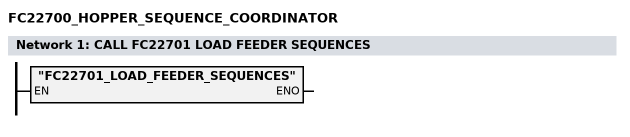
   RUNG wire#powerrail
      "FC22701_LOAD_FEEDER_SEQUENCES"()
   END_RUNG
   // the same network as SCL:
   "FC22701_LOAD_FEEDER_SEQUENCES"();
END_REGION
END_FUNCTION

FUNCTION "FC22701_LOAD_FEEDER_SEQUENCES" : Void   // FC22701, LAD
TITLE = FC22701 LOAD FEEDER SEQUENCES
{ S7_Optimized_Access := 'TRUE' }
VERSION : 0.1
// stored: AutoNumber false, IsIECCheckEnabled false, SetENOAutomatically false, UDAEnableTagReadback false
BEGIN

REGION Network 1: //////////_UNIT_01_//////////
END_REGION

REGION Network 2: /////_HOPPER_1_SEQUENCES_/////
END_REGION

REGION Network 3: CALL FB22701 LOAD FEEDER SEQUENCE TIME UNIT 01 HOPPER 1
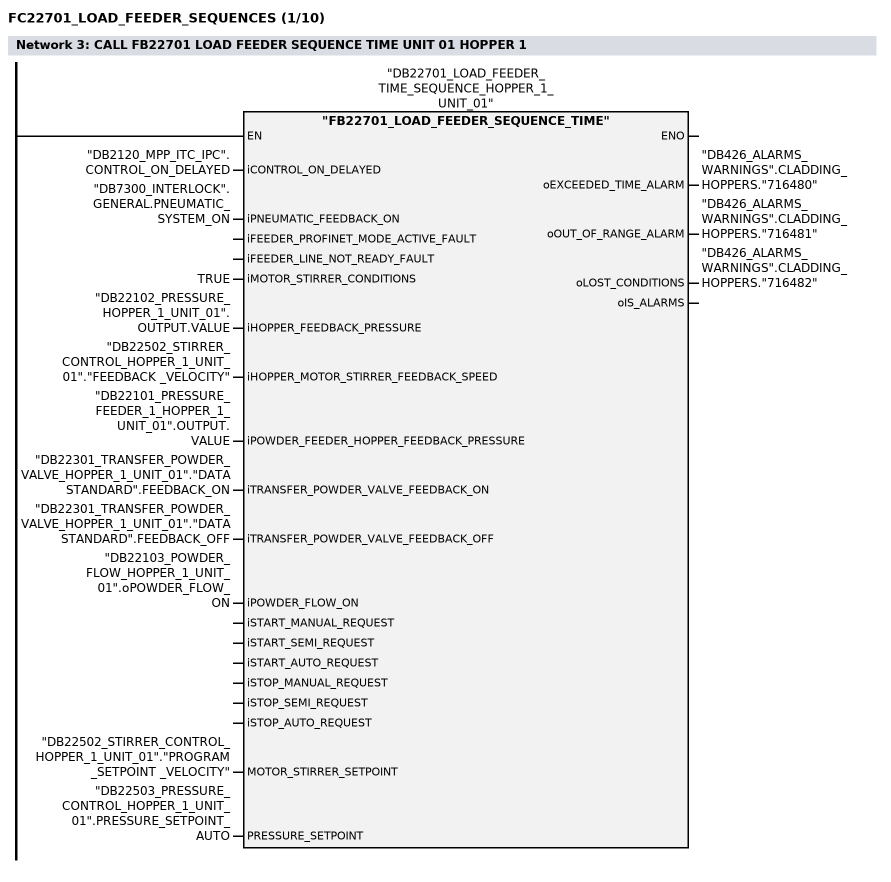
   RUNG wire#powerrail
      "DB22701_LOAD_FEEDER_TIME_SEQUENCE_HOPPER_1_UNIT_01"(iCONTROL_ON_DELAYED := "DB2120_MPP_ITC_IPC".CONTROL_ON_DELAYED, iPNEUMATIC_FEEDBACK_ON := "DB7300_INTERLOCK".GENERAL.PNEUMATIC_SYSTEM_ON, iFEEDER_PROFINET_MODE_ACTIVE_FAULT :=, iFEEDER_LINE_NOT_READY_FAULT :=, iMOTOR_STIRRER_CONDITIONS := TRUE, iHOPPER_FEEDBACK_PRESSURE := "DB22102_PRESSURE_HOPPER_1_UNIT_01".OUTPUT.VALUE, iHOPPER_MOTOR_STIRRER_FEEDBACK_SPEED := "DB22502_STIRRER_CONTROL_HOPPER_1_UNIT_01"."FEEDBACK _VELOCITY", iPOWDER_FEEDER_HOPPER_FEEDBACK_PRESSURE := "DB22101_PRESSURE_FEEDER_1_HOPPER_1_UNIT_01".OUTPUT.VALUE, iTRANSFER_POWDER_VALVE_FEEDBACK_ON := "DB22301_TRANSFER_POWDER_VALVE_HOPPER_1_UNIT_01"."DATA STANDARD".FEEDBACK_ON, iTRANSFER_POWDER_VALVE_FEEDBACK_OFF := "DB22301_TRANSFER_POWDER_VALVE_HOPPER_1_UNIT_01"."DATA STANDARD".FEEDBACK_OFF, iPOWDER_FLOW_ON := "DB22103_POWDER_FLOW_HOPPER_1_UNIT_01".oPOWDER_FLOW_ON, iSTART_MANUAL_REQUEST :=, iSTART_SEMI_REQUEST :=, iSTART_AUTO_REQUEST :=, iSTOP_MANUAL_REQUEST :=, iSTOP_SEMI_REQUEST :=, iSTOP_AUTO_REQUEST :=, MOTOR_STIRRER_SETPOINT := "DB22502_STIRRER_CONTROL_HOPPER_1_UNIT_01"."PROGRAM _SETPOINT _VELOCITY", PRESSURE_SETPOINT := "DB22503_PRESSURE_CONTROL_HOPPER_1_UNIT_01".PRESSURE_SETPOINT_AUTO, oEXCEEDED_TIME_ALARM => "DB426_ALARMS_WARNINGS".CLADDING_HOPPERS."716480", oOUT_OF_RANGE_ALARM => "DB426_ALARMS_WARNINGS".CLADDING_HOPPERS."716481", oLOST_CONDITIONS => "DB426_ALARMS_WARNINGS".CLADDING_HOPPERS."716482", oIS_ALARMS =>)
   END_RUNG
   // the same network as SCL:
   "DB22701_LOAD_FEEDER_TIME_SEQUENCE_HOPPER_1_UNIT_01"(iCONTROL_ON_DELAYED := "DB2120_MPP_ITC_IPC".CONTROL_ON_DELAYED,   // "FB22701_LOAD_FEEDER_SEQUENCE_TIME"
                           iPNEUMATIC_FEEDBACK_ON := "DB7300_INTERLOCK".GENERAL.PNEUMATIC_SYSTEM_ON,
                           iMOTOR_STIRRER_CONDITIONS := TRUE,
                           iHOPPER_FEEDBACK_PRESSURE := "DB22102_PRESSURE_HOPPER_1_UNIT_01".OUTPUT.VALUE,
                           iHOPPER_MOTOR_STIRRER_FEEDBACK_SPEED := "DB22502_STIRRER_CONTROL_HOPPER_1_UNIT_01"."FEEDBACK _VELOCITY",
                           iPOWDER_FEEDER_HOPPER_FEEDBACK_PRESSURE := "DB22101_PRESSURE_FEEDER_1_HOPPER_1_UNIT_01".OUTPUT.VALUE,
                           iTRANSFER_POWDER_VALVE_FEEDBACK_ON := "DB22301_TRANSFER_POWDER_VALVE_HOPPER_1_UNIT_01"."DATA STANDARD".FEEDBACK_ON,
                           iTRANSFER_POWDER_VALVE_FEEDBACK_OFF := "DB22301_TRANSFER_POWDER_VALVE_HOPPER_1_UNIT_01"."DATA STANDARD".FEEDBACK_OFF,
                           iPOWDER_FLOW_ON := "DB22103_POWDER_FLOW_HOPPER_1_UNIT_01".oPOWDER_FLOW_ON,
                           MOTOR_STIRRER_SETPOINT := "DB22502_STIRRER_CONTROL_HOPPER_1_UNIT_01"."PROGRAM _SETPOINT _VELOCITY",
                           PRESSURE_SETPOINT := "DB22503_PRESSURE_CONTROL_HOPPER_1_UNIT_01".PRESSURE_SETPOINT_AUTO,
                           oEXCEEDED_TIME_ALARM => "DB426_ALARMS_WARNINGS".CLADDING_HOPPERS."716480",
                           oOUT_OF_RANGE_ALARM => "DB426_ALARMS_WARNINGS".CLADDING_HOPPERS."716481",
                           oLOST_CONDITIONS => "DB426_ALARMS_WARNINGS".CLADDING_HOPPERS."716482");
END_REGION

REGION Network 4: CALL FB22702 LOAD FEEDER SEQUENCE WEIGHT UNIT 01 HOPPER 1
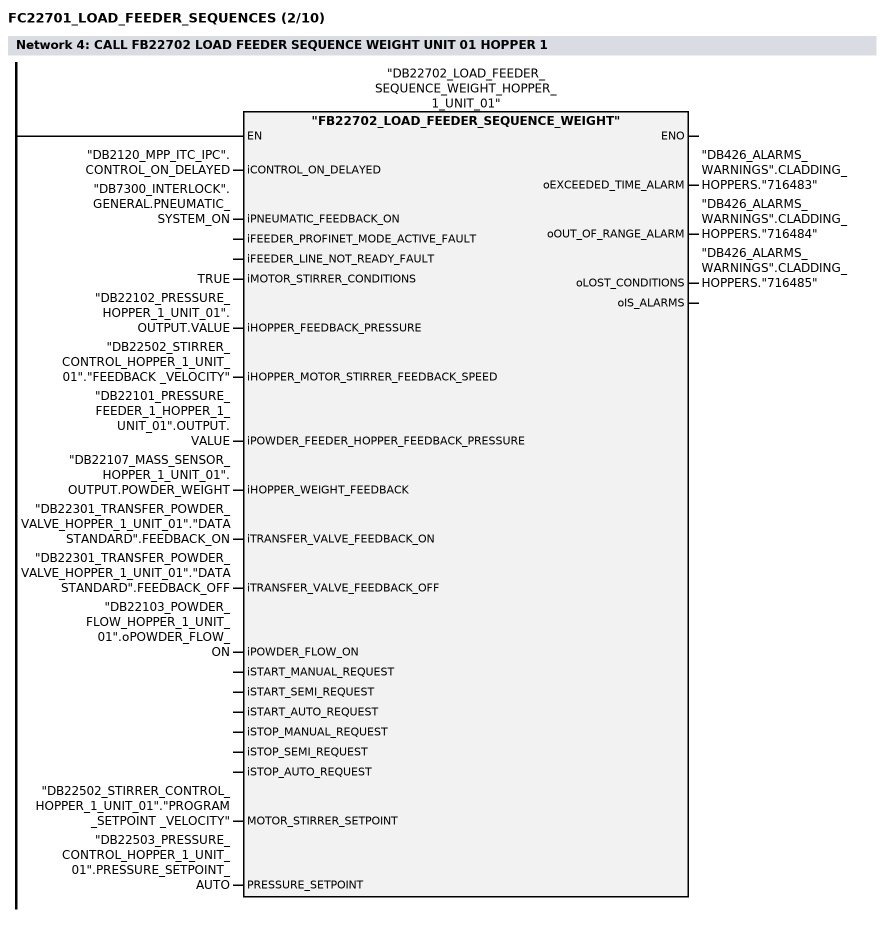
   RUNG wire#powerrail
      "DB22702_LOAD_FEEDER_SEQUENCE_WEIGHT_HOPPER_1_UNIT_01"(iCONTROL_ON_DELAYED := "DB2120_MPP_ITC_IPC".CONTROL_ON_DELAYED, iPNEUMATIC_FEEDBACK_ON := "DB7300_INTERLOCK".GENERAL.PNEUMATIC_SYSTEM_ON, iFEEDER_PROFINET_MODE_ACTIVE_FAULT :=, iFEEDER_LINE_NOT_READY_FAULT :=, iMOTOR_STIRRER_CONDITIONS := TRUE, iHOPPER_FEEDBACK_PRESSURE := "DB22102_PRESSURE_HOPPER_1_UNIT_01".OUTPUT.VALUE, iHOPPER_MOTOR_STIRRER_FEEDBACK_SPEED := "DB22502_STIRRER_CONTROL_HOPPER_1_UNIT_01"."FEEDBACK _VELOCITY", iPOWDER_FEEDER_HOPPER_FEEDBACK_PRESSURE := "DB22101_PRESSURE_FEEDER_1_HOPPER_1_UNIT_01".OUTPUT.VALUE, iHOPPER_WEIGHT_FEEDBACK := "DB22107_MASS_SENSOR_HOPPER_1_UNIT_01".OUTPUT.POWDER_WEIGHT, iTRANSFER_VALVE_FEEDBACK_ON := "DB22301_TRANSFER_POWDER_VALVE_HOPPER_1_UNIT_01"."DATA STANDARD".FEEDBACK_ON, iTRANSFER_VALVE_FEEDBACK_OFF := "DB22301_TRANSFER_POWDER_VALVE_HOPPER_1_UNIT_01"."DATA STANDARD".FEEDBACK_OFF, iPOWDER_FLOW_ON := "DB22103_POWDER_FLOW_HOPPER_1_UNIT_01".oPOWDER_FLOW_ON, iSTART_MANUAL_REQUEST :=, iSTART_SEMI_REQUEST :=, iSTART_AUTO_REQUEST :=, iSTOP_MANUAL_REQUEST :=, iSTOP_SEMI_REQUEST :=, iSTOP_AUTO_REQUEST :=, MOTOR_STIRRER_SETPOINT := "DB22502_STIRRER_CONTROL_HOPPER_1_UNIT_01"."PROGRAM _SETPOINT _VELOCITY", PRESSURE_SETPOINT := "DB22503_PRESSURE_CONTROL_HOPPER_1_UNIT_01".PRESSURE_SETPOINT_AUTO, oEXCEEDED_TIME_ALARM => "DB426_ALARMS_WARNINGS".CLADDING_HOPPERS."716483", oOUT_OF_RANGE_ALARM => "DB426_ALARMS_WARNINGS".CLADDING_HOPPERS."716484", oLOST_CONDITIONS => "DB426_ALARMS_WARNINGS".CLADDING_HOPPERS."716485", oIS_ALARMS =>)
   END_RUNG
   // the same network as SCL:
   "DB22702_LOAD_FEEDER_SEQUENCE_WEIGHT_HOPPER_1_UNIT_01"(iCONTROL_ON_DELAYED := "DB2120_MPP_ITC_IPC".CONTROL_ON_DELAYED,   // "FB22702_LOAD_FEEDER_SEQUENCE_WEIGHT"
                           iPNEUMATIC_FEEDBACK_ON := "DB7300_INTERLOCK".GENERAL.PNEUMATIC_SYSTEM_ON,
                           iMOTOR_STIRRER_CONDITIONS := TRUE,
                           iHOPPER_FEEDBACK_PRESSURE := "DB22102_PRESSURE_HOPPER_1_UNIT_01".OUTPUT.VALUE,
                           iHOPPER_MOTOR_STIRRER_FEEDBACK_SPEED := "DB22502_STIRRER_CONTROL_HOPPER_1_UNIT_01"."FEEDBACK _VELOCITY",
                           iPOWDER_FEEDER_HOPPER_FEEDBACK_PRESSURE := "DB22101_PRESSURE_FEEDER_1_HOPPER_1_UNIT_01".OUTPUT.VALUE,
                           iHOPPER_WEIGHT_FEEDBACK := "DB22107_MASS_SENSOR_HOPPER_1_UNIT_01".OUTPUT.POWDER_WEIGHT,
                           iTRANSFER_VALVE_FEEDBACK_ON := "DB22301_TRANSFER_POWDER_VALVE_HOPPER_1_UNIT_01"."DATA STANDARD".FEEDBACK_ON,
                           iTRANSFER_VALVE_FEEDBACK_OFF := "DB22301_TRANSFER_POWDER_VALVE_HOPPER_1_UNIT_01"."DATA STANDARD".FEEDBACK_OFF,
                           iPOWDER_FLOW_ON := "DB22103_POWDER_FLOW_HOPPER_1_UNIT_01".oPOWDER_FLOW_ON,
                           MOTOR_STIRRER_SETPOINT := "DB22502_STIRRER_CONTROL_HOPPER_1_UNIT_01"."PROGRAM _SETPOINT _VELOCITY",
                           PRESSURE_SETPOINT := "DB22503_PRESSURE_CONTROL_HOPPER_1_UNIT_01".PRESSURE_SETPOINT_AUTO,
                           oEXCEEDED_TIME_ALARM => "DB426_ALARMS_WARNINGS".CLADDING_HOPPERS."716483",
                           oOUT_OF_RANGE_ALARM => "DB426_ALARMS_WARNINGS".CLADDING_HOPPERS."716484",
                           oLOST_CONDITIONS => "DB426_ALARMS_WARNINGS".CLADDING_HOPPERS."716485");
END_REGION

REGION Network 5: /////_HOPPER_2_SEQUENCES_/////
END_REGION

REGION Network 6: CALL FB22701 LOAD FEEDER SEQUENCE TIME UNIT 01 HOPPER 2
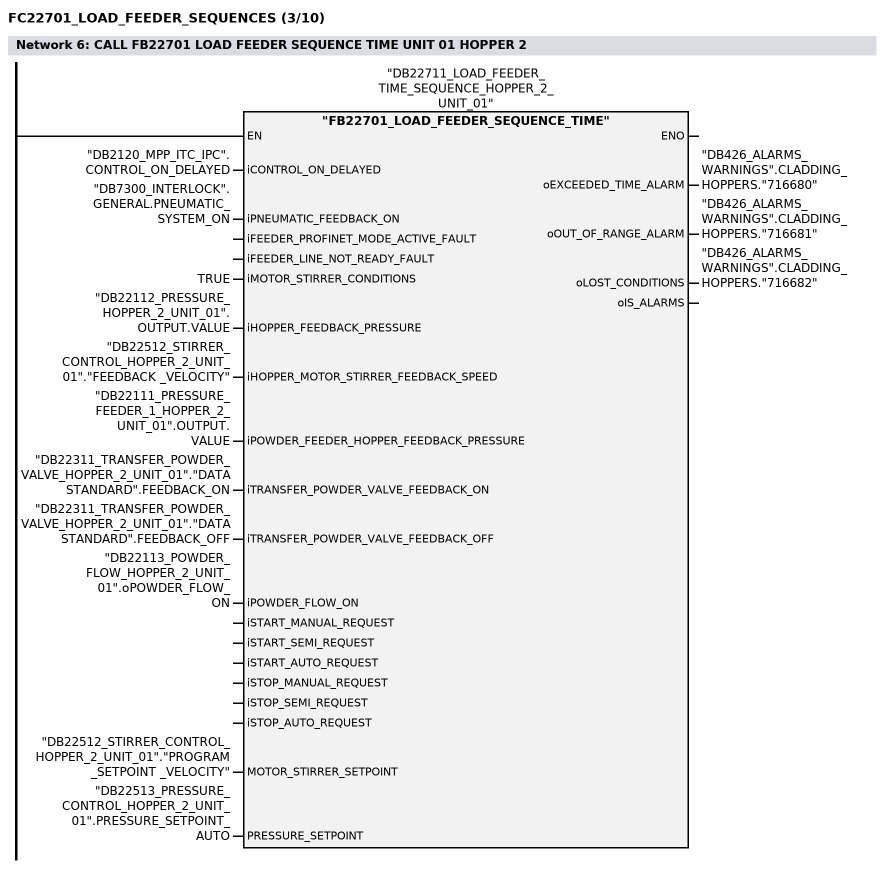
   RUNG wire#powerrail
      "DB22711_LOAD_FEEDER_TIME_SEQUENCE_HOPPER_2_UNIT_01"(iCONTROL_ON_DELAYED := "DB2120_MPP_ITC_IPC".CONTROL_ON_DELAYED, iPNEUMATIC_FEEDBACK_ON := "DB7300_INTERLOCK".GENERAL.PNEUMATIC_SYSTEM_ON, iFEEDER_PROFINET_MODE_ACTIVE_FAULT :=, iFEEDER_LINE_NOT_READY_FAULT :=, iMOTOR_STIRRER_CONDITIONS := TRUE, iHOPPER_FEEDBACK_PRESSURE := "DB22112_PRESSURE_HOPPER_2_UNIT_01".OUTPUT.VALUE, iHOPPER_MOTOR_STIRRER_FEEDBACK_SPEED := "DB22512_STIRRER_CONTROL_HOPPER_2_UNIT_01"."FEEDBACK _VELOCITY", iPOWDER_FEEDER_HOPPER_FEEDBACK_PRESSURE := "DB22111_PRESSURE_FEEDER_1_HOPPER_2_UNIT_01".OUTPUT.VALUE, iTRANSFER_POWDER_VALVE_FEEDBACK_ON := "DB22311_TRANSFER_POWDER_VALVE_HOPPER_2_UNIT_01"."DATA STANDARD".FEEDBACK_ON, iTRANSFER_POWDER_VALVE_FEEDBACK_OFF := "DB22311_TRANSFER_POWDER_VALVE_HOPPER_2_UNIT_01"."DATA STANDARD".FEEDBACK_OFF, iPOWDER_FLOW_ON := "DB22113_POWDER_FLOW_HOPPER_2_UNIT_01".oPOWDER_FLOW_ON, iSTART_MANUAL_REQUEST :=, iSTART_SEMI_REQUEST :=, iSTART_AUTO_REQUEST :=, iSTOP_MANUAL_REQUEST :=, iSTOP_SEMI_REQUEST :=, iSTOP_AUTO_REQUEST :=, MOTOR_STIRRER_SETPOINT := "DB22512_STIRRER_CONTROL_HOPPER_2_UNIT_01"."PROGRAM _SETPOINT _VELOCITY", PRESSURE_SETPOINT := "DB22513_PRESSURE_CONTROL_HOPPER_2_UNIT_01".PRESSURE_SETPOINT_AUTO, oEXCEEDED_TIME_ALARM => "DB426_ALARMS_WARNINGS".CLADDING_HOPPERS."716680", oOUT_OF_RANGE_ALARM => "DB426_ALARMS_WARNINGS".CLADDING_HOPPERS."716681", oLOST_CONDITIONS => "DB426_ALARMS_WARNINGS".CLADDING_HOPPERS."716682", oIS_ALARMS =>)
   END_RUNG
   // the same network as SCL:
   "DB22711_LOAD_FEEDER_TIME_SEQUENCE_HOPPER_2_UNIT_01"(iCONTROL_ON_DELAYED := "DB2120_MPP_ITC_IPC".CONTROL_ON_DELAYED,   // "FB22701_LOAD_FEEDER_SEQUENCE_TIME"
                           iPNEUMATIC_FEEDBACK_ON := "DB7300_INTERLOCK".GENERAL.PNEUMATIC_SYSTEM_ON,
                           iMOTOR_STIRRER_CONDITIONS := TRUE,
                           iHOPPER_FEEDBACK_PRESSURE := "DB22112_PRESSURE_HOPPER_2_UNIT_01".OUTPUT.VALUE,
                           iHOPPER_MOTOR_STIRRER_FEEDBACK_SPEED := "DB22512_STIRRER_CONTROL_HOPPER_2_UNIT_01"."FEEDBACK _VELOCITY",
                           iPOWDER_FEEDER_HOPPER_FEEDBACK_PRESSURE := "DB22111_PRESSURE_FEEDER_1_HOPPER_2_UNIT_01".OUTPUT.VALUE,
                           iTRANSFER_POWDER_VALVE_FEEDBACK_ON := "DB22311_TRANSFER_POWDER_VALVE_HOPPER_2_UNIT_01"."DATA STANDARD".FEEDBACK_ON,
                           iTRANSFER_POWDER_VALVE_FEEDBACK_OFF := "DB22311_TRANSFER_POWDER_VALVE_HOPPER_2_UNIT_01"."DATA STANDARD".FEEDBACK_OFF,
                           iPOWDER_FLOW_ON := "DB22113_POWDER_FLOW_HOPPER_2_UNIT_01".oPOWDER_FLOW_ON,
                           MOTOR_STIRRER_SETPOINT := "DB22512_STIRRER_CONTROL_HOPPER_2_UNIT_01"."PROGRAM _SETPOINT _VELOCITY",
                           PRESSURE_SETPOINT := "DB22513_PRESSURE_CONTROL_HOPPER_2_UNIT_01".PRESSURE_SETPOINT_AUTO,
                           oEXCEEDED_TIME_ALARM => "DB426_ALARMS_WARNINGS".CLADDING_HOPPERS."716680",
                           oOUT_OF_RANGE_ALARM => "DB426_ALARMS_WARNINGS".CLADDING_HOPPERS."716681",
                           oLOST_CONDITIONS => "DB426_ALARMS_WARNINGS".CLADDING_HOPPERS."716682");
END_REGION

REGION Network 7: CALL FB22702 LOAD FEEDER SEQUENCE WEIGHT UNIT 01 HOPPER 2
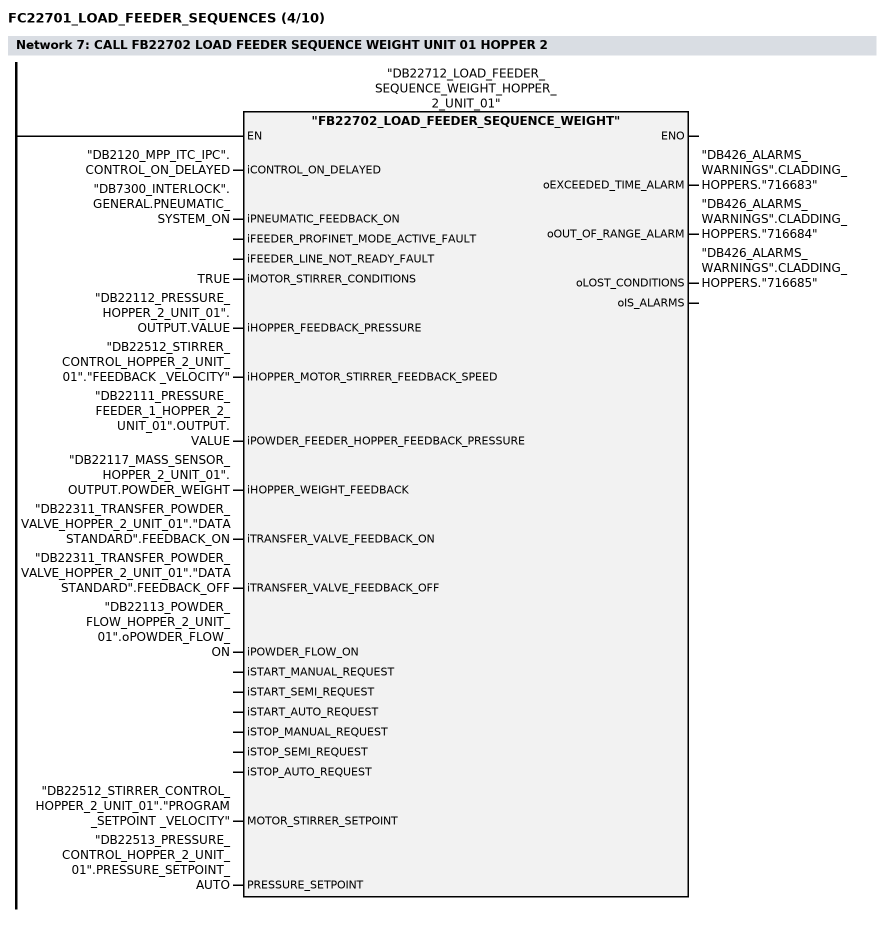
   RUNG wire#powerrail
      "DB22712_LOAD_FEEDER_SEQUENCE_WEIGHT_HOPPER_2_UNIT_01"(iCONTROL_ON_DELAYED := "DB2120_MPP_ITC_IPC".CONTROL_ON_DELAYED, iPNEUMATIC_FEEDBACK_ON := "DB7300_INTERLOCK".GENERAL.PNEUMATIC_SYSTEM_ON, iFEEDER_PROFINET_MODE_ACTIVE_FAULT :=, iFEEDER_LINE_NOT_READY_FAULT :=, iMOTOR_STIRRER_CONDITIONS := TRUE, iHOPPER_FEEDBACK_PRESSURE := "DB22112_PRESSURE_HOPPER_2_UNIT_01".OUTPUT.VALUE, iHOPPER_MOTOR_STIRRER_FEEDBACK_SPEED := "DB22512_STIRRER_CONTROL_HOPPER_2_UNIT_01"."FEEDBACK _VELOCITY", iPOWDER_FEEDER_HOPPER_FEEDBACK_PRESSURE := "DB22111_PRESSURE_FEEDER_1_HOPPER_2_UNIT_01".OUTPUT.VALUE, iHOPPER_WEIGHT_FEEDBACK := "DB22117_MASS_SENSOR_HOPPER_2_UNIT_01".OUTPUT.POWDER_WEIGHT, iTRANSFER_VALVE_FEEDBACK_ON := "DB22311_TRANSFER_POWDER_VALVE_HOPPER_2_UNIT_01"."DATA STANDARD".FEEDBACK_ON, iTRANSFER_VALVE_FEEDBACK_OFF := "DB22311_TRANSFER_POWDER_VALVE_HOPPER_2_UNIT_01"."DATA STANDARD".FEEDBACK_OFF, iPOWDER_FLOW_ON := "DB22113_POWDER_FLOW_HOPPER_2_UNIT_01".oPOWDER_FLOW_ON, iSTART_MANUAL_REQUEST :=, iSTART_SEMI_REQUEST :=, iSTART_AUTO_REQUEST :=, iSTOP_MANUAL_REQUEST :=, iSTOP_SEMI_REQUEST :=, iSTOP_AUTO_REQUEST :=, MOTOR_STIRRER_SETPOINT := "DB22512_STIRRER_CONTROL_HOPPER_2_UNIT_01"."PROGRAM _SETPOINT _VELOCITY", PRESSURE_SETPOINT := "DB22513_PRESSURE_CONTROL_HOPPER_2_UNIT_01".PRESSURE_SETPOINT_AUTO, oEXCEEDED_TIME_ALARM => "DB426_ALARMS_WARNINGS".CLADDING_HOPPERS."716683", oOUT_OF_RANGE_ALARM => "DB426_ALARMS_WARNINGS".CLADDING_HOPPERS."716684", oLOST_CONDITIONS => "DB426_ALARMS_WARNINGS".CLADDING_HOPPERS."716685", oIS_ALARMS =>)
   END_RUNG
   // the same network as SCL:
   "DB22712_LOAD_FEEDER_SEQUENCE_WEIGHT_HOPPER_2_UNIT_01"(iCONTROL_ON_DELAYED := "DB2120_MPP_ITC_IPC".CONTROL_ON_DELAYED,   // "FB22702_LOAD_FEEDER_SEQUENCE_WEIGHT"
                           iPNEUMATIC_FEEDBACK_ON := "DB7300_INTERLOCK".GENERAL.PNEUMATIC_SYSTEM_ON,
                           iMOTOR_STIRRER_CONDITIONS := TRUE,
                           iHOPPER_FEEDBACK_PRESSURE := "DB22112_PRESSURE_HOPPER_2_UNIT_01".OUTPUT.VALUE,
                           iHOPPER_MOTOR_STIRRER_FEEDBACK_SPEED := "DB22512_STIRRER_CONTROL_HOPPER_2_UNIT_01"."FEEDBACK _VELOCITY",
                           iPOWDER_FEEDER_HOPPER_FEEDBACK_PRESSURE := "DB22111_PRESSURE_FEEDER_1_HOPPER_2_UNIT_01".OUTPUT.VALUE,
                           iHOPPER_WEIGHT_FEEDBACK := "DB22117_MASS_SENSOR_HOPPER_2_UNIT_01".OUTPUT.POWDER_WEIGHT,
                           iTRANSFER_VALVE_FEEDBACK_ON := "DB22311_TRANSFER_POWDER_VALVE_HOPPER_2_UNIT_01"."DATA STANDARD".FEEDBACK_ON,
                           iTRANSFER_VALVE_FEEDBACK_OFF := "DB22311_TRANSFER_POWDER_VALVE_HOPPER_2_UNIT_01"."DATA STANDARD".FEEDBACK_OFF,
                           iPOWDER_FLOW_ON := "DB22113_POWDER_FLOW_HOPPER_2_UNIT_01".oPOWDER_FLOW_ON,
                           MOTOR_STIRRER_SETPOINT := "DB22512_STIRRER_CONTROL_HOPPER_2_UNIT_01"."PROGRAM _SETPOINT _VELOCITY",
                           PRESSURE_SETPOINT := "DB22513_PRESSURE_CONTROL_HOPPER_2_UNIT_01".PRESSURE_SETPOINT_AUTO,
                           oEXCEEDED_TIME_ALARM => "DB426_ALARMS_WARNINGS".CLADDING_HOPPERS."716683",
                           oOUT_OF_RANGE_ALARM => "DB426_ALARMS_WARNINGS".CLADDING_HOPPERS."716684",
                           oLOST_CONDITIONS => "DB426_ALARMS_WARNINGS".CLADDING_HOPPERS."716685");
END_REGION

REGION Network 8: //////////_UNIT_02_//////////
END_REGION

REGION Network 9: /////_HOPPER_1_SEQUENCES_/////
END_REGION

REGION Network 10: CALL FB22701 LOAD FEEDER SEQUENCE TIME UNIT 02 HOPPER 1
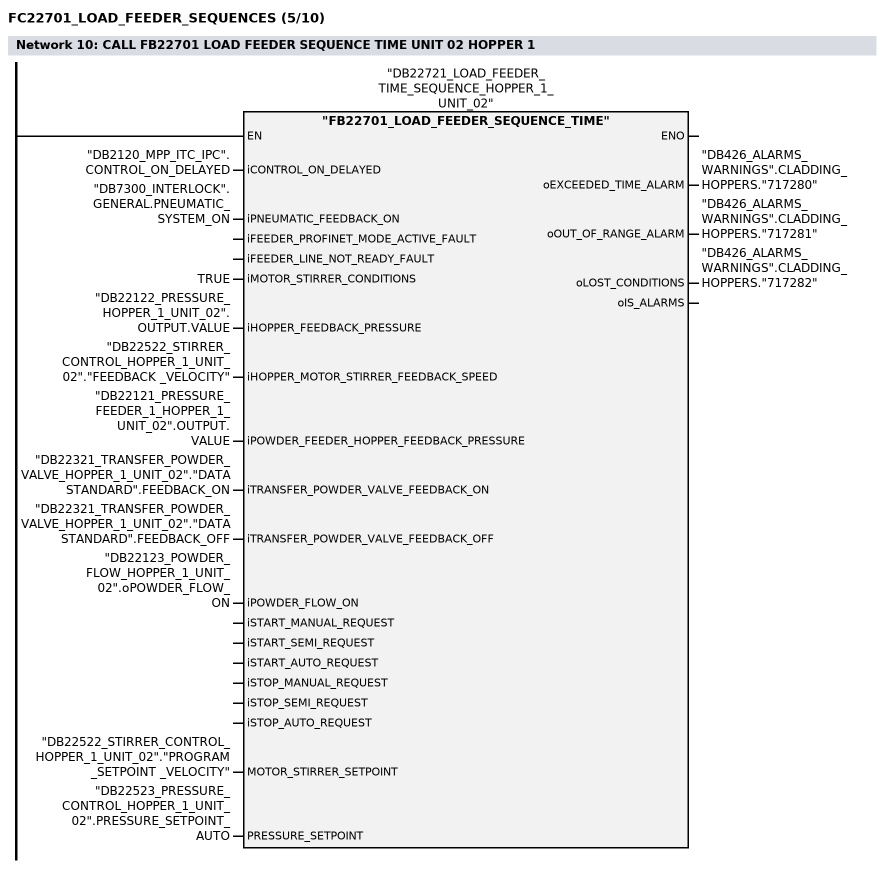
   RUNG wire#powerrail
      "DB22721_LOAD_FEEDER_TIME_SEQUENCE_HOPPER_1_UNIT_02"(iCONTROL_ON_DELAYED := "DB2120_MPP_ITC_IPC".CONTROL_ON_DELAYED, iPNEUMATIC_FEEDBACK_ON := "DB7300_INTERLOCK".GENERAL.PNEUMATIC_SYSTEM_ON, iFEEDER_PROFINET_MODE_ACTIVE_FAULT :=, iFEEDER_LINE_NOT_READY_FAULT :=, iMOTOR_STIRRER_CONDITIONS := TRUE, iHOPPER_FEEDBACK_PRESSURE := "DB22122_PRESSURE_HOPPER_1_UNIT_02".OUTPUT.VALUE, iHOPPER_MOTOR_STIRRER_FEEDBACK_SPEED := "DB22522_STIRRER_CONTROL_HOPPER_1_UNIT_02"."FEEDBACK _VELOCITY", iPOWDER_FEEDER_HOPPER_FEEDBACK_PRESSURE := "DB22121_PRESSURE_FEEDER_1_HOPPER_1_UNIT_02".OUTPUT.VALUE, iTRANSFER_POWDER_VALVE_FEEDBACK_ON := "DB22321_TRANSFER_POWDER_VALVE_HOPPER_1_UNIT_02"."DATA STANDARD".FEEDBACK_ON, iTRANSFER_POWDER_VALVE_FEEDBACK_OFF := "DB22321_TRANSFER_POWDER_VALVE_HOPPER_1_UNIT_02"."DATA STANDARD".FEEDBACK_OFF, iPOWDER_FLOW_ON := "DB22123_POWDER_FLOW_HOPPER_1_UNIT_02".oPOWDER_FLOW_ON, iSTART_MANUAL_REQUEST :=, iSTART_SEMI_REQUEST :=, iSTART_AUTO_REQUEST :=, iSTOP_MANUAL_REQUEST :=, iSTOP_SEMI_REQUEST :=, iSTOP_AUTO_REQUEST :=, MOTOR_STIRRER_SETPOINT := "DB22522_STIRRER_CONTROL_HOPPER_1_UNIT_02"."PROGRAM _SETPOINT _VELOCITY", PRESSURE_SETPOINT := "DB22523_PRESSURE_CONTROL_HOPPER_1_UNIT_02".PRESSURE_SETPOINT_AUTO, oEXCEEDED_TIME_ALARM => "DB426_ALARMS_WARNINGS".CLADDING_HOPPERS."717280", oOUT_OF_RANGE_ALARM => "DB426_ALARMS_WARNINGS".CLADDING_HOPPERS."717281", oLOST_CONDITIONS => "DB426_ALARMS_WARNINGS".CLADDING_HOPPERS."717282", oIS_ALARMS =>)
   END_RUNG
   // the same network as SCL:
   "DB22721_LOAD_FEEDER_TIME_SEQUENCE_HOPPER_1_UNIT_02"(iCONTROL_ON_DELAYED := "DB2120_MPP_ITC_IPC".CONTROL_ON_DELAYED,   // "FB22701_LOAD_FEEDER_SEQUENCE_TIME"
                           iPNEUMATIC_FEEDBACK_ON := "DB7300_INTERLOCK".GENERAL.PNEUMATIC_SYSTEM_ON,
                           iMOTOR_STIRRER_CONDITIONS := TRUE,
                           iHOPPER_FEEDBACK_PRESSURE := "DB22122_PRESSURE_HOPPER_1_UNIT_02".OUTPUT.VALUE,
                           iHOPPER_MOTOR_STIRRER_FEEDBACK_SPEED := "DB22522_STIRRER_CONTROL_HOPPER_1_UNIT_02"."FEEDBACK _VELOCITY",
                           iPOWDER_FEEDER_HOPPER_FEEDBACK_PRESSURE := "DB22121_PRESSURE_FEEDER_1_HOPPER_1_UNIT_02".OUTPUT.VALUE,
                           iTRANSFER_POWDER_VALVE_FEEDBACK_ON := "DB22321_TRANSFER_POWDER_VALVE_HOPPER_1_UNIT_02"."DATA STANDARD".FEEDBACK_ON,
                           iTRANSFER_POWDER_VALVE_FEEDBACK_OFF := "DB22321_TRANSFER_POWDER_VALVE_HOPPER_1_UNIT_02"."DATA STANDARD".FEEDBACK_OFF,
                           iPOWDER_FLOW_ON := "DB22123_POWDER_FLOW_HOPPER_1_UNIT_02".oPOWDER_FLOW_ON,
                           MOTOR_STIRRER_SETPOINT := "DB22522_STIRRER_CONTROL_HOPPER_1_UNIT_02"."PROGRAM _SETPOINT _VELOCITY",
                           PRESSURE_SETPOINT := "DB22523_PRESSURE_CONTROL_HOPPER_1_UNIT_02".PRESSURE_SETPOINT_AUTO,
                           oEXCEEDED_TIME_ALARM => "DB426_ALARMS_WARNINGS".CLADDING_HOPPERS."717280",
                           oOUT_OF_RANGE_ALARM => "DB426_ALARMS_WARNINGS".CLADDING_HOPPERS."717281",
                           oLOST_CONDITIONS => "DB426_ALARMS_WARNINGS".CLADDING_HOPPERS."717282");
END_REGION

REGION Network 11: CALL FB22702 LOAD FEEDER SEQUENCE WEIGHT UNIT 02 HOPPER 1
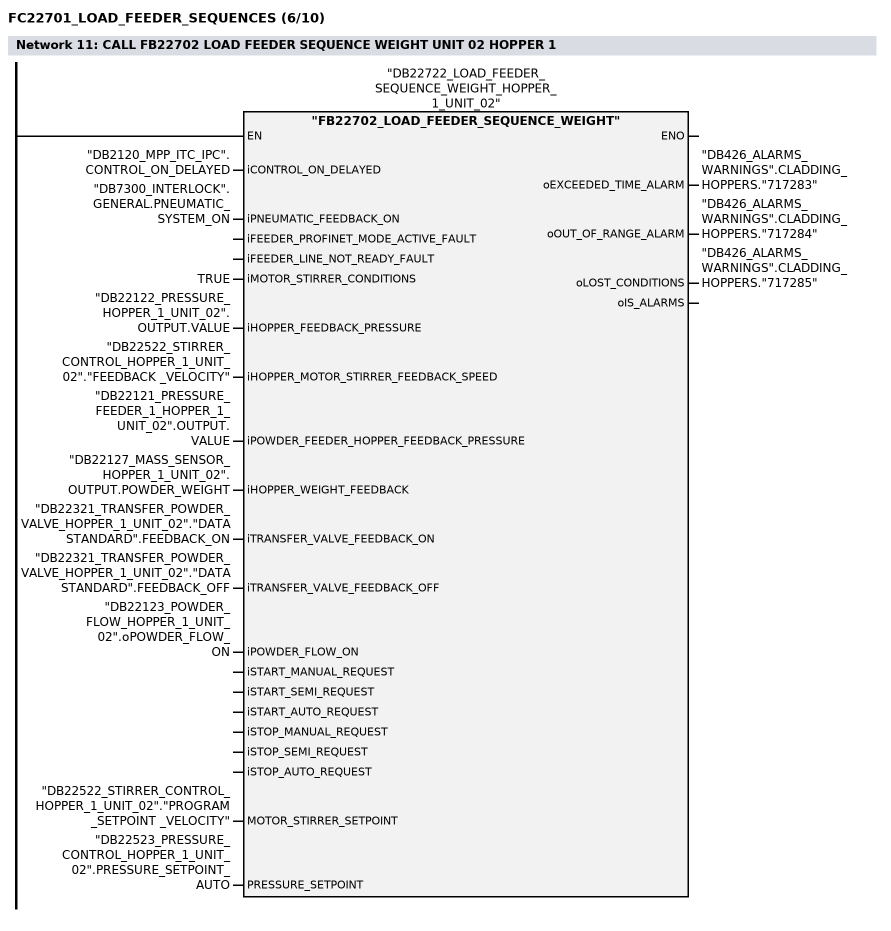
   RUNG wire#powerrail
      "DB22722_LOAD_FEEDER_SEQUENCE_WEIGHT_HOPPER_1_UNIT_02"(iCONTROL_ON_DELAYED := "DB2120_MPP_ITC_IPC".CONTROL_ON_DELAYED, iPNEUMATIC_FEEDBACK_ON := "DB7300_INTERLOCK".GENERAL.PNEUMATIC_SYSTEM_ON, iFEEDER_PROFINET_MODE_ACTIVE_FAULT :=, iFEEDER_LINE_NOT_READY_FAULT :=, iMOTOR_STIRRER_CONDITIONS := TRUE, iHOPPER_FEEDBACK_PRESSURE := "DB22122_PRESSURE_HOPPER_1_UNIT_02".OUTPUT.VALUE, iHOPPER_MOTOR_STIRRER_FEEDBACK_SPEED := "DB22522_STIRRER_CONTROL_HOPPER_1_UNIT_02"."FEEDBACK _VELOCITY", iPOWDER_FEEDER_HOPPER_FEEDBACK_PRESSURE := "DB22121_PRESSURE_FEEDER_1_HOPPER_1_UNIT_02".OUTPUT.VALUE, iHOPPER_WEIGHT_FEEDBACK := "DB22127_MASS_SENSOR_HOPPER_1_UNIT_02".OUTPUT.POWDER_WEIGHT, iTRANSFER_VALVE_FEEDBACK_ON := "DB22321_TRANSFER_POWDER_VALVE_HOPPER_1_UNIT_02"."DATA STANDARD".FEEDBACK_ON, iTRANSFER_VALVE_FEEDBACK_OFF := "DB22321_TRANSFER_POWDER_VALVE_HOPPER_1_UNIT_02"."DATA STANDARD".FEEDBACK_OFF, iPOWDER_FLOW_ON := "DB22123_POWDER_FLOW_HOPPER_1_UNIT_02".oPOWDER_FLOW_ON, iSTART_MANUAL_REQUEST :=, iSTART_SEMI_REQUEST :=, iSTART_AUTO_REQUEST :=, iSTOP_MANUAL_REQUEST :=, iSTOP_SEMI_REQUEST :=, iSTOP_AUTO_REQUEST :=, MOTOR_STIRRER_SETPOINT := "DB22522_STIRRER_CONTROL_HOPPER_1_UNIT_02"."PROGRAM _SETPOINT _VELOCITY", PRESSURE_SETPOINT := "DB22523_PRESSURE_CONTROL_HOPPER_1_UNIT_02".PRESSURE_SETPOINT_AUTO, oEXCEEDED_TIME_ALARM => "DB426_ALARMS_WARNINGS".CLADDING_HOPPERS."717283", oOUT_OF_RANGE_ALARM => "DB426_ALARMS_WARNINGS".CLADDING_HOPPERS."717284", oLOST_CONDITIONS => "DB426_ALARMS_WARNINGS".CLADDING_HOPPERS."717285", oIS_ALARMS =>)
   END_RUNG
   // the same network as SCL:
   "DB22722_LOAD_FEEDER_SEQUENCE_WEIGHT_HOPPER_1_UNIT_02"(iCONTROL_ON_DELAYED := "DB2120_MPP_ITC_IPC".CONTROL_ON_DELAYED,   // "FB22702_LOAD_FEEDER_SEQUENCE_WEIGHT"
                           iPNEUMATIC_FEEDBACK_ON := "DB7300_INTERLOCK".GENERAL.PNEUMATIC_SYSTEM_ON,
                           iMOTOR_STIRRER_CONDITIONS := TRUE,
                           iHOPPER_FEEDBACK_PRESSURE := "DB22122_PRESSURE_HOPPER_1_UNIT_02".OUTPUT.VALUE,
                           iHOPPER_MOTOR_STIRRER_FEEDBACK_SPEED := "DB22522_STIRRER_CONTROL_HOPPER_1_UNIT_02"."FEEDBACK _VELOCITY",
                           iPOWDER_FEEDER_HOPPER_FEEDBACK_PRESSURE := "DB22121_PRESSURE_FEEDER_1_HOPPER_1_UNIT_02".OUTPUT.VALUE,
                           iHOPPER_WEIGHT_FEEDBACK := "DB22127_MASS_SENSOR_HOPPER_1_UNIT_02".OUTPUT.POWDER_WEIGHT,
                           iTRANSFER_VALVE_FEEDBACK_ON := "DB22321_TRANSFER_POWDER_VALVE_HOPPER_1_UNIT_02"."DATA STANDARD".FEEDBACK_ON,
                           iTRANSFER_VALVE_FEEDBACK_OFF := "DB22321_TRANSFER_POWDER_VALVE_HOPPER_1_UNIT_02"."DATA STANDARD".FEEDBACK_OFF,
                           iPOWDER_FLOW_ON := "DB22123_POWDER_FLOW_HOPPER_1_UNIT_02".oPOWDER_FLOW_ON,
                           MOTOR_STIRRER_SETPOINT := "DB22522_STIRRER_CONTROL_HOPPER_1_UNIT_02"."PROGRAM _SETPOINT _VELOCITY",
                           PRESSURE_SETPOINT := "DB22523_PRESSURE_CONTROL_HOPPER_1_UNIT_02".PRESSURE_SETPOINT_AUTO,
                           oEXCEEDED_TIME_ALARM => "DB426_ALARMS_WARNINGS".CLADDING_HOPPERS."717283",
                           oOUT_OF_RANGE_ALARM => "DB426_ALARMS_WARNINGS".CLADDING_HOPPERS."717284",
                           oLOST_CONDITIONS => "DB426_ALARMS_WARNINGS".CLADDING_HOPPERS."717285");
END_REGION

REGION Network 12: /////_HOPPER_2_SEQUENCES_/////
END_REGION

REGION Network 13: CALL FB22701 LOAD FEEDER SEQUENCE TIME UNIT 02 HOPPER 2
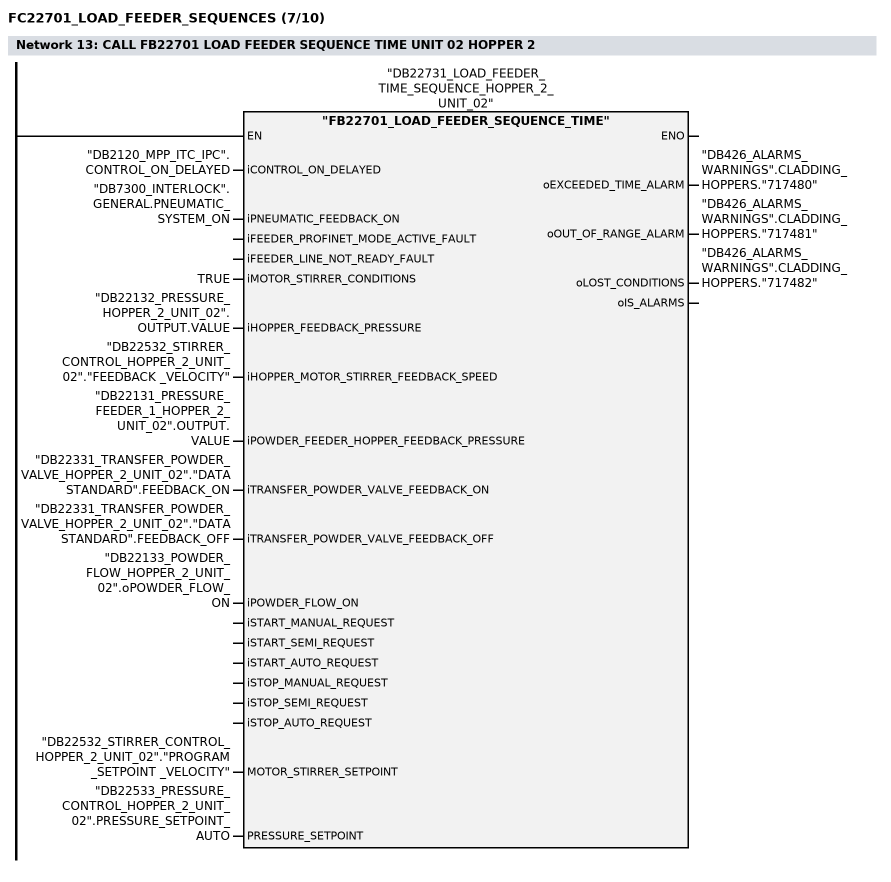
   RUNG wire#powerrail
      "DB22731_LOAD_FEEDER_TIME_SEQUENCE_HOPPER_2_UNIT_02"(iCONTROL_ON_DELAYED := "DB2120_MPP_ITC_IPC".CONTROL_ON_DELAYED, iPNEUMATIC_FEEDBACK_ON := "DB7300_INTERLOCK".GENERAL.PNEUMATIC_SYSTEM_ON, iFEEDER_PROFINET_MODE_ACTIVE_FAULT :=, iFEEDER_LINE_NOT_READY_FAULT :=, iMOTOR_STIRRER_CONDITIONS := TRUE, iHOPPER_FEEDBACK_PRESSURE := "DB22132_PRESSURE_HOPPER_2_UNIT_02".OUTPUT.VALUE, iHOPPER_MOTOR_STIRRER_FEEDBACK_SPEED := "DB22532_STIRRER_CONTROL_HOPPER_2_UNIT_02"."FEEDBACK _VELOCITY", iPOWDER_FEEDER_HOPPER_FEEDBACK_PRESSURE := "DB22131_PRESSURE_FEEDER_1_HOPPER_2_UNIT_02".OUTPUT.VALUE, iTRANSFER_POWDER_VALVE_FEEDBACK_ON := "DB22331_TRANSFER_POWDER_VALVE_HOPPER_2_UNIT_02"."DATA STANDARD".FEEDBACK_ON, iTRANSFER_POWDER_VALVE_FEEDBACK_OFF := "DB22331_TRANSFER_POWDER_VALVE_HOPPER_2_UNIT_02"."DATA STANDARD".FEEDBACK_OFF, iPOWDER_FLOW_ON := "DB22133_POWDER_FLOW_HOPPER_2_UNIT_02".oPOWDER_FLOW_ON, iSTART_MANUAL_REQUEST :=, iSTART_SEMI_REQUEST :=, iSTART_AUTO_REQUEST :=, iSTOP_MANUAL_REQUEST :=, iSTOP_SEMI_REQUEST :=, iSTOP_AUTO_REQUEST :=, MOTOR_STIRRER_SETPOINT := "DB22532_STIRRER_CONTROL_HOPPER_2_UNIT_02"."PROGRAM _SETPOINT _VELOCITY", PRESSURE_SETPOINT := "DB22533_PRESSURE_CONTROL_HOPPER_2_UNIT_02".PRESSURE_SETPOINT_AUTO, oEXCEEDED_TIME_ALARM => "DB426_ALARMS_WARNINGS".CLADDING_HOPPERS."717480", oOUT_OF_RANGE_ALARM => "DB426_ALARMS_WARNINGS".CLADDING_HOPPERS."717481", oLOST_CONDITIONS => "DB426_ALARMS_WARNINGS".CLADDING_HOPPERS."717482", oIS_ALARMS =>)
   END_RUNG
   // the same network as SCL:
   "DB22731_LOAD_FEEDER_TIME_SEQUENCE_HOPPER_2_UNIT_02"(iCONTROL_ON_DELAYED := "DB2120_MPP_ITC_IPC".CONTROL_ON_DELAYED,   // "FB22701_LOAD_FEEDER_SEQUENCE_TIME"
                           iPNEUMATIC_FEEDBACK_ON := "DB7300_INTERLOCK".GENERAL.PNEUMATIC_SYSTEM_ON,
                           iMOTOR_STIRRER_CONDITIONS := TRUE,
                           iHOPPER_FEEDBACK_PRESSURE := "DB22132_PRESSURE_HOPPER_2_UNIT_02".OUTPUT.VALUE,
                           iHOPPER_MOTOR_STIRRER_FEEDBACK_SPEED := "DB22532_STIRRER_CONTROL_HOPPER_2_UNIT_02"."FEEDBACK _VELOCITY",
                           iPOWDER_FEEDER_HOPPER_FEEDBACK_PRESSURE := "DB22131_PRESSURE_FEEDER_1_HOPPER_2_UNIT_02".OUTPUT.VALUE,
                           iTRANSFER_POWDER_VALVE_FEEDBACK_ON := "DB22331_TRANSFER_POWDER_VALVE_HOPPER_2_UNIT_02"."DATA STANDARD".FEEDBACK_ON,
                           iTRANSFER_POWDER_VALVE_FEEDBACK_OFF := "DB22331_TRANSFER_POWDER_VALVE_HOPPER_2_UNIT_02"."DATA STANDARD".FEEDBACK_OFF,
                           iPOWDER_FLOW_ON := "DB22133_POWDER_FLOW_HOPPER_2_UNIT_02".oPOWDER_FLOW_ON,
                           MOTOR_STIRRER_SETPOINT := "DB22532_STIRRER_CONTROL_HOPPER_2_UNIT_02"."PROGRAM _SETPOINT _VELOCITY",
                           PRESSURE_SETPOINT := "DB22533_PRESSURE_CONTROL_HOPPER_2_UNIT_02".PRESSURE_SETPOINT_AUTO,
                           oEXCEEDED_TIME_ALARM => "DB426_ALARMS_WARNINGS".CLADDING_HOPPERS."717480",
                           oOUT_OF_RANGE_ALARM => "DB426_ALARMS_WARNINGS".CLADDING_HOPPERS."717481",
                           oLOST_CONDITIONS => "DB426_ALARMS_WARNINGS".CLADDING_HOPPERS."717482");
END_REGION

REGION Network 14: CALL FB22702 LOAD FEEDER SEQUENCE WEIGHT UNIT 02 HOPPER 2
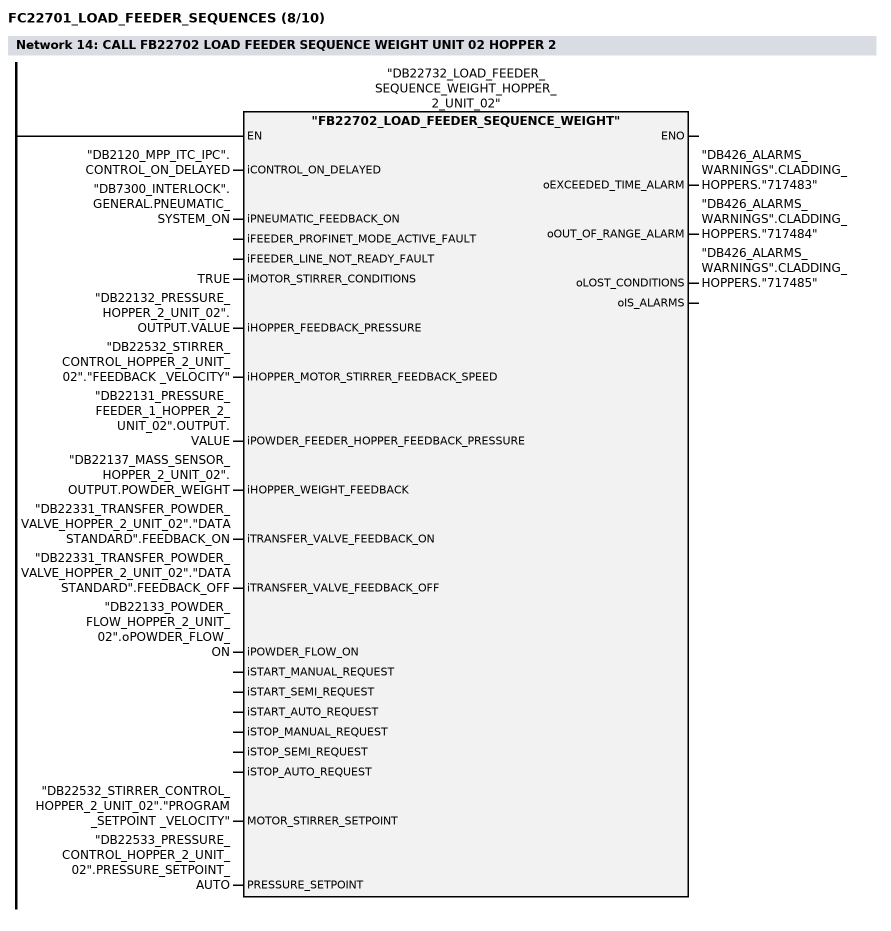
   RUNG wire#powerrail
      "DB22732_LOAD_FEEDER_SEQUENCE_WEIGHT_HOPPER_2_UNIT_02"(iCONTROL_ON_DELAYED := "DB2120_MPP_ITC_IPC".CONTROL_ON_DELAYED, iPNEUMATIC_FEEDBACK_ON := "DB7300_INTERLOCK".GENERAL.PNEUMATIC_SYSTEM_ON, iFEEDER_PROFINET_MODE_ACTIVE_FAULT :=, iFEEDER_LINE_NOT_READY_FAULT :=, iMOTOR_STIRRER_CONDITIONS := TRUE, iHOPPER_FEEDBACK_PRESSURE := "DB22132_PRESSURE_HOPPER_2_UNIT_02".OUTPUT.VALUE, iHOPPER_MOTOR_STIRRER_FEEDBACK_SPEED := "DB22532_STIRRER_CONTROL_HOPPER_2_UNIT_02"."FEEDBACK _VELOCITY", iPOWDER_FEEDER_HOPPER_FEEDBACK_PRESSURE := "DB22131_PRESSURE_FEEDER_1_HOPPER_2_UNIT_02".OUTPUT.VALUE, iHOPPER_WEIGHT_FEEDBACK := "DB22137_MASS_SENSOR_HOPPER_2_UNIT_02".OUTPUT.POWDER_WEIGHT, iTRANSFER_VALVE_FEEDBACK_ON := "DB22331_TRANSFER_POWDER_VALVE_HOPPER_2_UNIT_02"."DATA STANDARD".FEEDBACK_ON, iTRANSFER_VALVE_FEEDBACK_OFF := "DB22331_TRANSFER_POWDER_VALVE_HOPPER_2_UNIT_02"."DATA STANDARD".FEEDBACK_OFF, iPOWDER_FLOW_ON := "DB22133_POWDER_FLOW_HOPPER_2_UNIT_02".oPOWDER_FLOW_ON, iSTART_MANUAL_REQUEST :=, iSTART_SEMI_REQUEST :=, iSTART_AUTO_REQUEST :=, iSTOP_MANUAL_REQUEST :=, iSTOP_SEMI_REQUEST :=, iSTOP_AUTO_REQUEST :=, MOTOR_STIRRER_SETPOINT := "DB22532_STIRRER_CONTROL_HOPPER_2_UNIT_02"."PROGRAM _SETPOINT _VELOCITY", PRESSURE_SETPOINT := "DB22533_PRESSURE_CONTROL_HOPPER_2_UNIT_02".PRESSURE_SETPOINT_AUTO, oEXCEEDED_TIME_ALARM => "DB426_ALARMS_WARNINGS".CLADDING_HOPPERS."717483", oOUT_OF_RANGE_ALARM => "DB426_ALARMS_WARNINGS".CLADDING_HOPPERS."717484", oLOST_CONDITIONS => "DB426_ALARMS_WARNINGS".CLADDING_HOPPERS."717485", oIS_ALARMS =>)
   END_RUNG
   // the same network as SCL:
   "DB22732_LOAD_FEEDER_SEQUENCE_WEIGHT_HOPPER_2_UNIT_02"(iCONTROL_ON_DELAYED := "DB2120_MPP_ITC_IPC".CONTROL_ON_DELAYED,   // "FB22702_LOAD_FEEDER_SEQUENCE_WEIGHT"
                           iPNEUMATIC_FEEDBACK_ON := "DB7300_INTERLOCK".GENERAL.PNEUMATIC_SYSTEM_ON,
                           iMOTOR_STIRRER_CONDITIONS := TRUE,
                           iHOPPER_FEEDBACK_PRESSURE := "DB22132_PRESSURE_HOPPER_2_UNIT_02".OUTPUT.VALUE,
                           iHOPPER_MOTOR_STIRRER_FEEDBACK_SPEED := "DB22532_STIRRER_CONTROL_HOPPER_2_UNIT_02"."FEEDBACK _VELOCITY",
                           iPOWDER_FEEDER_HOPPER_FEEDBACK_PRESSURE := "DB22131_PRESSURE_FEEDER_1_HOPPER_2_UNIT_02".OUTPUT.VALUE,
                           iHOPPER_WEIGHT_FEEDBACK := "DB22137_MASS_SENSOR_HOPPER_2_UNIT_02".OUTPUT.POWDER_WEIGHT,
                           iTRANSFER_VALVE_FEEDBACK_ON := "DB22331_TRANSFER_POWDER_VALVE_HOPPER_2_UNIT_02"."DATA STANDARD".FEEDBACK_ON,
                           iTRANSFER_VALVE_FEEDBACK_OFF := "DB22331_TRANSFER_POWDER_VALVE_HOPPER_2_UNIT_02"."DATA STANDARD".FEEDBACK_OFF,
                           iPOWDER_FLOW_ON := "DB22133_POWDER_FLOW_HOPPER_2_UNIT_02".oPOWDER_FLOW_ON,
                           MOTOR_STIRRER_SETPOINT := "DB22532_STIRRER_CONTROL_HOPPER_2_UNIT_02"."PROGRAM _SETPOINT _VELOCITY",
                           PRESSURE_SETPOINT := "DB22533_PRESSURE_CONTROL_HOPPER_2_UNIT_02".PRESSURE_SETPOINT_AUTO,
                           oEXCEEDED_TIME_ALARM => "DB426_ALARMS_WARNINGS".CLADDING_HOPPERS."717483",
                           oOUT_OF_RANGE_ALARM => "DB426_ALARMS_WARNINGS".CLADDING_HOPPERS."717484",
                           oLOST_CONDITIONS => "DB426_ALARMS_WARNINGS".CLADDING_HOPPERS."717485");
END_REGION

REGION Network 15: /////_HOPPER_3_SEQUENCES_/////
END_REGION

REGION Network 16: CALL FB22701 LOAD FEEDER SEQUENCE TIME UNIT 02 HOPPER 3
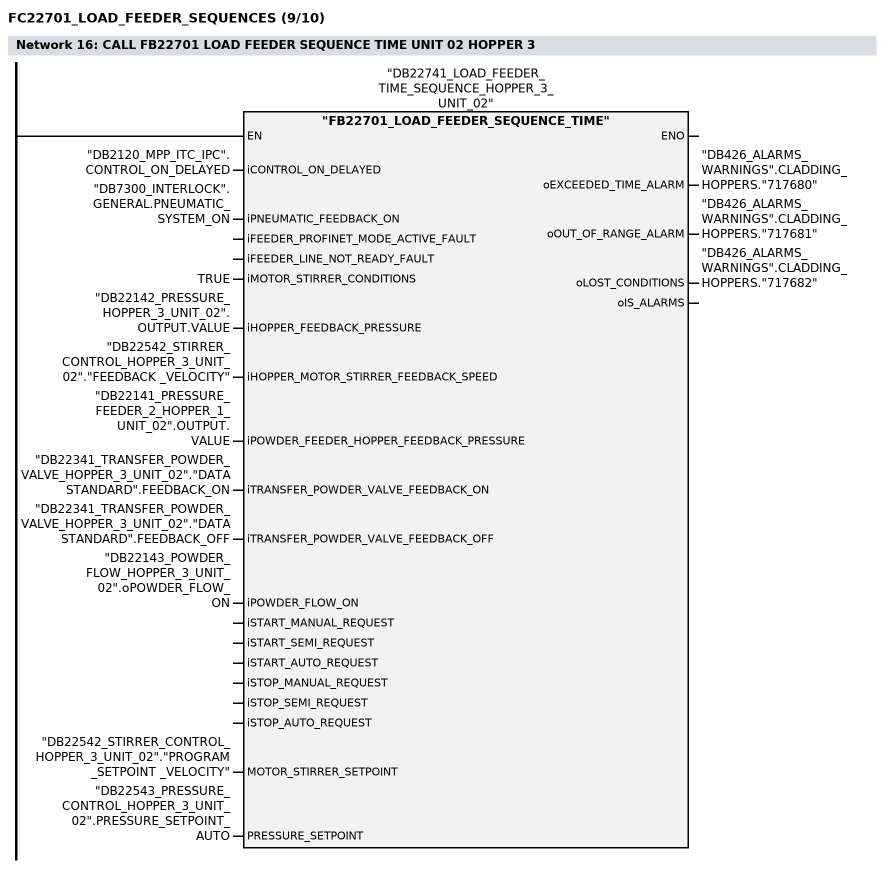
   RUNG wire#powerrail
      "DB22741_LOAD_FEEDER_TIME_SEQUENCE_HOPPER_3_UNIT_02"(iCONTROL_ON_DELAYED := "DB2120_MPP_ITC_IPC".CONTROL_ON_DELAYED, iPNEUMATIC_FEEDBACK_ON := "DB7300_INTERLOCK".GENERAL.PNEUMATIC_SYSTEM_ON, iFEEDER_PROFINET_MODE_ACTIVE_FAULT :=, iFEEDER_LINE_NOT_READY_FAULT :=, iMOTOR_STIRRER_CONDITIONS := TRUE, iHOPPER_FEEDBACK_PRESSURE := "DB22142_PRESSURE_HOPPER_3_UNIT_02".OUTPUT.VALUE, iHOPPER_MOTOR_STIRRER_FEEDBACK_SPEED := "DB22542_STIRRER_CONTROL_HOPPER_3_UNIT_02"."FEEDBACK _VELOCITY", iPOWDER_FEEDER_HOPPER_FEEDBACK_PRESSURE := "DB22141_PRESSURE_FEEDER_2_HOPPER_1_UNIT_02".OUTPUT.VALUE, iTRANSFER_POWDER_VALVE_FEEDBACK_ON := "DB22341_TRANSFER_POWDER_VALVE_HOPPER_3_UNIT_02"."DATA STANDARD".FEEDBACK_ON, iTRANSFER_POWDER_VALVE_FEEDBACK_OFF := "DB22341_TRANSFER_POWDER_VALVE_HOPPER_3_UNIT_02"."DATA STANDARD".FEEDBACK_OFF, iPOWDER_FLOW_ON := "DB22143_POWDER_FLOW_HOPPER_3_UNIT_02".oPOWDER_FLOW_ON, iSTART_MANUAL_REQUEST :=, iSTART_SEMI_REQUEST :=, iSTART_AUTO_REQUEST :=, iSTOP_MANUAL_REQUEST :=, iSTOP_SEMI_REQUEST :=, iSTOP_AUTO_REQUEST :=, MOTOR_STIRRER_SETPOINT := "DB22542_STIRRER_CONTROL_HOPPER_3_UNIT_02"."PROGRAM _SETPOINT _VELOCITY", PRESSURE_SETPOINT := "DB22543_PRESSURE_CONTROL_HOPPER_3_UNIT_02".PRESSURE_SETPOINT_AUTO, oEXCEEDED_TIME_ALARM => "DB426_ALARMS_WARNINGS".CLADDING_HOPPERS."717680", oOUT_OF_RANGE_ALARM => "DB426_ALARMS_WARNINGS".CLADDING_HOPPERS."717681", oLOST_CONDITIONS => "DB426_ALARMS_WARNINGS".CLADDING_HOPPERS."717682", oIS_ALARMS =>)
   END_RUNG
   // the same network as SCL:
   "DB22741_LOAD_FEEDER_TIME_SEQUENCE_HOPPER_3_UNIT_02"(iCONTROL_ON_DELAYED := "DB2120_MPP_ITC_IPC".CONTROL_ON_DELAYED,   // "FB22701_LOAD_FEEDER_SEQUENCE_TIME"
                           iPNEUMATIC_FEEDBACK_ON := "DB7300_INTERLOCK".GENERAL.PNEUMATIC_SYSTEM_ON,
                           iMOTOR_STIRRER_CONDITIONS := TRUE,
                           iHOPPER_FEEDBACK_PRESSURE := "DB22142_PRESSURE_HOPPER_3_UNIT_02".OUTPUT.VALUE,
                           iHOPPER_MOTOR_STIRRER_FEEDBACK_SPEED := "DB22542_STIRRER_CONTROL_HOPPER_3_UNIT_02"."FEEDBACK _VELOCITY",
                           iPOWDER_FEEDER_HOPPER_FEEDBACK_PRESSURE := "DB22141_PRESSURE_FEEDER_2_HOPPER_1_UNIT_02".OUTPUT.VALUE,
                           iTRANSFER_POWDER_VALVE_FEEDBACK_ON := "DB22341_TRANSFER_POWDER_VALVE_HOPPER_3_UNIT_02"."DATA STANDARD".FEEDBACK_ON,
                           iTRANSFER_POWDER_VALVE_FEEDBACK_OFF := "DB22341_TRANSFER_POWDER_VALVE_HOPPER_3_UNIT_02"."DATA STANDARD".FEEDBACK_OFF,
                           iPOWDER_FLOW_ON := "DB22143_POWDER_FLOW_HOPPER_3_UNIT_02".oPOWDER_FLOW_ON,
                           MOTOR_STIRRER_SETPOINT := "DB22542_STIRRER_CONTROL_HOPPER_3_UNIT_02"."PROGRAM _SETPOINT _VELOCITY",
                           PRESSURE_SETPOINT := "DB22543_PRESSURE_CONTROL_HOPPER_3_UNIT_02".PRESSURE_SETPOINT_AUTO,
                           oEXCEEDED_TIME_ALARM => "DB426_ALARMS_WARNINGS".CLADDING_HOPPERS."717680",
                           oOUT_OF_RANGE_ALARM => "DB426_ALARMS_WARNINGS".CLADDING_HOPPERS."717681",
                           oLOST_CONDITIONS => "DB426_ALARMS_WARNINGS".CLADDING_HOPPERS."717682");
END_REGION

REGION Network 17: CALL FB22702 LOAD FEEDER SEQUENCE WEIGHT UNIT 02 HOPPER 3
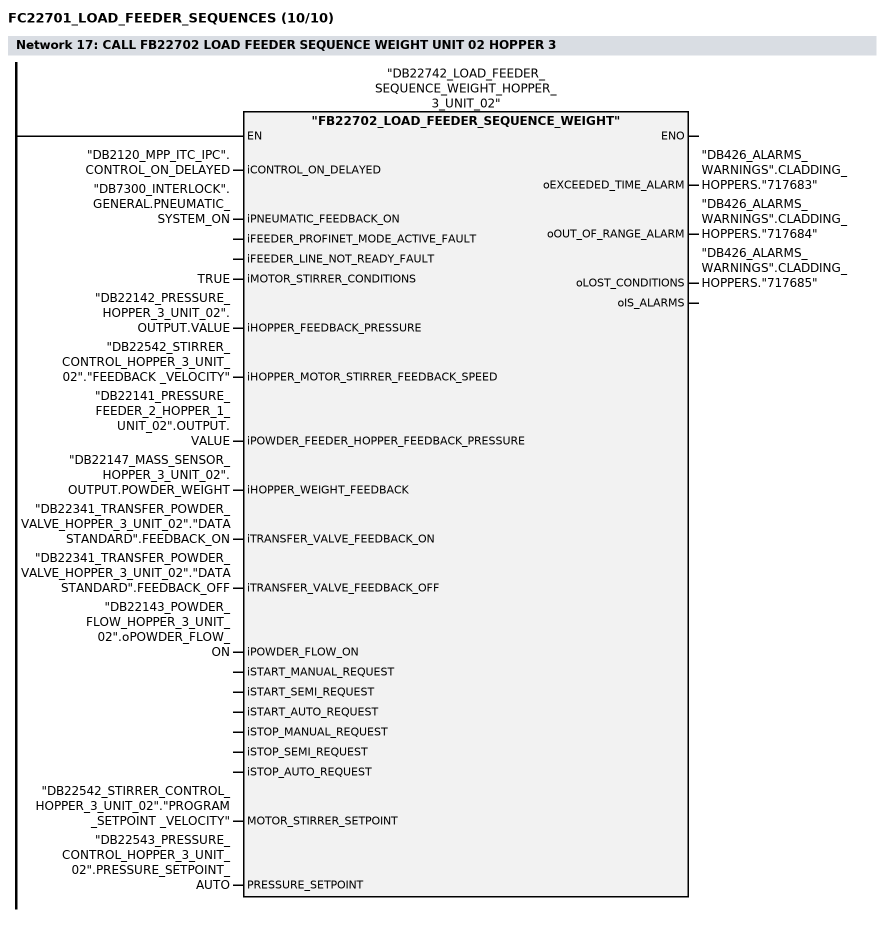
   RUNG wire#powerrail
      "DB22742_LOAD_FEEDER_SEQUENCE_WEIGHT_HOPPER_3_UNIT_02"(iCONTROL_ON_DELAYED := "DB2120_MPP_ITC_IPC".CONTROL_ON_DELAYED, iPNEUMATIC_FEEDBACK_ON := "DB7300_INTERLOCK".GENERAL.PNEUMATIC_SYSTEM_ON, iFEEDER_PROFINET_MODE_ACTIVE_FAULT :=, iFEEDER_LINE_NOT_READY_FAULT :=, iMOTOR_STIRRER_CONDITIONS := TRUE, iHOPPER_FEEDBACK_PRESSURE := "DB22142_PRESSURE_HOPPER_3_UNIT_02".OUTPUT.VALUE, iHOPPER_MOTOR_STIRRER_FEEDBACK_SPEED := "DB22542_STIRRER_CONTROL_HOPPER_3_UNIT_02"."FEEDBACK _VELOCITY", iPOWDER_FEEDER_HOPPER_FEEDBACK_PRESSURE := "DB22141_PRESSURE_FEEDER_2_HOPPER_1_UNIT_02".OUTPUT.VALUE, iHOPPER_WEIGHT_FEEDBACK := "DB22147_MASS_SENSOR_HOPPER_3_UNIT_02".OUTPUT.POWDER_WEIGHT, iTRANSFER_VALVE_FEEDBACK_ON := "DB22341_TRANSFER_POWDER_VALVE_HOPPER_3_UNIT_02"."DATA STANDARD".FEEDBACK_ON, iTRANSFER_VALVE_FEEDBACK_OFF := "DB22341_TRANSFER_POWDER_VALVE_HOPPER_3_UNIT_02"."DATA STANDARD".FEEDBACK_OFF, iPOWDER_FLOW_ON := "DB22143_POWDER_FLOW_HOPPER_3_UNIT_02".oPOWDER_FLOW_ON, iSTART_MANUAL_REQUEST :=, iSTART_SEMI_REQUEST :=, iSTART_AUTO_REQUEST :=, iSTOP_MANUAL_REQUEST :=, iSTOP_SEMI_REQUEST :=, iSTOP_AUTO_REQUEST :=, MOTOR_STIRRER_SETPOINT := "DB22542_STIRRER_CONTROL_HOPPER_3_UNIT_02"."PROGRAM _SETPOINT _VELOCITY", PRESSURE_SETPOINT := "DB22543_PRESSURE_CONTROL_HOPPER_3_UNIT_02".PRESSURE_SETPOINT_AUTO, oEXCEEDED_TIME_ALARM => "DB426_ALARMS_WARNINGS".CLADDING_HOPPERS."717683", oOUT_OF_RANGE_ALARM => "DB426_ALARMS_WARNINGS".CLADDING_HOPPERS."717684", oLOST_CONDITIONS => "DB426_ALARMS_WARNINGS".CLADDING_HOPPERS."717685", oIS_ALARMS =>)
   END_RUNG
   // the same network as SCL:
   "DB22742_LOAD_FEEDER_SEQUENCE_WEIGHT_HOPPER_3_UNIT_02"(iCONTROL_ON_DELAYED := "DB2120_MPP_ITC_IPC".CONTROL_ON_DELAYED,   // "FB22702_LOAD_FEEDER_SEQUENCE_WEIGHT"
                           iPNEUMATIC_FEEDBACK_ON := "DB7300_INTERLOCK".GENERAL.PNEUMATIC_SYSTEM_ON,
                           iMOTOR_STIRRER_CONDITIONS := TRUE,
                           iHOPPER_FEEDBACK_PRESSURE := "DB22142_PRESSURE_HOPPER_3_UNIT_02".OUTPUT.VALUE,
                           iHOPPER_MOTOR_STIRRER_FEEDBACK_SPEED := "DB22542_STIRRER_CONTROL_HOPPER_3_UNIT_02"."FEEDBACK _VELOCITY",
                           iPOWDER_FEEDER_HOPPER_FEEDBACK_PRESSURE := "DB22141_PRESSURE_FEEDER_2_HOPPER_1_UNIT_02".OUTPUT.VALUE,
                           iHOPPER_WEIGHT_FEEDBACK := "DB22147_MASS_SENSOR_HOPPER_3_UNIT_02".OUTPUT.POWDER_WEIGHT,
                           iTRANSFER_VALVE_FEEDBACK_ON := "DB22341_TRANSFER_POWDER_VALVE_HOPPER_3_UNIT_02"."DATA STANDARD".FEEDBACK_ON,
                           iTRANSFER_VALVE_FEEDBACK_OFF := "DB22341_TRANSFER_POWDER_VALVE_HOPPER_3_UNIT_02"."DATA STANDARD".FEEDBACK_OFF,
                           iPOWDER_FLOW_ON := "DB22143_POWDER_FLOW_HOPPER_3_UNIT_02".oPOWDER_FLOW_ON,
                           MOTOR_STIRRER_SETPOINT := "DB22542_STIRRER_CONTROL_HOPPER_3_UNIT_02"."PROGRAM _SETPOINT _VELOCITY",
                           PRESSURE_SETPOINT := "DB22543_PRESSURE_CONTROL_HOPPER_3_UNIT_02".PRESSURE_SETPOINT_AUTO,
                           oEXCEEDED_TIME_ALARM => "DB426_ALARMS_WARNINGS".CLADDING_HOPPERS."717683",
                           oOUT_OF_RANGE_ALARM => "DB426_ALARMS_WARNINGS".CLADDING_HOPPERS."717684",
                           oLOST_CONDITIONS => "DB426_ALARMS_WARNINGS".CLADDING_HOPPERS."717685");
END_REGION
END_FUNCTION

FUNCTION "FC2100_GENERAL" : Void   // FC2100, LAD
{ S7_Optimized_Access := 'FALSE' }
AUTHOR : ETXETAR
VERSION : 1.0
// stored: AutoNumber false, IsIECCheckEnabled false, SetENOAutomatically false, UDAEnableTagReadback false
   VAR CONSTANT
      FC_NUMBER : DInt := 2100;   // FC NUMBER
   END_VAR
BEGIN

REGION Network 1: ALWAYS OFF
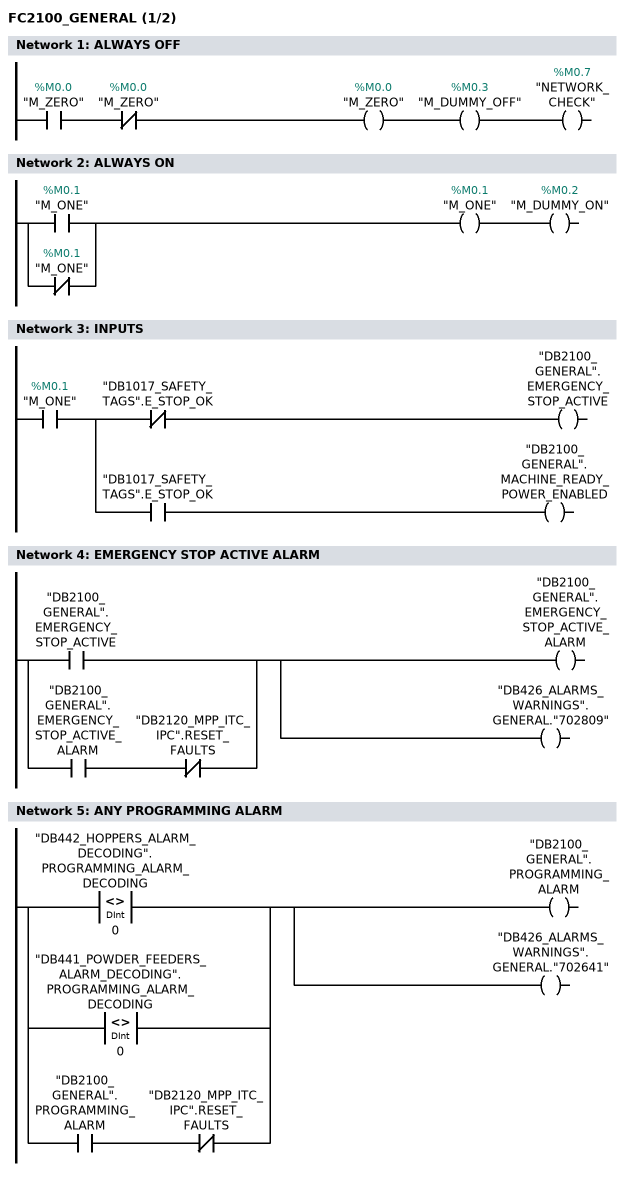
   RUNG wire#powerrail
      Contact( "M_ZERO" )
      I_Contact( "M_ZERO" )
      Coil( "M_ZERO" )
      Coil( "M_DUMMY_OFF" )
      Coil( "NETWORK_CHECK" )
   END_RUNG
   // the same network as SCL:
   "M_ZERO" := "M_ZERO" AND NOT "M_ZERO";
   "M_DUMMY_OFF" := "M_ZERO";
   "NETWORK_CHECK" := "M_ZERO";
END_REGION

REGION Network 2: ALWAYS ON
   RUNG wire#powerrail
      Contact( "M_ONE" )
      wire#w1
      Coil( "M_ONE" )
      Coil( "M_DUMMY_ON" )
   END_RUNG
   RUNG wire#powerrail
      I_Contact( "M_ONE" )
   END_RUNG wire#w1
   // the same network as SCL:
   "M_ONE" := "M_ONE" OR NOT "M_ONE";
   "M_DUMMY_ON" := "M_ONE";
END_REGION

REGION Network 3: INPUTS
   RUNG wire#powerrail
      Contact( "M_ONE" )
      wire#w1
      I_Contact( "DB1017_SAFETY_TAGS".E_STOP_OK )
      Coil( "DB2100_GENERAL".EMERGENCY_STOP_ACTIVE )
   END_RUNG
   RUNG wire#w1
      Contact( "DB1017_SAFETY_TAGS".E_STOP_OK )
      Coil( "DB2100_GENERAL".MACHINE_READY_POWER_ENABLED )
   END_RUNG
   // the same network as SCL:
   "DB2100_GENERAL".EMERGENCY_STOP_ACTIVE := "M_ONE" AND NOT "DB1017_SAFETY_TAGS".E_STOP_OK;
   "DB2100_GENERAL".MACHINE_READY_POWER_ENABLED := "M_ONE" AND "DB1017_SAFETY_TAGS".E_STOP_OK;
END_REGION

REGION Network 4: EMERGENCY STOP ACTIVE ALARM
   RUNG wire#powerrail
      Contact( "DB2100_GENERAL".EMERGENCY_STOP_ACTIVE )
      wire#w1
      Coil( "DB2100_GENERAL".EMERGENCY_STOP_ACTIVE_ALARM )
   END_RUNG
   RUNG wire#powerrail
      Contact( "DB2100_GENERAL".EMERGENCY_STOP_ACTIVE_ALARM )
      I_Contact( "DB2120_MPP_ITC_IPC".RESET_FAULTS )
   END_RUNG wire#w1
   RUNG wire#w1
      Coil( "DB426_ALARMS_WARNINGS".GENERAL."702809" )
   END_RUNG
   // the same network as SCL:
   "DB2100_GENERAL".EMERGENCY_STOP_ACTIVE_ALARM := "DB2100_GENERAL".EMERGENCY_STOP_ACTIVE OR ("DB2100_GENERAL".EMERGENCY_STOP_ACTIVE_ALARM AND NOT "DB2120_MPP_ITC_IPC".RESET_FAULTS);
   "DB426_ALARMS_WARNINGS".GENERAL."702809" := "DB2100_GENERAL".EMERGENCY_STOP_ACTIVE_ALARM;
END_REGION

REGION Network 5: ANY PROGRAMMING ALARM
   RUNG wire#powerrail
      { S7_Templates := "SrcType := DInt" } NE_Contact(in1 := "DB442_HOPPERS_ALARM_DECODING".PROGRAMMING_ALARM_DECODING, in2 := 0)
      wire#w1
      Coil( "DB2100_GENERAL".PROGRAMMING_ALARM )
   END_RUNG
   RUNG wire#powerrail
      { S7_Templates := "SrcType := DInt" } NE_Contact(in1 := "DB441_POWDER_FEEDERS_ALARM_DECODING".PROGRAMMING_ALARM_DECODING, in2 := 0)
   END_RUNG wire#w1
   RUNG wire#powerrail
      Contact( "DB2100_GENERAL".PROGRAMMING_ALARM )
      I_Contact( "DB2120_MPP_ITC_IPC".RESET_FAULTS )
   END_RUNG wire#w1
   RUNG wire#w1
      Coil( "DB426_ALARMS_WARNINGS".GENERAL."702641" )
   END_RUNG
   // the same network as SCL:
   "DB2100_GENERAL".PROGRAMMING_ALARM := ("DB442_HOPPERS_ALARM_DECODING".PROGRAMMING_ALARM_DECODING <> 0) OR ("DB441_POWDER_FEEDERS_ALARM_DECODING".PROGRAMMING_ALARM_DECODING <> 0) OR ("DB2100_GENERAL".PROGRAMMING_ALARM AND NOT "DB2120_MPP_ITC_IPC".RESET_FAULTS);
   "DB426_ALARMS_WARNINGS".GENERAL."702641" := "DB2100_GENERAL".PROGRAMMING_ALARM;
END_REGION

REGION Network 6: CHECK NETWORK LOGIC ALARM
   // CHECK EVERY NETWORK LOGIC WHERE THE M0.7 IS PROGRAMMED, THOSE NETWORK MUST BE ADAPTED ACCORDING TO THE MACHINE STRUCTURE
   // 
   // DELETE THIS NETWORK
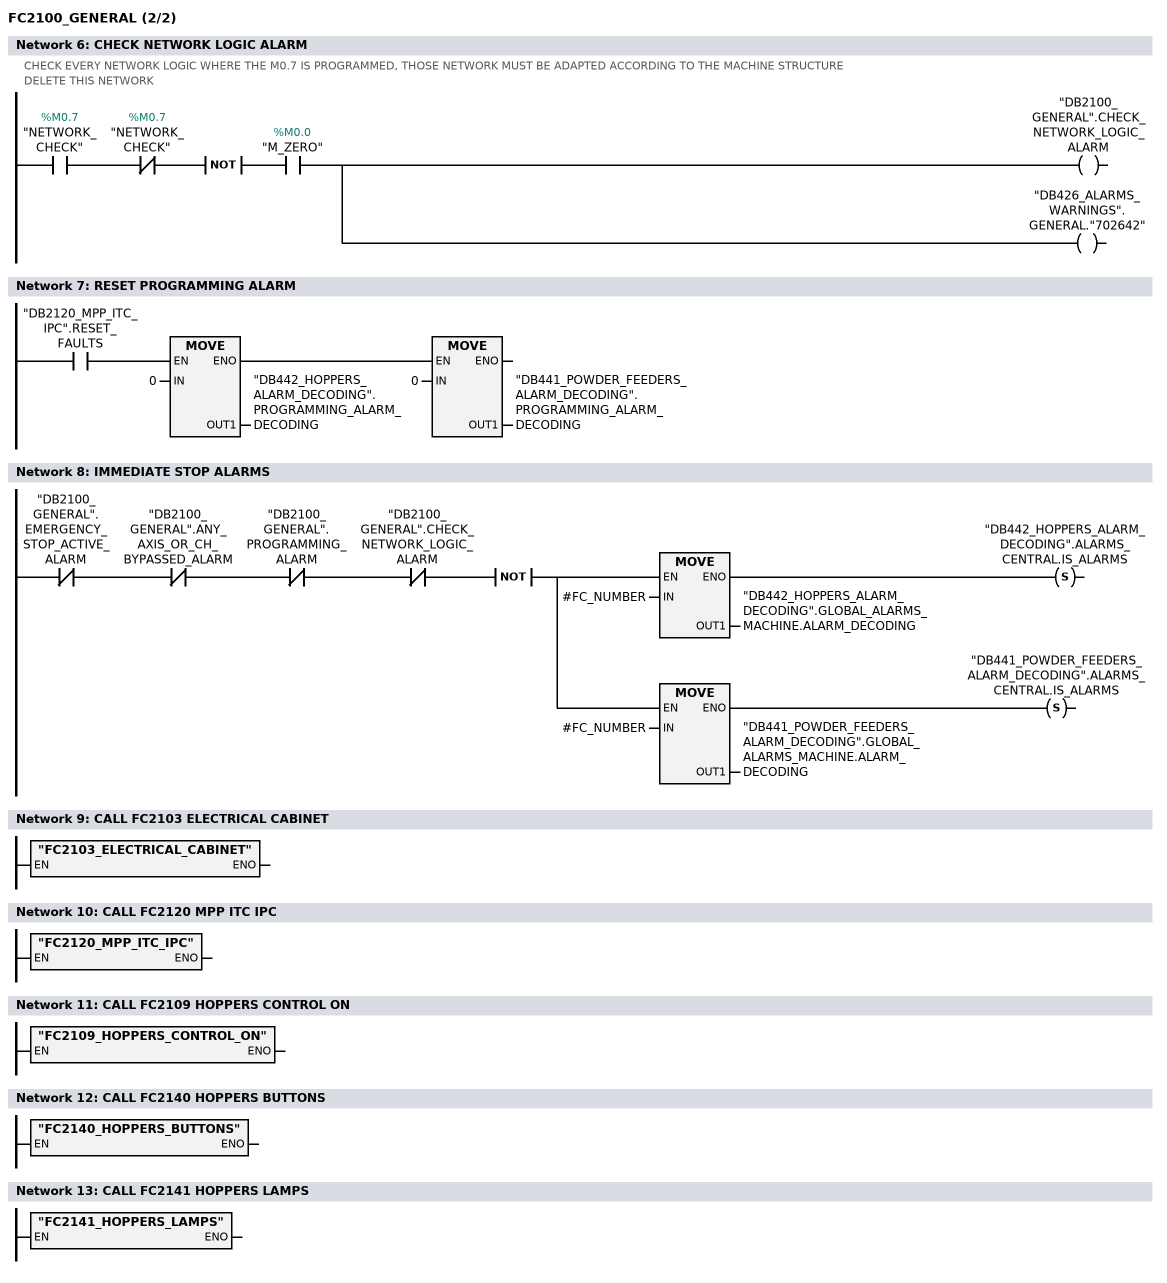
   RUNG wire#powerrail
      Contact( "NETWORK_CHECK" )
      I_Contact( "NETWORK_CHECK" )
      Not()
      Contact( "M_ZERO" )
      wire#w1
      Coil( "DB2100_GENERAL".CHECK_NETWORK_LOGIC_ALARM )
   END_RUNG
   RUNG wire#w1
      Coil( "DB426_ALARMS_WARNINGS".GENERAL."702642" )
   END_RUNG
   // the same network as SCL:
   "DB2100_GENERAL".CHECK_NETWORK_LOGIC_ALARM := NOT ("NETWORK_CHECK" AND NOT "NETWORK_CHECK") AND "M_ZERO";
   "DB426_ALARMS_WARNINGS".GENERAL."702642" := "DB2100_GENERAL".CHECK_NETWORK_LOGIC_ALARM;
END_REGION

REGION Network 7: RESET PROGRAMMING ALARM
   RUNG wire#powerrail
      Contact( "DB2120_MPP_ITC_IPC".RESET_FAULTS )
      { S7_GenerateENO := "TRUE" } Move(in := 0, out1 => "DB442_HOPPERS_ALARM_DECODING".PROGRAMMING_ALARM_DECODING)
      { S7_GenerateENO := "TRUE" } Move(in := 0, out1 => "DB441_POWDER_FEEDERS_ALARM_DECODING".PROGRAMMING_ALARM_DECODING)
   END_RUNG
   // the same network as SCL:
   // ENO of a box is taken as its EN; it also drops when the box reports an error
   IF "DB2120_MPP_ITC_IPC".RESET_FAULTS THEN
       "DB442_HOPPERS_ALARM_DECODING".PROGRAMMING_ALARM_DECODING := 0;
       "DB441_POWDER_FEEDERS_ALARM_DECODING".PROGRAMMING_ALARM_DECODING := 0;
   END_IF;
END_REGION

REGION Network 8: IMMEDIATE STOP ALARMS
   RUNG wire#powerrail
      I_Contact( "DB2100_GENERAL".EMERGENCY_STOP_ACTIVE_ALARM )
      I_Contact( "DB2100_GENERAL".ANY_AXIS_OR_CH_BYPASSED_ALARM )
      I_Contact( "DB2100_GENERAL".PROGRAMMING_ALARM )
      I_Contact( "DB2100_GENERAL".CHECK_NETWORK_LOGIC_ALARM )
      Not()
      wire#w1
      { S7_GenerateENO := "TRUE" } Move(in := #FC_NUMBER, out1 => "DB442_HOPPERS_ALARM_DECODING".GLOBAL_ALARMS_MACHINE.ALARM_DECODING)
      S_Coil( "DB442_HOPPERS_ALARM_DECODING".ALARMS_CENTRAL.IS_ALARMS )
   END_RUNG
   RUNG wire#w1
      { S7_GenerateENO := "TRUE" } Move(in := #FC_NUMBER, out1 => "DB441_POWDER_FEEDERS_ALARM_DECODING".GLOBAL_ALARMS_MACHINE.ALARM_DECODING)
      S_Coil( "DB441_POWDER_FEEDERS_ALARM_DECODING".ALARMS_CENTRAL.IS_ALARMS )
   END_RUNG
   // the same network as SCL:
   // ENO of a box is taken as its EN; it also drops when the box reports an error
   IF NOT (NOT "DB2100_GENERAL".EMERGENCY_STOP_ACTIVE_ALARM AND NOT "DB2100_GENERAL".ANY_AXIS_OR_CH_BYPASSED_ALARM AND NOT "DB2100_GENERAL".PROGRAMMING_ALARM AND NOT "DB2100_GENERAL".CHECK_NETWORK_LOGIC_ALARM) THEN
       "DB442_HOPPERS_ALARM_DECODING".GLOBAL_ALARMS_MACHINE.ALARM_DECODING := #FC_NUMBER;
       "DB442_HOPPERS_ALARM_DECODING".ALARMS_CENTRAL.IS_ALARMS := TRUE;
       "DB441_POWDER_FEEDERS_ALARM_DECODING".GLOBAL_ALARMS_MACHINE.ALARM_DECODING := #FC_NUMBER;
       "DB441_POWDER_FEEDERS_ALARM_DECODING".ALARMS_CENTRAL.IS_ALARMS := TRUE;
   END_IF;
END_REGION

REGION Network 9: CALL FC2103 ELECTRICAL CABINET
   RUNG wire#powerrail
      "FC2103_ELECTRICAL_CABINET"()
   END_RUNG
   // the same network as SCL:
   "FC2103_ELECTRICAL_CABINET"();
END_REGION

REGION Network 10: CALL FC2120 MPP ITC IPC
   RUNG wire#powerrail
      "FC2120_MPP_ITC_IPC"()
   END_RUNG
   // the same network as SCL:
   "FC2120_MPP_ITC_IPC"();
END_REGION

REGION Network 11: CALL FC2109 HOPPERS CONTROL ON
   RUNG wire#powerrail
      "FC2109_HOPPERS_CONTROL_ON"()
   END_RUNG
   // the same network as SCL:
   "FC2109_HOPPERS_CONTROL_ON"();
END_REGION

REGION Network 12: CALL FC2140 HOPPERS BUTTONS
   RUNG wire#powerrail
      "FC2140_HOPPERS_BUTTONS"()
   END_RUNG
   // the same network as SCL:
   "FC2140_HOPPERS_BUTTONS"();
END_REGION

REGION Network 13: CALL FC2141 HOPPERS LAMPS
   RUNG wire#powerrail
      "FC2141_HOPPERS_LAMPS"()
   END_RUNG
   // the same network as SCL:
   "FC2141_HOPPERS_LAMPS"();
END_REGION
END_FUNCTION

FUNCTION "FC2103_ELECTRICAL_CABINET" : Void   // FC2103, LAD
{ S7_Optimized_Access := 'FALSE' }
AUTHOR : ETXETAR
VERSION : 1.0
// stored: AutoNumber false, IsIECCheckEnabled false, SetENOAutomatically false, UDAEnableTagReadback false
   VAR CONSTANT
      FC_NUMBER : DInt := 2103;
   END_VAR
   VAR_TEMP   // added for the SCL form of the ladder/FBD networks
      _w1 : Bool;
   END_VAR
BEGIN

REGION Network 1: INPUTS
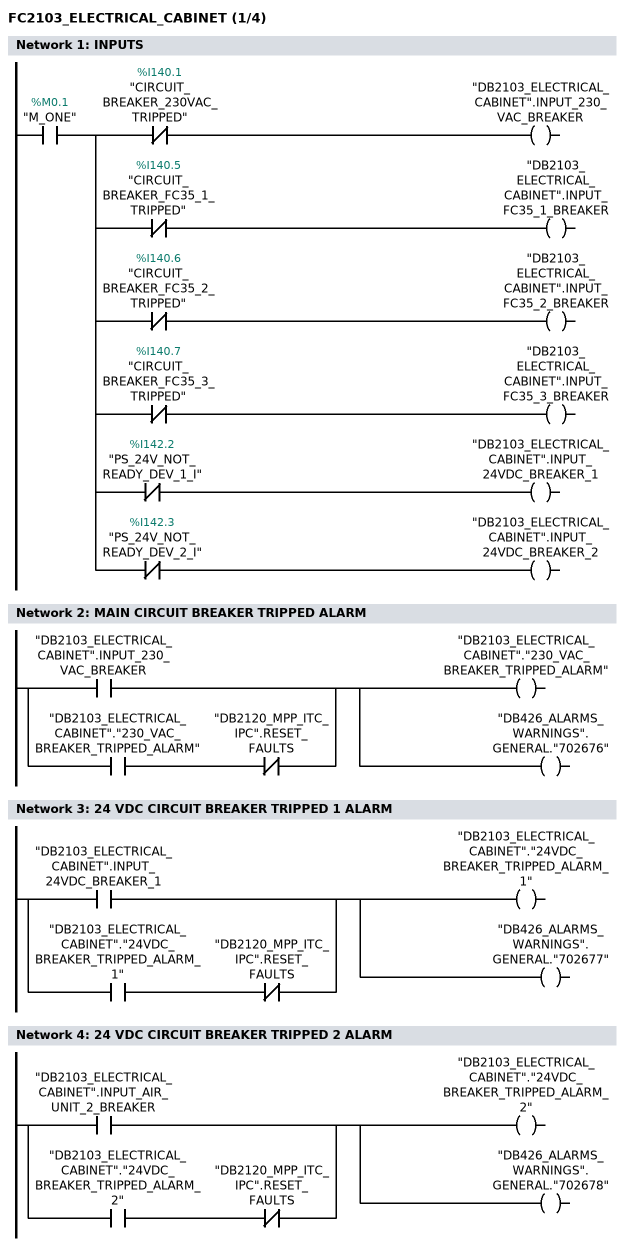
   RUNG wire#powerrail
      Contact( "M_ONE" )
      wire#w1
      I_Contact( "CIRCUIT_BREAKER_230VAC_TRIPPED" )
      Coil( "DB2103_ELECTRICAL_CABINET".INPUT_230_VAC_BREAKER )
   END_RUNG
   RUNG wire#w1
      I_Contact( "CIRCUIT_BREAKER_FC35_1_TRIPPED" )
      Coil( "DB2103_ELECTRICAL_CABINET".INPUT_FC35_1_BREAKER )
   END_RUNG
   RUNG wire#w1
      I_Contact( "CIRCUIT_BREAKER_FC35_2_TRIPPED" )
      Coil( "DB2103_ELECTRICAL_CABINET".INPUT_FC35_2_BREAKER )
   END_RUNG
   RUNG wire#w1
      I_Contact( "CIRCUIT_BREAKER_FC35_3_TRIPPED" )
      Coil( "DB2103_ELECTRICAL_CABINET".INPUT_FC35_3_BREAKER )
   END_RUNG
   RUNG wire#w1
      I_Contact( "PS_24V_NOT_READY_DEV_1_I" )
      Coil( "DB2103_ELECTRICAL_CABINET".INPUT_24VDC_BREAKER_1 )
   END_RUNG
   RUNG wire#w1
      I_Contact( "PS_24V_NOT_READY_DEV_2_I" )
      Coil( "DB2103_ELECTRICAL_CABINET".INPUT_24VDC_BREAKER_2 )
   END_RUNG
   // the same network as SCL:
   "DB2103_ELECTRICAL_CABINET".INPUT_230_VAC_BREAKER := "M_ONE" AND NOT "CIRCUIT_BREAKER_230VAC_TRIPPED";
   "DB2103_ELECTRICAL_CABINET".INPUT_FC35_1_BREAKER := "M_ONE" AND NOT "CIRCUIT_BREAKER_FC35_1_TRIPPED";
   "DB2103_ELECTRICAL_CABINET".INPUT_FC35_2_BREAKER := "M_ONE" AND NOT "CIRCUIT_BREAKER_FC35_2_TRIPPED";
   "DB2103_ELECTRICAL_CABINET".INPUT_FC35_3_BREAKER := "M_ONE" AND NOT "CIRCUIT_BREAKER_FC35_3_TRIPPED";
   "DB2103_ELECTRICAL_CABINET".INPUT_24VDC_BREAKER_1 := "M_ONE" AND NOT "PS_24V_NOT_READY_DEV_1_I";
   "DB2103_ELECTRICAL_CABINET".INPUT_24VDC_BREAKER_2 := "M_ONE" AND NOT "PS_24V_NOT_READY_DEV_2_I";
END_REGION

REGION Network 2: MAIN CIRCUIT BREAKER TRIPPED ALARM
   RUNG wire#powerrail
      Contact( "DB2103_ELECTRICAL_CABINET".INPUT_230_VAC_BREAKER )
      wire#w1
      Coil( "DB2103_ELECTRICAL_CABINET"."230_VAC_BREAKER_TRIPPED_ALARM" )
   END_RUNG
   RUNG wire#powerrail
      Contact( "DB2103_ELECTRICAL_CABINET"."230_VAC_BREAKER_TRIPPED_ALARM" )
      I_Contact( "DB2120_MPP_ITC_IPC".RESET_FAULTS )
   END_RUNG wire#w1
   RUNG wire#w1
      Coil( "DB426_ALARMS_WARNINGS".GENERAL."702676" )
   END_RUNG
   // the same network as SCL:
   "DB2103_ELECTRICAL_CABINET"."230_VAC_BREAKER_TRIPPED_ALARM" := "DB2103_ELECTRICAL_CABINET".INPUT_230_VAC_BREAKER OR ("DB2103_ELECTRICAL_CABINET"."230_VAC_BREAKER_TRIPPED_ALARM" AND NOT "DB2120_MPP_ITC_IPC".RESET_FAULTS);
   "DB426_ALARMS_WARNINGS".GENERAL."702676" := "DB2103_ELECTRICAL_CABINET"."230_VAC_BREAKER_TRIPPED_ALARM";
END_REGION

REGION Network 3: 24 VDC CIRCUIT BREAKER TRIPPED 1 ALARM
   RUNG wire#powerrail
      Contact( "DB2103_ELECTRICAL_CABINET".INPUT_24VDC_BREAKER_1 )
      wire#w1
      Coil( "DB2103_ELECTRICAL_CABINET"."24VDC_BREAKER_TRIPPED_ALARM_1" )
   END_RUNG
   RUNG wire#powerrail
      Contact( "DB2103_ELECTRICAL_CABINET"."24VDC_BREAKER_TRIPPED_ALARM_1" )
      I_Contact( "DB2120_MPP_ITC_IPC".RESET_FAULTS )
   END_RUNG wire#w1
   RUNG wire#w1
      Coil( "DB426_ALARMS_WARNINGS".GENERAL."702677" )
   END_RUNG
   // the same network as SCL:
   "DB2103_ELECTRICAL_CABINET"."24VDC_BREAKER_TRIPPED_ALARM_1" := "DB2103_ELECTRICAL_CABINET".INPUT_24VDC_BREAKER_1 OR ("DB2103_ELECTRICAL_CABINET"."24VDC_BREAKER_TRIPPED_ALARM_1" AND NOT "DB2120_MPP_ITC_IPC".RESET_FAULTS);
   "DB426_ALARMS_WARNINGS".GENERAL."702677" := "DB2103_ELECTRICAL_CABINET"."24VDC_BREAKER_TRIPPED_ALARM_1";
END_REGION

REGION Network 4: 24 VDC CIRCUIT BREAKER TRIPPED 2 ALARM
   RUNG wire#powerrail
      Contact( "DB2103_ELECTRICAL_CABINET".INPUT_AIR_UNIT_2_BREAKER )
      wire#w1
      Coil( "DB2103_ELECTRICAL_CABINET"."24VDC_BREAKER_TRIPPED_ALARM_2" )
   END_RUNG
   RUNG wire#powerrail
      Contact( "DB2103_ELECTRICAL_CABINET"."24VDC_BREAKER_TRIPPED_ALARM_2" )
      I_Contact( "DB2120_MPP_ITC_IPC".RESET_FAULTS )
   END_RUNG wire#w1
   RUNG wire#w1
      Coil( "DB426_ALARMS_WARNINGS".GENERAL."702678" )
   END_RUNG
   // the same network as SCL:
   "DB2103_ELECTRICAL_CABINET"."24VDC_BREAKER_TRIPPED_ALARM_2" := "DB2103_ELECTRICAL_CABINET".INPUT_AIR_UNIT_2_BREAKER OR ("DB2103_ELECTRICAL_CABINET"."24VDC_BREAKER_TRIPPED_ALARM_2" AND NOT "DB2120_MPP_ITC_IPC".RESET_FAULTS);
   "DB426_ALARMS_WARNINGS".GENERAL."702678" := "DB2103_ELECTRICAL_CABINET"."24VDC_BREAKER_TRIPPED_ALARM_2";
END_REGION

REGION Network 5: FC35_1 CIRCUIT BREAKER TRIPPED ALARM
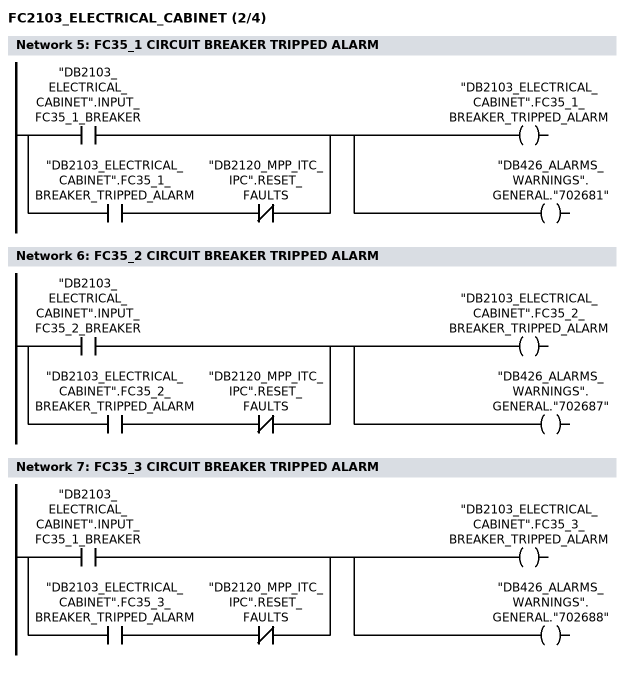
   RUNG wire#powerrail
      Contact( "DB2103_ELECTRICAL_CABINET".INPUT_FC35_1_BREAKER )
      wire#w1
      Coil( "DB2103_ELECTRICAL_CABINET".FC35_1_BREAKER_TRIPPED_ALARM )
   END_RUNG
   RUNG wire#powerrail
      Contact( "DB2103_ELECTRICAL_CABINET".FC35_1_BREAKER_TRIPPED_ALARM )
      I_Contact( "DB2120_MPP_ITC_IPC".RESET_FAULTS )
   END_RUNG wire#w1
   RUNG wire#w1
      Coil( "DB426_ALARMS_WARNINGS".GENERAL."702681" )
   END_RUNG
   // the same network as SCL:
   "DB2103_ELECTRICAL_CABINET".FC35_1_BREAKER_TRIPPED_ALARM := "DB2103_ELECTRICAL_CABINET".INPUT_FC35_1_BREAKER OR ("DB2103_ELECTRICAL_CABINET".FC35_1_BREAKER_TRIPPED_ALARM AND NOT "DB2120_MPP_ITC_IPC".RESET_FAULTS);
   "DB426_ALARMS_WARNINGS".GENERAL."702681" := "DB2103_ELECTRICAL_CABINET".FC35_1_BREAKER_TRIPPED_ALARM;
END_REGION

REGION Network 6: FC35_2 CIRCUIT BREAKER TRIPPED ALARM
   RUNG wire#powerrail
      Contact( "DB2103_ELECTRICAL_CABINET".INPUT_FC35_2_BREAKER )
      wire#w1
      Coil( "DB2103_ELECTRICAL_CABINET".FC35_2_BREAKER_TRIPPED_ALARM )
   END_RUNG
   RUNG wire#powerrail
      Contact( "DB2103_ELECTRICAL_CABINET".FC35_2_BREAKER_TRIPPED_ALARM )
      I_Contact( "DB2120_MPP_ITC_IPC".RESET_FAULTS )
   END_RUNG wire#w1
   RUNG wire#w1
      Coil( "DB426_ALARMS_WARNINGS".GENERAL."702687" )
   END_RUNG
   // the same network as SCL:
   "DB2103_ELECTRICAL_CABINET".FC35_2_BREAKER_TRIPPED_ALARM := "DB2103_ELECTRICAL_CABINET".INPUT_FC35_2_BREAKER OR ("DB2103_ELECTRICAL_CABINET".FC35_2_BREAKER_TRIPPED_ALARM AND NOT "DB2120_MPP_ITC_IPC".RESET_FAULTS);
   "DB426_ALARMS_WARNINGS".GENERAL."702687" := "DB2103_ELECTRICAL_CABINET".FC35_2_BREAKER_TRIPPED_ALARM;
END_REGION

REGION Network 7: FC35_3 CIRCUIT BREAKER TRIPPED ALARM
   RUNG wire#powerrail
      Contact( "DB2103_ELECTRICAL_CABINET".INPUT_FC35_1_BREAKER )
      wire#w1
      Coil( "DB2103_ELECTRICAL_CABINET".FC35_3_BREAKER_TRIPPED_ALARM )
   END_RUNG
   RUNG wire#powerrail
      Contact( "DB2103_ELECTRICAL_CABINET".FC35_3_BREAKER_TRIPPED_ALARM )
      I_Contact( "DB2120_MPP_ITC_IPC".RESET_FAULTS )
   END_RUNG wire#w1
   RUNG wire#w1
      Coil( "DB426_ALARMS_WARNINGS".GENERAL."702688" )
   END_RUNG
   // the same network as SCL:
   "DB2103_ELECTRICAL_CABINET".FC35_3_BREAKER_TRIPPED_ALARM := "DB2103_ELECTRICAL_CABINET".INPUT_FC35_1_BREAKER OR ("DB2103_ELECTRICAL_CABINET".FC35_3_BREAKER_TRIPPED_ALARM AND NOT "DB2120_MPP_ITC_IPC".RESET_FAULTS);
   "DB426_ALARMS_WARNINGS".GENERAL."702688" := "DB2103_ELECTRICAL_CABINET".FC35_3_BREAKER_TRIPPED_ALARM;
END_REGION

REGION Network 8: IMMEDIATE STOP ALARMS
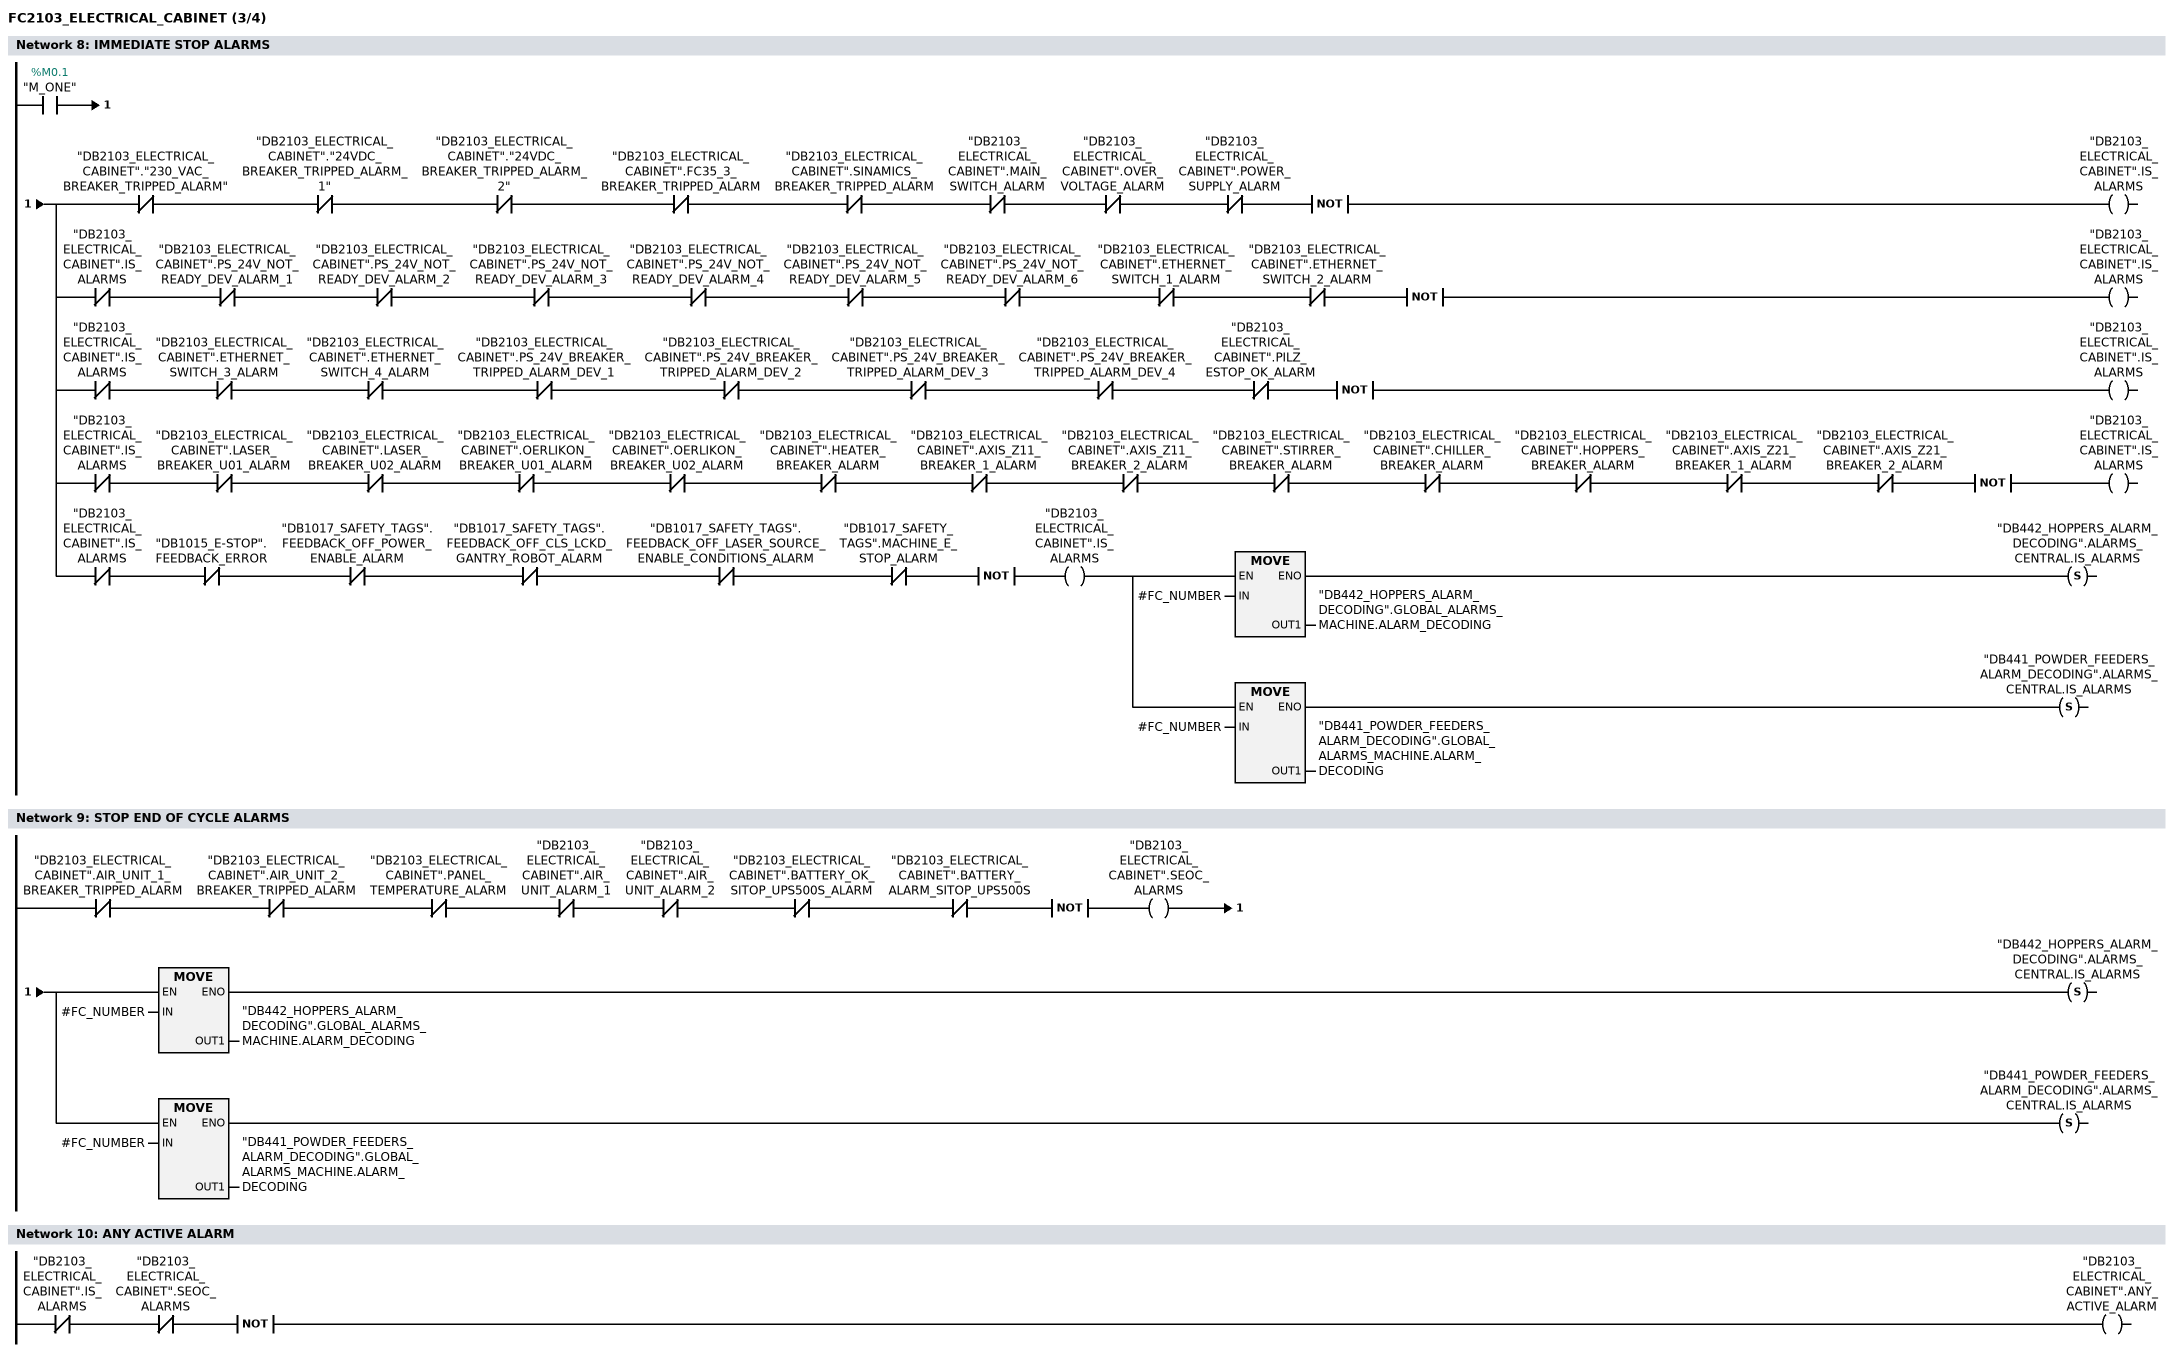
   RUNG wire#powerrail
      Contact( "M_ONE" )
      wire#w1
      I_Contact( "DB2103_ELECTRICAL_CABINET"."230_VAC_BREAKER_TRIPPED_ALARM" )
      I_Contact( "DB2103_ELECTRICAL_CABINET"."24VDC_BREAKER_TRIPPED_ALARM_1" )
      I_Contact( "DB2103_ELECTRICAL_CABINET"."24VDC_BREAKER_TRIPPED_ALARM_2" )
      I_Contact( "DB2103_ELECTRICAL_CABINET".FC35_3_BREAKER_TRIPPED_ALARM )
      I_Contact( "DB2103_ELECTRICAL_CABINET".SINAMICS_BREAKER_TRIPPED_ALARM )
      I_Contact( "DB2103_ELECTRICAL_CABINET".MAIN_SWITCH_ALARM )
      I_Contact( "DB2103_ELECTRICAL_CABINET".OVER_VOLTAGE_ALARM )
      I_Contact( "DB2103_ELECTRICAL_CABINET".POWER_SUPPLY_ALARM )
      Not()
      Coil( "DB2103_ELECTRICAL_CABINET".IS_ALARMS )
   END_RUNG
   RUNG wire#w1
      I_Contact( "DB2103_ELECTRICAL_CABINET".IS_ALARMS )
      I_Contact( "DB2103_ELECTRICAL_CABINET".PS_24V_NOT_READY_DEV_ALARM_1 )
      I_Contact( "DB2103_ELECTRICAL_CABINET".PS_24V_NOT_READY_DEV_ALARM_2 )
      I_Contact( "DB2103_ELECTRICAL_CABINET".PS_24V_NOT_READY_DEV_ALARM_3 )
      I_Contact( "DB2103_ELECTRICAL_CABINET".PS_24V_NOT_READY_DEV_ALARM_4 )
      I_Contact( "DB2103_ELECTRICAL_CABINET".PS_24V_NOT_READY_DEV_ALARM_5 )
      I_Contact( "DB2103_ELECTRICAL_CABINET".PS_24V_NOT_READY_DEV_ALARM_6 )
      I_Contact( "DB2103_ELECTRICAL_CABINET".ETHERNET_SWITCH_1_ALARM )
      I_Contact( "DB2103_ELECTRICAL_CABINET".ETHERNET_SWITCH_2_ALARM )
      Not()
      Coil( "DB2103_ELECTRICAL_CABINET".IS_ALARMS )
   END_RUNG
   RUNG wire#w1
      I_Contact( "DB2103_ELECTRICAL_CABINET".IS_ALARMS )
      I_Contact( "DB2103_ELECTRICAL_CABINET".ETHERNET_SWITCH_3_ALARM )
      I_Contact( "DB2103_ELECTRICAL_CABINET".ETHERNET_SWITCH_4_ALARM )
      I_Contact( "DB2103_ELECTRICAL_CABINET".PS_24V_BREAKER_TRIPPED_ALARM_DEV_1 )
      I_Contact( "DB2103_ELECTRICAL_CABINET".PS_24V_BREAKER_TRIPPED_ALARM_DEV_2 )
      I_Contact( "DB2103_ELECTRICAL_CABINET".PS_24V_BREAKER_TRIPPED_ALARM_DEV_3 )
      I_Contact( "DB2103_ELECTRICAL_CABINET".PS_24V_BREAKER_TRIPPED_ALARM_DEV_4 )
      I_Contact( "DB2103_ELECTRICAL_CABINET".PILZ_ESTOP_OK_ALARM )
      Not()
      Coil( "DB2103_ELECTRICAL_CABINET".IS_ALARMS )
   END_RUNG
   RUNG wire#w1
      I_Contact( "DB2103_ELECTRICAL_CABINET".IS_ALARMS )
      I_Contact( "DB2103_ELECTRICAL_CABINET".LASER_BREAKER_U01_ALARM )
      I_Contact( "DB2103_ELECTRICAL_CABINET".LASER_BREAKER_U02_ALARM )
      I_Contact( "DB2103_ELECTRICAL_CABINET".OERLIKON_BREAKER_U01_ALARM )
      I_Contact( "DB2103_ELECTRICAL_CABINET".OERLIKON_BREAKER_U02_ALARM )
      I_Contact( "DB2103_ELECTRICAL_CABINET".HEATER_BREAKER_ALARM )
      I_Contact( "DB2103_ELECTRICAL_CABINET".AXIS_Z11_BREAKER_1_ALARM )
      I_Contact( "DB2103_ELECTRICAL_CABINET".AXIS_Z11_BREAKER_2_ALARM )
      I_Contact( "DB2103_ELECTRICAL_CABINET".STIRRER_BREAKER_ALARM )
      I_Contact( "DB2103_ELECTRICAL_CABINET".CHILLER_BREAKER_ALARM )
      I_Contact( "DB2103_ELECTRICAL_CABINET".HOPPERS_BREAKER_ALARM )
      I_Contact( "DB2103_ELECTRICAL_CABINET".AXIS_Z21_BREAKER_1_ALARM )
      I_Contact( "DB2103_ELECTRICAL_CABINET".AXIS_Z21_BREAKER_2_ALARM )
      Not()
      Coil( "DB2103_ELECTRICAL_CABINET".IS_ALARMS )
   END_RUNG
   RUNG wire#w1
      I_Contact( "DB2103_ELECTRICAL_CABINET".IS_ALARMS )
      I_Contact( "DB1015_E-STOP".FEEDBACK_ERROR )
      I_Contact( "DB1017_SAFETY_TAGS".FEEDBACK_OFF_POWER_ENABLE_ALARM )
      I_Contact( "DB1017_SAFETY_TAGS".FEEDBACK_OFF_CLS_LCKD_GANTRY_ROBOT_ALARM )
      I_Contact( "DB1017_SAFETY_TAGS".FEEDBACK_OFF_LASER_SOURCE_ENABLE_CONDITIONS_ALARM )
      I_Contact( "DB1017_SAFETY_TAGS".MACHINE_E_STOP_ALARM )
      Not()
      Coil( "DB2103_ELECTRICAL_CABINET".IS_ALARMS )
      wire#w2
      { S7_GenerateENO := "TRUE" } Move(in := #FC_NUMBER, out1 => "DB442_HOPPERS_ALARM_DECODING".GLOBAL_ALARMS_MACHINE.ALARM_DECODING)
      S_Coil( "DB442_HOPPERS_ALARM_DECODING".ALARMS_CENTRAL.IS_ALARMS )
   END_RUNG
   RUNG wire#w2
      { S7_GenerateENO := "TRUE" } Move(in := #FC_NUMBER, out1 => "DB441_POWDER_FEEDERS_ALARM_DECODING".GLOBAL_ALARMS_MACHINE.ALARM_DECODING)
      S_Coil( "DB441_POWDER_FEEDERS_ALARM_DECODING".ALARMS_CENTRAL.IS_ALARMS )
   END_RUNG
   // the same network as SCL:
   // ENO of a box is taken as its EN; it also drops when the box reports an error
   "DB2103_ELECTRICAL_CABINET".IS_ALARMS := NOT ("M_ONE" AND NOT "DB2103_ELECTRICAL_CABINET"."230_VAC_BREAKER_TRIPPED_ALARM" AND NOT "DB2103_ELECTRICAL_CABINET"."24VDC_BREAKER_TRIPPED_ALARM_1" AND NOT "DB2103_ELECTRICAL_CABINET"."24VDC_BREAKER_TRIPPED_ALARM_2" AND NOT "DB2103_ELECTRICAL_CABINET".FC35_3_BREAKER_TRIPPED_ALARM AND NOT "DB2103_ELECTRICAL_CABINET".SINAMICS_BREAKER_TRIPPED_ALARM AND NOT "DB2103_ELECTRICAL_CABINET".MAIN_SWITCH_ALARM AND NOT "DB2103_ELECTRICAL_CABINET".OVER_VOLTAGE_ALARM AND NOT "DB2103_ELECTRICAL_CABINET".POWER_SUPPLY_ALARM);
   "DB2103_ELECTRICAL_CABINET".IS_ALARMS := NOT ("M_ONE" AND NOT "DB2103_ELECTRICAL_CABINET".IS_ALARMS AND NOT "DB2103_ELECTRICAL_CABINET".PS_24V_NOT_READY_DEV_ALARM_1 AND NOT "DB2103_ELECTRICAL_CABINET".PS_24V_NOT_READY_DEV_ALARM_2 AND NOT "DB2103_ELECTRICAL_CABINET".PS_24V_NOT_READY_DEV_ALARM_3 AND NOT "DB2103_ELECTRICAL_CABINET".PS_24V_NOT_READY_DEV_ALARM_4 AND NOT "DB2103_ELECTRICAL_CABINET".PS_24V_NOT_READY_DEV_ALARM_5 AND NOT "DB2103_ELECTRICAL_CABINET".PS_24V_NOT_READY_DEV_ALARM_6 AND NOT "DB2103_ELECTRICAL_CABINET".ETHERNET_SWITCH_1_ALARM AND NOT "DB2103_ELECTRICAL_CABINET".ETHERNET_SWITCH_2_ALARM);
   "DB2103_ELECTRICAL_CABINET".IS_ALARMS := NOT ("M_ONE" AND NOT "DB2103_ELECTRICAL_CABINET".IS_ALARMS AND NOT "DB2103_ELECTRICAL_CABINET".ETHERNET_SWITCH_3_ALARM AND NOT "DB2103_ELECTRICAL_CABINET".ETHERNET_SWITCH_4_ALARM AND NOT "DB2103_ELECTRICAL_CABINET".PS_24V_BREAKER_TRIPPED_ALARM_DEV_1 AND NOT "DB2103_ELECTRICAL_CABINET".PS_24V_BREAKER_TRIPPED_ALARM_DEV_2 AND NOT "DB2103_ELECTRICAL_CABINET".PS_24V_BREAKER_TRIPPED_ALARM_DEV_3 AND NOT "DB2103_ELECTRICAL_CABINET".PS_24V_BREAKER_TRIPPED_ALARM_DEV_4 AND NOT "DB2103_ELECTRICAL_CABINET".PILZ_ESTOP_OK_ALARM);
   "DB2103_ELECTRICAL_CABINET".IS_ALARMS := NOT ("M_ONE" AND NOT "DB2103_ELECTRICAL_CABINET".IS_ALARMS AND NOT "DB2103_ELECTRICAL_CABINET".LASER_BREAKER_U01_ALARM AND NOT "DB2103_ELECTRICAL_CABINET".LASER_BREAKER_U02_ALARM AND NOT "DB2103_ELECTRICAL_CABINET".OERLIKON_BREAKER_U01_ALARM AND NOT "DB2103_ELECTRICAL_CABINET".OERLIKON_BREAKER_U02_ALARM AND NOT "DB2103_ELECTRICAL_CABINET".HEATER_BREAKER_ALARM AND NOT "DB2103_ELECTRICAL_CABINET".AXIS_Z11_BREAKER_1_ALARM AND NOT "DB2103_ELECTRICAL_CABINET".AXIS_Z11_BREAKER_2_ALARM AND NOT "DB2103_ELECTRICAL_CABINET".STIRRER_BREAKER_ALARM AND NOT "DB2103_ELECTRICAL_CABINET".CHILLER_BREAKER_ALARM AND NOT "DB2103_ELECTRICAL_CABINET".HOPPERS_BREAKER_ALARM AND NOT "DB2103_ELECTRICAL_CABINET".AXIS_Z21_BREAKER_1_ALARM AND NOT "DB2103_ELECTRICAL_CABINET".AXIS_Z21_BREAKER_2_ALARM);
   "DB2103_ELECTRICAL_CABINET".IS_ALARMS := NOT ("M_ONE" AND NOT "DB2103_ELECTRICAL_CABINET".IS_ALARMS AND NOT "DB1015_E-STOP".FEEDBACK_ERROR AND NOT "DB1017_SAFETY_TAGS".FEEDBACK_OFF_POWER_ENABLE_ALARM AND NOT "DB1017_SAFETY_TAGS".FEEDBACK_OFF_CLS_LCKD_GANTRY_ROBOT_ALARM AND NOT "DB1017_SAFETY_TAGS".FEEDBACK_OFF_LASER_SOURCE_ENABLE_CONDITIONS_ALARM AND NOT "DB1017_SAFETY_TAGS".MACHINE_E_STOP_ALARM);
   IF "DB2103_ELECTRICAL_CABINET".IS_ALARMS THEN
       "DB442_HOPPERS_ALARM_DECODING".GLOBAL_ALARMS_MACHINE.ALARM_DECODING := #FC_NUMBER;
       "DB442_HOPPERS_ALARM_DECODING".ALARMS_CENTRAL.IS_ALARMS := TRUE;
       "DB441_POWDER_FEEDERS_ALARM_DECODING".GLOBAL_ALARMS_MACHINE.ALARM_DECODING := #FC_NUMBER;
       "DB441_POWDER_FEEDERS_ALARM_DECODING".ALARMS_CENTRAL.IS_ALARMS := TRUE;
   END_IF;
END_REGION

REGION Network 9: STOP END OF CYCLE ALARMS
   RUNG wire#powerrail
      I_Contact( "DB2103_ELECTRICAL_CABINET".AIR_UNIT_1_BREAKER_TRIPPED_ALARM )
      I_Contact( "DB2103_ELECTRICAL_CABINET".AIR_UNIT_2_BREAKER_TRIPPED_ALARM )
      I_Contact( "DB2103_ELECTRICAL_CABINET".PANEL_TEMPERATURE_ALARM )
      I_Contact( "DB2103_ELECTRICAL_CABINET".AIR_UNIT_ALARM_1 )
      I_Contact( "DB2103_ELECTRICAL_CABINET".AIR_UNIT_ALARM_2 )
      I_Contact( "DB2103_ELECTRICAL_CABINET".BATTERY_OK_SITOP_UPS500S_ALARM )
      I_Contact( "DB2103_ELECTRICAL_CABINET".BATTERY_ALARM_SITOP_UPS500S )
      Not()
      Coil( "DB2103_ELECTRICAL_CABINET".SEOC_ALARMS )
      wire#w1
      { S7_GenerateENO := "TRUE" } Move(in := #FC_NUMBER, out1 => "DB442_HOPPERS_ALARM_DECODING".GLOBAL_ALARMS_MACHINE.ALARM_DECODING)
      S_Coil( "DB442_HOPPERS_ALARM_DECODING".ALARMS_CENTRAL.IS_ALARMS )
   END_RUNG
   RUNG wire#w1
      { S7_GenerateENO := "TRUE" } Move(in := #FC_NUMBER, out1 => "DB441_POWDER_FEEDERS_ALARM_DECODING".GLOBAL_ALARMS_MACHINE.ALARM_DECODING)
      S_Coil( "DB441_POWDER_FEEDERS_ALARM_DECODING".ALARMS_CENTRAL.IS_ALARMS )
   END_RUNG
   // the same network as SCL:
   // ENO of a box is taken as its EN; it also drops when the box reports an error
   "DB2103_ELECTRICAL_CABINET".SEOC_ALARMS := NOT (NOT "DB2103_ELECTRICAL_CABINET".AIR_UNIT_1_BREAKER_TRIPPED_ALARM AND NOT "DB2103_ELECTRICAL_CABINET".AIR_UNIT_2_BREAKER_TRIPPED_ALARM AND NOT "DB2103_ELECTRICAL_CABINET".PANEL_TEMPERATURE_ALARM AND NOT "DB2103_ELECTRICAL_CABINET".AIR_UNIT_ALARM_1 AND NOT "DB2103_ELECTRICAL_CABINET".AIR_UNIT_ALARM_2 AND NOT "DB2103_ELECTRICAL_CABINET".BATTERY_OK_SITOP_UPS500S_ALARM AND NOT "DB2103_ELECTRICAL_CABINET".BATTERY_ALARM_SITOP_UPS500S);
   IF "DB2103_ELECTRICAL_CABINET".SEOC_ALARMS THEN
       "DB442_HOPPERS_ALARM_DECODING".GLOBAL_ALARMS_MACHINE.ALARM_DECODING := #FC_NUMBER;
       "DB442_HOPPERS_ALARM_DECODING".ALARMS_CENTRAL.IS_ALARMS := TRUE;
       "DB441_POWDER_FEEDERS_ALARM_DECODING".GLOBAL_ALARMS_MACHINE.ALARM_DECODING := #FC_NUMBER;
       "DB441_POWDER_FEEDERS_ALARM_DECODING".ALARMS_CENTRAL.IS_ALARMS := TRUE;
   END_IF;
END_REGION

REGION Network 10: ANY ACTIVE ALARM
   RUNG wire#powerrail
      I_Contact( "DB2103_ELECTRICAL_CABINET".IS_ALARMS )
      I_Contact( "DB2103_ELECTRICAL_CABINET".SEOC_ALARMS )
      Not()
      Coil( "DB2103_ELECTRICAL_CABINET".ANY_ACTIVE_ALARM )
   END_RUNG
   // the same network as SCL:
   "DB2103_ELECTRICAL_CABINET".ANY_ACTIVE_ALARM := NOT (NOT "DB2103_ELECTRICAL_CABINET".IS_ALARMS AND NOT "DB2103_ELECTRICAL_CABINET".SEOC_ALARMS);
END_REGION

REGION Network 11: WARNINGS
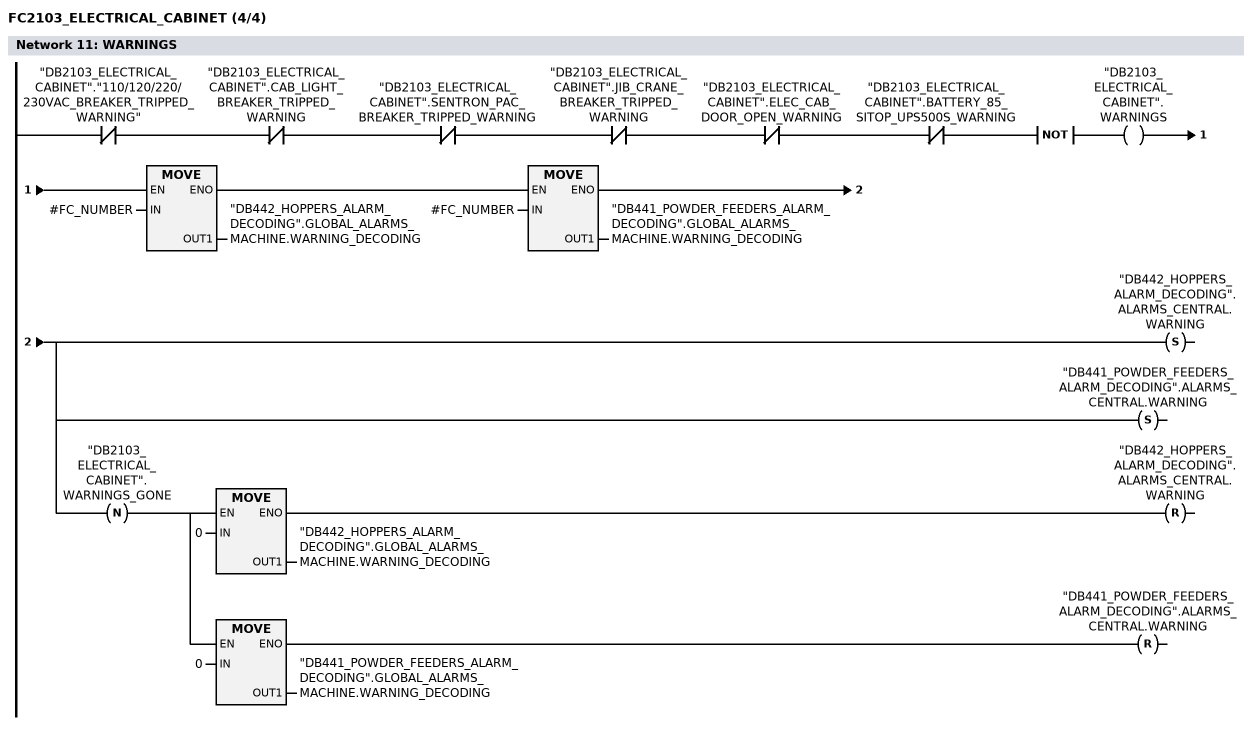
   RUNG wire#powerrail
      I_Contact( "DB2103_ELECTRICAL_CABINET"."110/120/220/230VAC_BREAKER_TRIPPED_WARNING" )
      I_Contact( "DB2103_ELECTRICAL_CABINET".CAB_LIGHT_BREAKER_TRIPPED_WARNING )
      I_Contact( "DB2103_ELECTRICAL_CABINET".SENTRON_PAC_BREAKER_TRIPPED_WARNING )
      I_Contact( "DB2103_ELECTRICAL_CABINET".JIB_CRANE_BREAKER_TRIPPED_WARNING )
      I_Contact( "DB2103_ELECTRICAL_CABINET".ELEC_CAB_DOOR_OPEN_WARNING )
      I_Contact( "DB2103_ELECTRICAL_CABINET".BATTERY_85_SITOP_UPS500S_WARNING )
      Not()
      Coil( "DB2103_ELECTRICAL_CABINET".WARNINGS )
      { S7_GenerateENO := "TRUE" } Move(in := #FC_NUMBER, out1 => "DB442_HOPPERS_ALARM_DECODING".GLOBAL_ALARMS_MACHINE.WARNING_DECODING)
      { S7_GenerateENO := "TRUE" } Move(in := #FC_NUMBER, out1 => "DB441_POWDER_FEEDERS_ALARM_DECODING".GLOBAL_ALARMS_MACHINE.WARNING_DECODING)
      wire#w1
      S_Coil( "DB442_HOPPERS_ALARM_DECODING".ALARMS_CENTRAL.WARNING )
   END_RUNG
   RUNG wire#w1
      S_Coil( "DB441_POWDER_FEEDERS_ALARM_DECODING".ALARMS_CENTRAL.WARNING )
   END_RUNG
   RUNG wire#w1
      N_Trig( "DB2103_ELECTRICAL_CABINET".WARNINGS_GONE )
      wire#w2
      { S7_GenerateENO := "TRUE" } Move(in := 0, out1 => "DB442_HOPPERS_ALARM_DECODING".GLOBAL_ALARMS_MACHINE.WARNING_DECODING)
      R_Coil( "DB442_HOPPERS_ALARM_DECODING".ALARMS_CENTRAL.WARNING )
   END_RUNG
   RUNG wire#w2
      { S7_GenerateENO := "TRUE" } Move(in := 0, out1 => "DB441_POWDER_FEEDERS_ALARM_DECODING".GLOBAL_ALARMS_MACHINE.WARNING_DECODING)
      R_Coil( "DB441_POWDER_FEEDERS_ALARM_DECODING".ALARMS_CENTRAL.WARNING )
   END_RUNG
   // the same network as SCL:
   // ENO of a box is taken as its EN; it also drops when the box reports an error
   "DB2103_ELECTRICAL_CABINET".WARNINGS := NOT (NOT "DB2103_ELECTRICAL_CABINET"."110/120/220/230VAC_BREAKER_TRIPPED_WARNING" AND NOT "DB2103_ELECTRICAL_CABINET".CAB_LIGHT_BREAKER_TRIPPED_WARNING AND NOT "DB2103_ELECTRICAL_CABINET".SENTRON_PAC_BREAKER_TRIPPED_WARNING AND NOT "DB2103_ELECTRICAL_CABINET".JIB_CRANE_BREAKER_TRIPPED_WARNING AND NOT "DB2103_ELECTRICAL_CABINET".ELEC_CAB_DOOR_OPEN_WARNING AND NOT "DB2103_ELECTRICAL_CABINET".BATTERY_85_SITOP_UPS500S_WARNING);
   IF "DB2103_ELECTRICAL_CABINET".WARNINGS THEN
       "DB442_HOPPERS_ALARM_DECODING".GLOBAL_ALARMS_MACHINE.WARNING_DECODING := #FC_NUMBER;
       "DB441_POWDER_FEEDERS_ALARM_DECODING".GLOBAL_ALARMS_MACHINE.WARNING_DECODING := #FC_NUMBER;
       "DB442_HOPPERS_ALARM_DECODING".ALARMS_CENTRAL.WARNING := TRUE;
       "DB441_POWDER_FEEDERS_ALARM_DECODING".ALARMS_CENTRAL.WARNING := TRUE;
   END_IF;
   #_w1 := NOT "DB2103_ELECTRICAL_CABINET".WARNINGS AND "DB2103_ELECTRICAL_CABINET".WARNINGS_GONE;   // falling edge
   "DB2103_ELECTRICAL_CABINET".WARNINGS_GONE := "DB2103_ELECTRICAL_CABINET".WARNINGS;
   IF #_w1 THEN
       "DB442_HOPPERS_ALARM_DECODING".GLOBAL_ALARMS_MACHINE.WARNING_DECODING := 0;
       "DB442_HOPPERS_ALARM_DECODING".ALARMS_CENTRAL.WARNING := FALSE;
       "DB441_POWDER_FEEDERS_ALARM_DECODING".GLOBAL_ALARMS_MACHINE.WARNING_DECODING := 0;
       "DB441_POWDER_FEEDERS_ALARM_DECODING".ALARMS_CENTRAL.WARNING := FALSE;
   END_IF;
END_REGION
END_FUNCTION

FUNCTION "FC2120_MPP_ITC_IPC" : Void   // FC2120, LAD
{ S7_Optimized_Access := 'FALSE' }
AUTHOR : ETXETAR
VERSION : 1.0
// stored: AutoNumber false, IsIECCheckEnabled false, SetENOAutomatically false, UDAEnableTagReadback false
   VAR_TEMP
      O_BYTE_0 : Struct   // OPTIONS BYTE 0
         IPC : Bool;   // IPC OPTION
      END_STRUCT;
      TCU_INDEX_SEL : Int;
   END_VAR
   VAR CONSTANT
      FC_NUMBER : DInt := 2120;   // FC NUMBER
   END_VAR
   VAR_TEMP   // added for the SCL form of the ladder/FBD networks
      _w1 : Bool;
      _w2 : Bool;
   END_VAR
BEGIN

REGION Network 1: OPTIONS
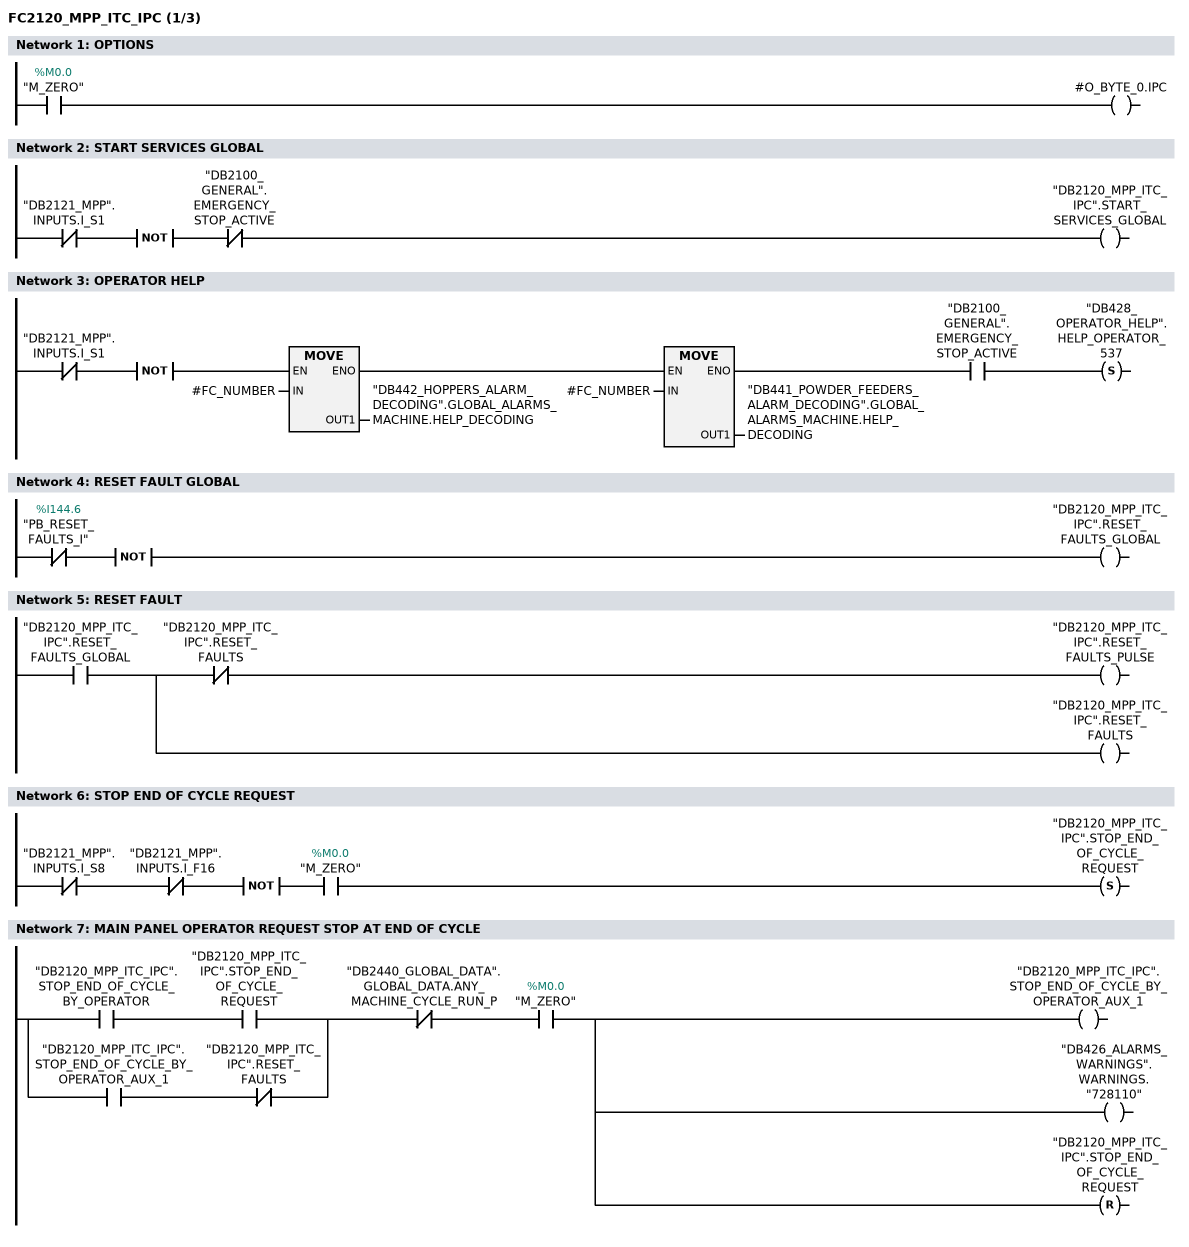
   RUNG wire#powerrail
      Contact( "M_ZERO" )
      Coil( #O_BYTE_0.IPC )
   END_RUNG
   // the same network as SCL:
   #O_BYTE_0.IPC := "M_ZERO";
END_REGION

REGION Network 2: START SERVICES GLOBAL
   RUNG wire#powerrail
      I_Contact( "DB2121_MPP".INPUTS.I_S1 )
      Not()
      I_Contact( "DB2100_GENERAL".EMERGENCY_STOP_ACTIVE )
      Coil( "DB2120_MPP_ITC_IPC".START_SERVICES_GLOBAL )
   END_RUNG
   // the same network as SCL:
   "DB2120_MPP_ITC_IPC".START_SERVICES_GLOBAL := NOT (NOT "DB2121_MPP".INPUTS.I_S1) AND NOT "DB2100_GENERAL".EMERGENCY_STOP_ACTIVE;
END_REGION

REGION Network 3: OPERATOR HELP
   RUNG wire#powerrail
      I_Contact( "DB2121_MPP".INPUTS.I_S1 )
      Not()
      { S7_GenerateENO := "TRUE" } Move(in := #FC_NUMBER, out1 => "DB442_HOPPERS_ALARM_DECODING".GLOBAL_ALARMS_MACHINE.HELP_DECODING)
      { S7_GenerateENO := "TRUE" } Move(in := #FC_NUMBER, out1 => "DB441_POWDER_FEEDERS_ALARM_DECODING".GLOBAL_ALARMS_MACHINE.HELP_DECODING)
      Contact( "DB2100_GENERAL".EMERGENCY_STOP_ACTIVE )
      S_Coil( "DB428_OPERATOR_HELP".HELP_OPERATOR_537 )
   END_RUNG
   // the same network as SCL:
   // ENO of a box is taken as its EN; it also drops when the box reports an error
   #_w1 := NOT (NOT "DB2121_MPP".INPUTS.I_S1);
   IF #_w1 THEN
       "DB442_HOPPERS_ALARM_DECODING".GLOBAL_ALARMS_MACHINE.HELP_DECODING := #FC_NUMBER;
       "DB441_POWDER_FEEDERS_ALARM_DECODING".GLOBAL_ALARMS_MACHINE.HELP_DECODING := #FC_NUMBER;
   END_IF;
   IF #_w1 AND "DB2100_GENERAL".EMERGENCY_STOP_ACTIVE THEN
       "DB428_OPERATOR_HELP".HELP_OPERATOR_537 := TRUE;
   END_IF;
END_REGION

REGION Network 4: RESET FAULT GLOBAL
   RUNG wire#powerrail
      I_Contact( "PB_RESET_FAULTS_I" )
      Not()
      Coil( "DB2120_MPP_ITC_IPC".RESET_FAULTS_GLOBAL )
   END_RUNG
   // the same network as SCL:
   "DB2120_MPP_ITC_IPC".RESET_FAULTS_GLOBAL := NOT (NOT "PB_RESET_FAULTS_I");
END_REGION

REGION Network 5: RESET FAULT
   RUNG wire#powerrail
      Contact( "DB2120_MPP_ITC_IPC".RESET_FAULTS_GLOBAL )
      wire#w1
      I_Contact( "DB2120_MPP_ITC_IPC".RESET_FAULTS )
      Coil( "DB2120_MPP_ITC_IPC".RESET_FAULTS_PULSE )
   END_RUNG
   RUNG wire#w1
      Coil( "DB2120_MPP_ITC_IPC".RESET_FAULTS )
   END_RUNG
   // the same network as SCL:
   "DB2120_MPP_ITC_IPC".RESET_FAULTS_PULSE := "DB2120_MPP_ITC_IPC".RESET_FAULTS_GLOBAL AND NOT "DB2120_MPP_ITC_IPC".RESET_FAULTS;
   "DB2120_MPP_ITC_IPC".RESET_FAULTS := "DB2120_MPP_ITC_IPC".RESET_FAULTS_GLOBAL;
END_REGION

REGION Network 6: STOP END OF CYCLE REQUEST
   RUNG wire#powerrail
      I_Contact( "DB2121_MPP".INPUTS.I_S8 )
      I_Contact( "DB2121_MPP".INPUTS.I_F16 )
      Not()
      Contact( "M_ZERO" )
      S_Coil( "DB2120_MPP_ITC_IPC".STOP_END_OF_CYCLE_REQUEST )
   END_RUNG
   // the same network as SCL:
   IF NOT (NOT "DB2121_MPP".INPUTS.I_S8 AND NOT "DB2121_MPP".INPUTS.I_F16) AND "M_ZERO" THEN
       "DB2120_MPP_ITC_IPC".STOP_END_OF_CYCLE_REQUEST := TRUE;
   END_IF;
END_REGION

REGION Network 7: MAIN PANEL OPERATOR REQUEST STOP AT END OF CYCLE
   RUNG wire#powerrail
      Contact( "DB2120_MPP_ITC_IPC".STOP_END_OF_CYCLE_BY_OPERATOR )
      Contact( "DB2120_MPP_ITC_IPC".STOP_END_OF_CYCLE_REQUEST )
      wire#w1
      I_Contact( "DB2440_GLOBAL_DATA".GLOBAL_DATA.ANY_MACHINE_CYCLE_RUN_P )
      Contact( "M_ZERO" )
      wire#w2
      Coil( "DB2120_MPP_ITC_IPC".STOP_END_OF_CYCLE_BY_OPERATOR_AUX_1 )
   END_RUNG
   RUNG wire#powerrail
      Contact( "DB2120_MPP_ITC_IPC".STOP_END_OF_CYCLE_BY_OPERATOR_AUX_1 )
      I_Contact( "DB2120_MPP_ITC_IPC".RESET_FAULTS )
   END_RUNG wire#w1
   RUNG wire#w2
      Coil( "DB426_ALARMS_WARNINGS".WARNINGS."728110" )
   END_RUNG
   RUNG wire#w2
      R_Coil( "DB2120_MPP_ITC_IPC".STOP_END_OF_CYCLE_REQUEST )
   END_RUNG
   // the same network as SCL:
   "DB2120_MPP_ITC_IPC".STOP_END_OF_CYCLE_BY_OPERATOR_AUX_1 := (("DB2120_MPP_ITC_IPC".STOP_END_OF_CYCLE_BY_OPERATOR AND "DB2120_MPP_ITC_IPC".STOP_END_OF_CYCLE_REQUEST) OR ("DB2120_MPP_ITC_IPC".STOP_END_OF_CYCLE_BY_OPERATOR_AUX_1 AND NOT "DB2120_MPP_ITC_IPC".RESET_FAULTS)) AND NOT "DB2440_GLOBAL_DATA".GLOBAL_DATA.ANY_MACHINE_CYCLE_RUN_P AND "M_ZERO";
   "DB426_ALARMS_WARNINGS".WARNINGS."728110" := "DB2120_MPP_ITC_IPC".STOP_END_OF_CYCLE_BY_OPERATOR_AUX_1;
   IF "DB2120_MPP_ITC_IPC".STOP_END_OF_CYCLE_BY_OPERATOR_AUX_1 THEN
       "DB2120_MPP_ITC_IPC".STOP_END_OF_CYCLE_REQUEST := FALSE;
   END_IF;
END_REGION

REGION Network 8: AUXILIARY PANEL OPERATOR REQUEST STOP AT END OF CYCLE
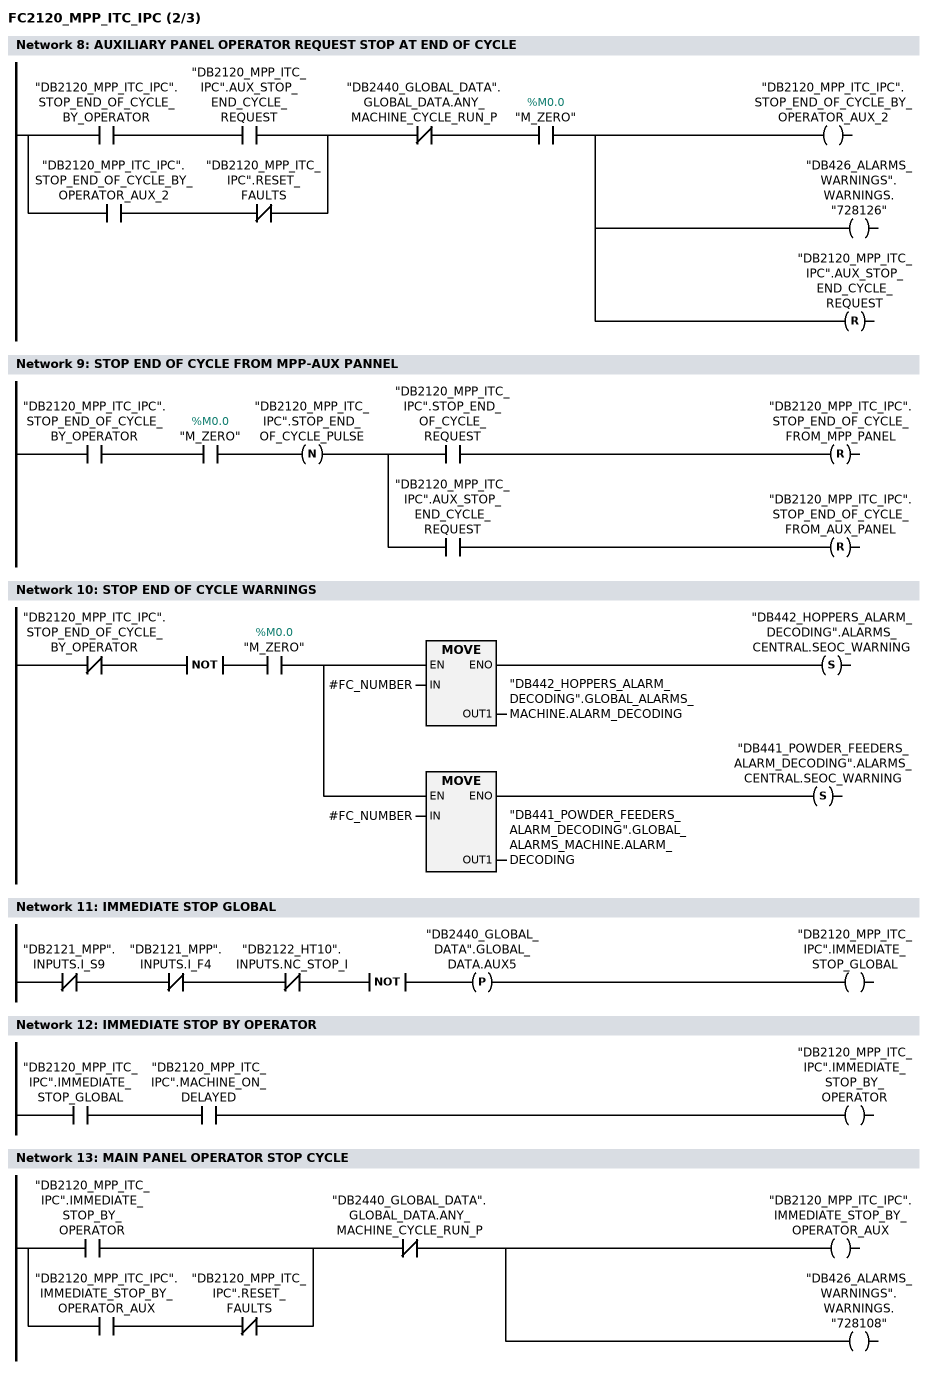
   RUNG wire#powerrail
      Contact( "DB2120_MPP_ITC_IPC".STOP_END_OF_CYCLE_BY_OPERATOR )
      Contact( "DB2120_MPP_ITC_IPC".AUX_STOP_END_CYCLE_REQUEST )
      wire#w1
      I_Contact( "DB2440_GLOBAL_DATA".GLOBAL_DATA.ANY_MACHINE_CYCLE_RUN_P )
      Contact( "M_ZERO" )
      wire#w2
      Coil( "DB2120_MPP_ITC_IPC".STOP_END_OF_CYCLE_BY_OPERATOR_AUX_2 )
   END_RUNG
   RUNG wire#powerrail
      Contact( "DB2120_MPP_ITC_IPC".STOP_END_OF_CYCLE_BY_OPERATOR_AUX_2 )
      I_Contact( "DB2120_MPP_ITC_IPC".RESET_FAULTS )
   END_RUNG wire#w1
   RUNG wire#w2
      Coil( "DB426_ALARMS_WARNINGS".WARNINGS."728126" )
   END_RUNG
   RUNG wire#w2
      R_Coil( "DB2120_MPP_ITC_IPC".AUX_STOP_END_CYCLE_REQUEST )
   END_RUNG
   // the same network as SCL:
   "DB2120_MPP_ITC_IPC".STOP_END_OF_CYCLE_BY_OPERATOR_AUX_2 := (("DB2120_MPP_ITC_IPC".STOP_END_OF_CYCLE_BY_OPERATOR AND "DB2120_MPP_ITC_IPC".AUX_STOP_END_CYCLE_REQUEST) OR ("DB2120_MPP_ITC_IPC".STOP_END_OF_CYCLE_BY_OPERATOR_AUX_2 AND NOT "DB2120_MPP_ITC_IPC".RESET_FAULTS)) AND NOT "DB2440_GLOBAL_DATA".GLOBAL_DATA.ANY_MACHINE_CYCLE_RUN_P AND "M_ZERO";
   "DB426_ALARMS_WARNINGS".WARNINGS."728126" := "DB2120_MPP_ITC_IPC".STOP_END_OF_CYCLE_BY_OPERATOR_AUX_2;
   IF "DB2120_MPP_ITC_IPC".STOP_END_OF_CYCLE_BY_OPERATOR_AUX_2 THEN
       "DB2120_MPP_ITC_IPC".AUX_STOP_END_CYCLE_REQUEST := FALSE;
   END_IF;
END_REGION

REGION Network 9: STOP END OF CYCLE FROM MPP-AUX PANNEL
   RUNG wire#powerrail
      Contact( "DB2120_MPP_ITC_IPC".STOP_END_OF_CYCLE_BY_OPERATOR )
      Contact( "M_ZERO" )
      N_Trig( "DB2120_MPP_ITC_IPC".STOP_END_OF_CYCLE_PULSE )
      wire#w1
      Contact( "DB2120_MPP_ITC_IPC".STOP_END_OF_CYCLE_REQUEST )
      R_Coil( "DB2120_MPP_ITC_IPC".STOP_END_OF_CYCLE_FROM_MPP_PANEL )
   END_RUNG
   RUNG wire#w1
      Contact( "DB2120_MPP_ITC_IPC".AUX_STOP_END_CYCLE_REQUEST )
      R_Coil( "DB2120_MPP_ITC_IPC".STOP_END_OF_CYCLE_FROM_AUX_PANEL )
   END_RUNG
   // the same network as SCL:
   #_w1 := "DB2120_MPP_ITC_IPC".STOP_END_OF_CYCLE_BY_OPERATOR AND "M_ZERO";
   #_w2 := NOT #_w1 AND "DB2120_MPP_ITC_IPC".STOP_END_OF_CYCLE_PULSE;   // falling edge
   "DB2120_MPP_ITC_IPC".STOP_END_OF_CYCLE_PULSE := #_w1;
   IF #_w2 AND "DB2120_MPP_ITC_IPC".STOP_END_OF_CYCLE_REQUEST THEN
       "DB2120_MPP_ITC_IPC".STOP_END_OF_CYCLE_FROM_MPP_PANEL := FALSE;
   END_IF;
   IF #_w2 AND "DB2120_MPP_ITC_IPC".AUX_STOP_END_CYCLE_REQUEST THEN
       "DB2120_MPP_ITC_IPC".STOP_END_OF_CYCLE_FROM_AUX_PANEL := FALSE;
   END_IF;
END_REGION

REGION Network 10: STOP END OF CYCLE WARNINGS
   RUNG wire#powerrail
      I_Contact( "DB2120_MPP_ITC_IPC".STOP_END_OF_CYCLE_BY_OPERATOR )
      Not()
      Contact( "M_ZERO" )
      wire#w1
      { S7_GenerateENO := "TRUE" } Move(in := #FC_NUMBER, out1 => "DB442_HOPPERS_ALARM_DECODING".GLOBAL_ALARMS_MACHINE.ALARM_DECODING)
      S_Coil( "DB442_HOPPERS_ALARM_DECODING".ALARMS_CENTRAL.SEOC_WARNING )
   END_RUNG
   RUNG wire#w1
      { S7_GenerateENO := "TRUE" } Move(in := #FC_NUMBER, out1 => "DB441_POWDER_FEEDERS_ALARM_DECODING".GLOBAL_ALARMS_MACHINE.ALARM_DECODING)
      S_Coil( "DB441_POWDER_FEEDERS_ALARM_DECODING".ALARMS_CENTRAL.SEOC_WARNING )
   END_RUNG
   // the same network as SCL:
   // ENO of a box is taken as its EN; it also drops when the box reports an error
   IF NOT (NOT "DB2120_MPP_ITC_IPC".STOP_END_OF_CYCLE_BY_OPERATOR) AND "M_ZERO" THEN
       "DB442_HOPPERS_ALARM_DECODING".GLOBAL_ALARMS_MACHINE.ALARM_DECODING := #FC_NUMBER;
       "DB442_HOPPERS_ALARM_DECODING".ALARMS_CENTRAL.SEOC_WARNING := TRUE;
       "DB441_POWDER_FEEDERS_ALARM_DECODING".GLOBAL_ALARMS_MACHINE.ALARM_DECODING := #FC_NUMBER;
       "DB441_POWDER_FEEDERS_ALARM_DECODING".ALARMS_CENTRAL.SEOC_WARNING := TRUE;
   END_IF;
END_REGION

REGION Network 11: IMMEDIATE STOP GLOBAL
   RUNG wire#powerrail
      I_Contact( "DB2121_MPP".INPUTS.I_S9 )
      I_Contact( "DB2121_MPP".INPUTS.I_F4 )
      I_Contact( "DB2122_HT10".INPUTS.NC_STOP_I )
      Not()
      P_Trig( "DB2440_GLOBAL_DATA".GLOBAL_DATA.AUX5 )
      Coil( "DB2120_MPP_ITC_IPC".IMMEDIATE_STOP_GLOBAL )
   END_RUNG
   // the same network as SCL:
   #_w1 := NOT (NOT "DB2121_MPP".INPUTS.I_S9 AND NOT "DB2121_MPP".INPUTS.I_F4 AND NOT "DB2122_HT10".INPUTS.NC_STOP_I);
   #_w2 := #_w1 AND NOT "DB2440_GLOBAL_DATA".GLOBAL_DATA.AUX5;   // rising edge
   "DB2440_GLOBAL_DATA".GLOBAL_DATA.AUX5 := #_w1;
   "DB2120_MPP_ITC_IPC".IMMEDIATE_STOP_GLOBAL := #_w2;
END_REGION

REGION Network 12: IMMEDIATE STOP BY OPERATOR
   RUNG wire#powerrail
      Contact( "DB2120_MPP_ITC_IPC".IMMEDIATE_STOP_GLOBAL )
      Contact( "DB2120_MPP_ITC_IPC".MACHINE_ON_DELAYED )
      Coil( "DB2120_MPP_ITC_IPC".IMMEDIATE_STOP_BY_OPERATOR )
   END_RUNG
   // the same network as SCL:
   "DB2120_MPP_ITC_IPC".IMMEDIATE_STOP_BY_OPERATOR := "DB2120_MPP_ITC_IPC".IMMEDIATE_STOP_GLOBAL AND "DB2120_MPP_ITC_IPC".MACHINE_ON_DELAYED;
END_REGION

REGION Network 13: MAIN PANEL OPERATOR STOP CYCLE
   RUNG wire#powerrail
      Contact( "DB2120_MPP_ITC_IPC".IMMEDIATE_STOP_BY_OPERATOR )
      wire#w1
      I_Contact( "DB2440_GLOBAL_DATA".GLOBAL_DATA.ANY_MACHINE_CYCLE_RUN_P )
      wire#w2
      Coil( "DB2120_MPP_ITC_IPC".IMMEDIATE_STOP_BY_OPERATOR_AUX )
   END_RUNG
   RUNG wire#powerrail
      Contact( "DB2120_MPP_ITC_IPC".IMMEDIATE_STOP_BY_OPERATOR_AUX )
      I_Contact( "DB2120_MPP_ITC_IPC".RESET_FAULTS )
   END_RUNG wire#w1
   RUNG wire#w2
      Coil( "DB426_ALARMS_WARNINGS".WARNINGS."728108" )
   END_RUNG
   // the same network as SCL:
   "DB2120_MPP_ITC_IPC".IMMEDIATE_STOP_BY_OPERATOR_AUX := ("DB2120_MPP_ITC_IPC".IMMEDIATE_STOP_BY_OPERATOR OR ("DB2120_MPP_ITC_IPC".IMMEDIATE_STOP_BY_OPERATOR_AUX AND NOT "DB2120_MPP_ITC_IPC".RESET_FAULTS)) AND NOT "DB2440_GLOBAL_DATA".GLOBAL_DATA.ANY_MACHINE_CYCLE_RUN_P;
   "DB426_ALARMS_WARNINGS".WARNINGS."728108" := "DB2120_MPP_ITC_IPC".IMMEDIATE_STOP_BY_OPERATOR_AUX;
END_REGION

REGION Network 14: IMMEDIATE STOP WARNING
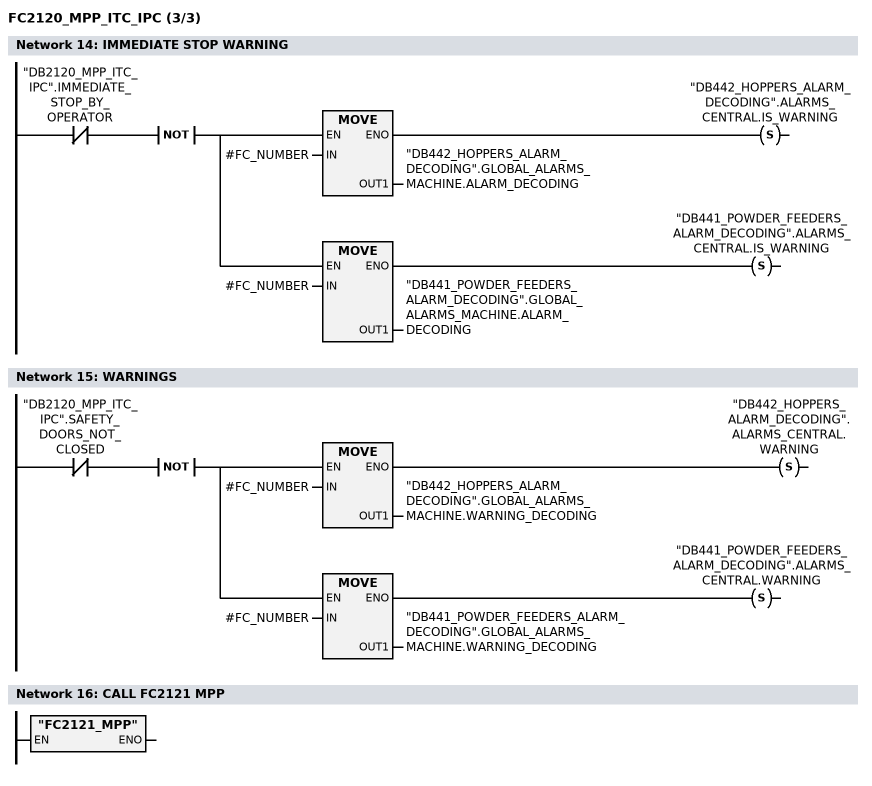
   RUNG wire#powerrail
      I_Contact( "DB2120_MPP_ITC_IPC".IMMEDIATE_STOP_BY_OPERATOR )
      Not()
      wire#w1
      { S7_GenerateENO := "TRUE" } Move(in := #FC_NUMBER, out1 => "DB442_HOPPERS_ALARM_DECODING".GLOBAL_ALARMS_MACHINE.ALARM_DECODING)
      S_Coil( "DB442_HOPPERS_ALARM_DECODING".ALARMS_CENTRAL.IS_WARNING )
   END_RUNG
   RUNG wire#w1
      { S7_GenerateENO := "TRUE" } Move(in := #FC_NUMBER, out1 => "DB441_POWDER_FEEDERS_ALARM_DECODING".GLOBAL_ALARMS_MACHINE.ALARM_DECODING)
      S_Coil( "DB441_POWDER_FEEDERS_ALARM_DECODING".ALARMS_CENTRAL.IS_WARNING )
   END_RUNG
   // the same network as SCL:
   // ENO of a box is taken as its EN; it also drops when the box reports an error
   IF NOT (NOT "DB2120_MPP_ITC_IPC".IMMEDIATE_STOP_BY_OPERATOR) THEN
       "DB442_HOPPERS_ALARM_DECODING".GLOBAL_ALARMS_MACHINE.ALARM_DECODING := #FC_NUMBER;
       "DB442_HOPPERS_ALARM_DECODING".ALARMS_CENTRAL.IS_WARNING := TRUE;
       "DB441_POWDER_FEEDERS_ALARM_DECODING".GLOBAL_ALARMS_MACHINE.ALARM_DECODING := #FC_NUMBER;
       "DB441_POWDER_FEEDERS_ALARM_DECODING".ALARMS_CENTRAL.IS_WARNING := TRUE;
   END_IF;
END_REGION

REGION Network 15: WARNINGS
   RUNG wire#powerrail
      I_Contact( "DB2120_MPP_ITC_IPC".SAFETY_DOORS_NOT_CLOSED )
      Not()
      wire#w1
      { S7_GenerateENO := "TRUE" } Move(in := #FC_NUMBER, out1 => "DB442_HOPPERS_ALARM_DECODING".GLOBAL_ALARMS_MACHINE.WARNING_DECODING)
      S_Coil( "DB442_HOPPERS_ALARM_DECODING".ALARMS_CENTRAL.WARNING )
   END_RUNG
   RUNG wire#w1
      { S7_GenerateENO := "TRUE" } Move(in := #FC_NUMBER, out1 => "DB441_POWDER_FEEDERS_ALARM_DECODING".GLOBAL_ALARMS_MACHINE.WARNING_DECODING)
      S_Coil( "DB441_POWDER_FEEDERS_ALARM_DECODING".ALARMS_CENTRAL.WARNING )
   END_RUNG
   // the same network as SCL:
   // ENO of a box is taken as its EN; it also drops when the box reports an error
   IF NOT (NOT "DB2120_MPP_ITC_IPC".SAFETY_DOORS_NOT_CLOSED) THEN
       "DB442_HOPPERS_ALARM_DECODING".GLOBAL_ALARMS_MACHINE.WARNING_DECODING := #FC_NUMBER;
       "DB442_HOPPERS_ALARM_DECODING".ALARMS_CENTRAL.WARNING := TRUE;
       "DB441_POWDER_FEEDERS_ALARM_DECODING".GLOBAL_ALARMS_MACHINE.WARNING_DECODING := #FC_NUMBER;
       "DB441_POWDER_FEEDERS_ALARM_DECODING".ALARMS_CENTRAL.WARNING := TRUE;
   END_IF;
END_REGION

REGION Network 16: CALL FC2121 MPP
   RUNG wire#powerrail
      "FC2121_MPP"()
   END_RUNG
   // the same network as SCL:
   "FC2121_MPP"();
END_REGION
END_FUNCTION

FUNCTION "FC2121_MPP" : Void   // FC2121, LAD
{ S7_Optimized_Access := 'FALSE' }
AUTHOR : ETXETAR
VERSION : 1.0
// stored: AutoNumber false, IsIECCheckEnabled false, SetENOAutomatically false, UDAEnableTagReadback false
   VAR_TEMP
      ONE : Int;
      RETVAL1 : Int;
      SIMU_PANEL_HMI_SEL : Bool;   // SIMULATED PANEL IN HMI SELECTED
   END_VAR
   VAR CONSTANT
      FC_NUMBER : DInt := 2121;   // FC NUMBER
   END_VAR
BEGIN

REGION Network 1: INPUTS
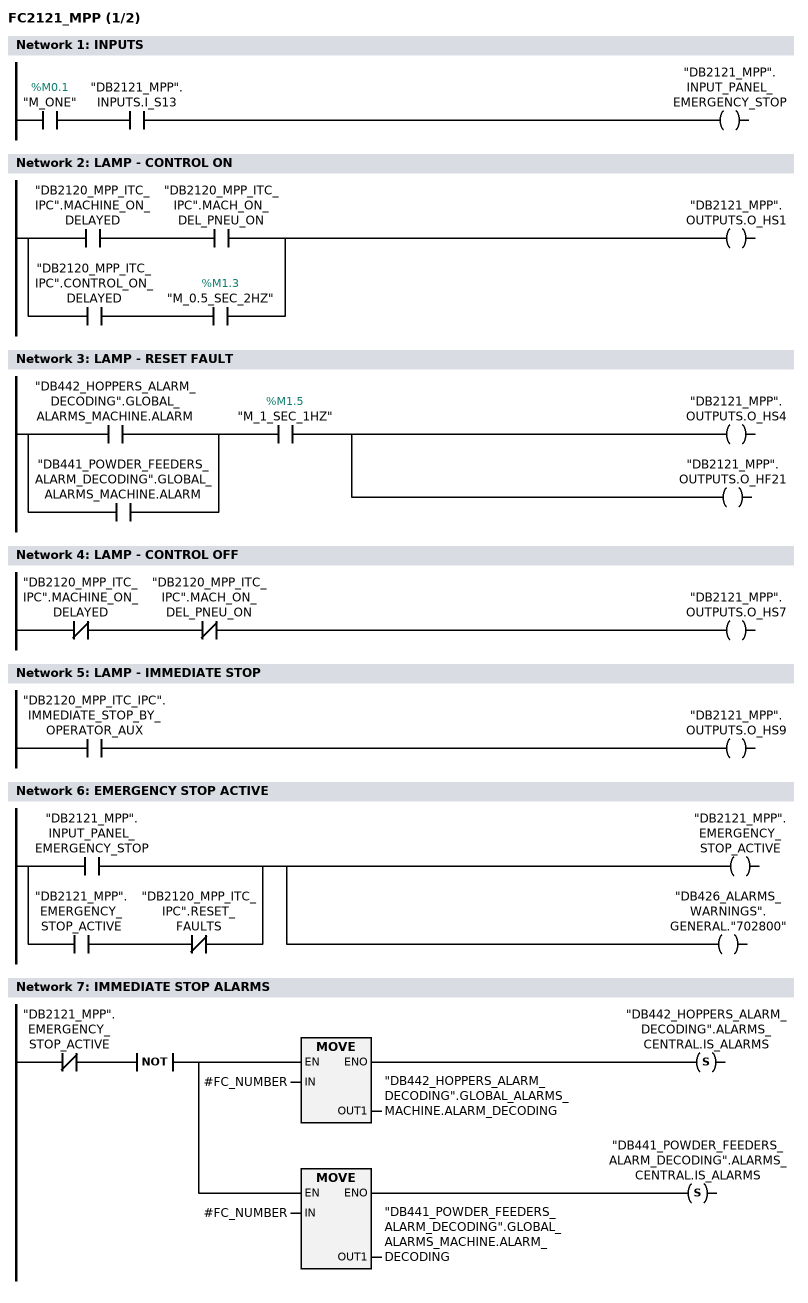
   RUNG wire#powerrail
      Contact( "M_ONE" )
      Contact( "DB2121_MPP".INPUTS.I_S13 )
      Coil( "DB2121_MPP".INPUT_PANEL_EMERGENCY_STOP )
   END_RUNG
   // the same network as SCL:
   "DB2121_MPP".INPUT_PANEL_EMERGENCY_STOP := "M_ONE" AND "DB2121_MPP".INPUTS.I_S13;
END_REGION

REGION Network 2: LAMP - CONTROL ON
   RUNG wire#powerrail
      Contact( "DB2120_MPP_ITC_IPC".MACHINE_ON_DELAYED )
      Contact( "DB2120_MPP_ITC_IPC".MACH_ON_DEL_PNEU_ON )
      wire#w1
      Coil( "DB2121_MPP".OUTPUTS.O_HS1 )
   END_RUNG
   RUNG wire#powerrail
      Contact( "DB2120_MPP_ITC_IPC".CONTROL_ON_DELAYED )
      Contact( "M_0.5_SEC_2HZ" )
   END_RUNG wire#w1
   // the same network as SCL:
   "DB2121_MPP".OUTPUTS.O_HS1 := ("DB2120_MPP_ITC_IPC".MACHINE_ON_DELAYED AND "DB2120_MPP_ITC_IPC".MACH_ON_DEL_PNEU_ON) OR ("DB2120_MPP_ITC_IPC".CONTROL_ON_DELAYED AND "M_0.5_SEC_2HZ");
END_REGION

REGION Network 3: LAMP - RESET FAULT
   RUNG wire#powerrail
      Contact( "DB442_HOPPERS_ALARM_DECODING".GLOBAL_ALARMS_MACHINE.ALARM )
      wire#w1
      Contact( "M_1_SEC_1HZ" )
      wire#w2
      Coil( "DB2121_MPP".OUTPUTS.O_HS4 )
   END_RUNG
   RUNG wire#powerrail
      Contact( "DB441_POWDER_FEEDERS_ALARM_DECODING".GLOBAL_ALARMS_MACHINE.ALARM )
   END_RUNG wire#w1
   RUNG wire#w2
      Coil( "DB2121_MPP".OUTPUTS.O_HF21 )
   END_RUNG
   // the same network as SCL:
   "DB2121_MPP".OUTPUTS.O_HS4 := ("DB442_HOPPERS_ALARM_DECODING".GLOBAL_ALARMS_MACHINE.ALARM OR "DB441_POWDER_FEEDERS_ALARM_DECODING".GLOBAL_ALARMS_MACHINE.ALARM) AND "M_1_SEC_1HZ";
   "DB2121_MPP".OUTPUTS.O_HF21 := "DB2121_MPP".OUTPUTS.O_HS4;
END_REGION

REGION Network 4: LAMP - CONTROL OFF
   RUNG wire#powerrail
      I_Contact( "DB2120_MPP_ITC_IPC".MACHINE_ON_DELAYED )
      I_Contact( "DB2120_MPP_ITC_IPC".MACH_ON_DEL_PNEU_ON )
      Coil( "DB2121_MPP".OUTPUTS.O_HS7 )
   END_RUNG
   // the same network as SCL:
   "DB2121_MPP".OUTPUTS.O_HS7 := NOT "DB2120_MPP_ITC_IPC".MACHINE_ON_DELAYED AND NOT "DB2120_MPP_ITC_IPC".MACH_ON_DEL_PNEU_ON;
END_REGION

REGION Network 5: LAMP - IMMEDIATE STOP
   RUNG wire#powerrail
      Contact( "DB2120_MPP_ITC_IPC".IMMEDIATE_STOP_BY_OPERATOR_AUX )
      Coil( "DB2121_MPP".OUTPUTS.O_HS9 )
   END_RUNG
   // the same network as SCL:
   "DB2121_MPP".OUTPUTS.O_HS9 := "DB2120_MPP_ITC_IPC".IMMEDIATE_STOP_BY_OPERATOR_AUX;
END_REGION

REGION Network 6: EMERGENCY STOP ACTIVE
   RUNG wire#powerrail
      Contact( "DB2121_MPP".INPUT_PANEL_EMERGENCY_STOP )
      wire#w1
      Coil( "DB2121_MPP".EMERGENCY_STOP_ACTIVE )
   END_RUNG
   RUNG wire#powerrail
      Contact( "DB2121_MPP".EMERGENCY_STOP_ACTIVE )
      I_Contact( "DB2120_MPP_ITC_IPC".RESET_FAULTS )
   END_RUNG wire#w1
   RUNG wire#w1
      Coil( "DB426_ALARMS_WARNINGS".GENERAL."702800" )
   END_RUNG
   // the same network as SCL:
   "DB2121_MPP".EMERGENCY_STOP_ACTIVE := "DB2121_MPP".INPUT_PANEL_EMERGENCY_STOP OR ("DB2121_MPP".EMERGENCY_STOP_ACTIVE AND NOT "DB2120_MPP_ITC_IPC".RESET_FAULTS);
   "DB426_ALARMS_WARNINGS".GENERAL."702800" := "DB2121_MPP".EMERGENCY_STOP_ACTIVE;
END_REGION

REGION Network 7: IMMEDIATE STOP ALARMS
   RUNG wire#powerrail
      I_Contact( "DB2121_MPP".EMERGENCY_STOP_ACTIVE )
      Not()
      wire#w1
      { S7_GenerateENO := "TRUE" } Move(in := #FC_NUMBER, out1 => "DB442_HOPPERS_ALARM_DECODING".GLOBAL_ALARMS_MACHINE.ALARM_DECODING)
      S_Coil( "DB442_HOPPERS_ALARM_DECODING".ALARMS_CENTRAL.IS_ALARMS )
   END_RUNG
   RUNG wire#w1
      { S7_GenerateENO := "TRUE" } Move(in := #FC_NUMBER, out1 => "DB441_POWDER_FEEDERS_ALARM_DECODING".GLOBAL_ALARMS_MACHINE.ALARM_DECODING)
      S_Coil( "DB441_POWDER_FEEDERS_ALARM_DECODING".ALARMS_CENTRAL.IS_ALARMS )
   END_RUNG
   // the same network as SCL:
   // ENO of a box is taken as its EN; it also drops when the box reports an error
   IF NOT (NOT "DB2121_MPP".EMERGENCY_STOP_ACTIVE) THEN
       "DB442_HOPPERS_ALARM_DECODING".GLOBAL_ALARMS_MACHINE.ALARM_DECODING := #FC_NUMBER;
       "DB442_HOPPERS_ALARM_DECODING".ALARMS_CENTRAL.IS_ALARMS := TRUE;
       "DB441_POWDER_FEEDERS_ALARM_DECODING".GLOBAL_ALARMS_MACHINE.ALARM_DECODING := #FC_NUMBER;
       "DB441_POWDER_FEEDERS_ALARM_DECODING".ALARMS_CENTRAL.IS_ALARMS := TRUE;
   END_IF;
END_REGION

REGION Network 8: WARNING
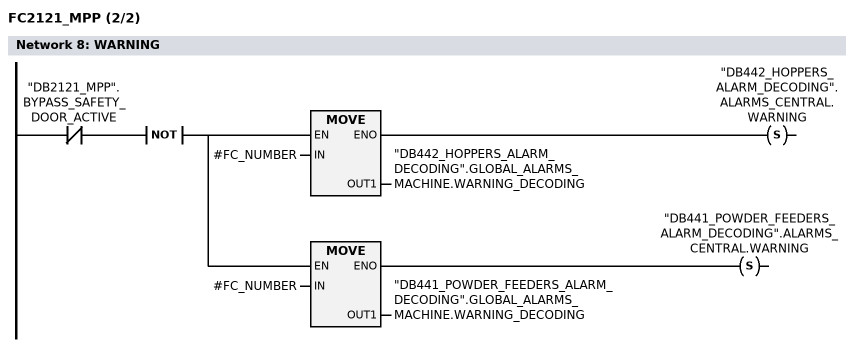
   RUNG wire#powerrail
      I_Contact( "DB2121_MPP".BYPASS_SAFETY_DOOR_ACTIVE )
      Not()
      wire#w1
      { S7_GenerateENO := "TRUE" } Move(in := #FC_NUMBER, out1 => "DB442_HOPPERS_ALARM_DECODING".GLOBAL_ALARMS_MACHINE.WARNING_DECODING)
      S_Coil( "DB442_HOPPERS_ALARM_DECODING".ALARMS_CENTRAL.WARNING )
   END_RUNG
   RUNG wire#w1
      { S7_GenerateENO := "TRUE" } Move(in := #FC_NUMBER, out1 => "DB441_POWDER_FEEDERS_ALARM_DECODING".GLOBAL_ALARMS_MACHINE.WARNING_DECODING)
      S_Coil( "DB441_POWDER_FEEDERS_ALARM_DECODING".ALARMS_CENTRAL.WARNING )
   END_RUNG
   // the same network as SCL:
   // ENO of a box is taken as its EN; it also drops when the box reports an error
   IF NOT (NOT "DB2121_MPP".BYPASS_SAFETY_DOOR_ACTIVE) THEN
       "DB442_HOPPERS_ALARM_DECODING".GLOBAL_ALARMS_MACHINE.WARNING_DECODING := #FC_NUMBER;
       "DB442_HOPPERS_ALARM_DECODING".ALARMS_CENTRAL.WARNING := TRUE;
       "DB441_POWDER_FEEDERS_ALARM_DECODING".GLOBAL_ALARMS_MACHINE.WARNING_DECODING := #FC_NUMBER;
       "DB441_POWDER_FEEDERS_ALARM_DECODING".ALARMS_CENTRAL.WARNING := TRUE;
   END_IF;
END_REGION
END_FUNCTION

FUNCTION "FC2109_HOPPERS_CONTROL_ON" : Void   // FC2109, LAD
{ S7_Optimized_Access := 'FALSE' }
AUTHOR : ETXETAR
VERSION : 1.0
// stored: AutoNumber false, IsIECCheckEnabled false, SetENOAutomatically false, UDAEnableTagReadback false
   VAR_TEMP
      O_BYTE_0 : Struct   // OPTIONS BYTE 0
         GM_COOLANT_PUMP_OFF_DELAY : Bool;   // GM COOLANT PUMP POWER OFF DELAY OPTION
      END_STRUCT;
   END_VAR
   VAR CONSTANT
      FC_NUMBER : DInt := 2109;   // FC NUMBER
   END_VAR
   VAR_TEMP   // added for the SCL form of the ladder/FBD networks
      _w1 : Bool;
   END_VAR
BEGIN

REGION Network 1: INPUTS
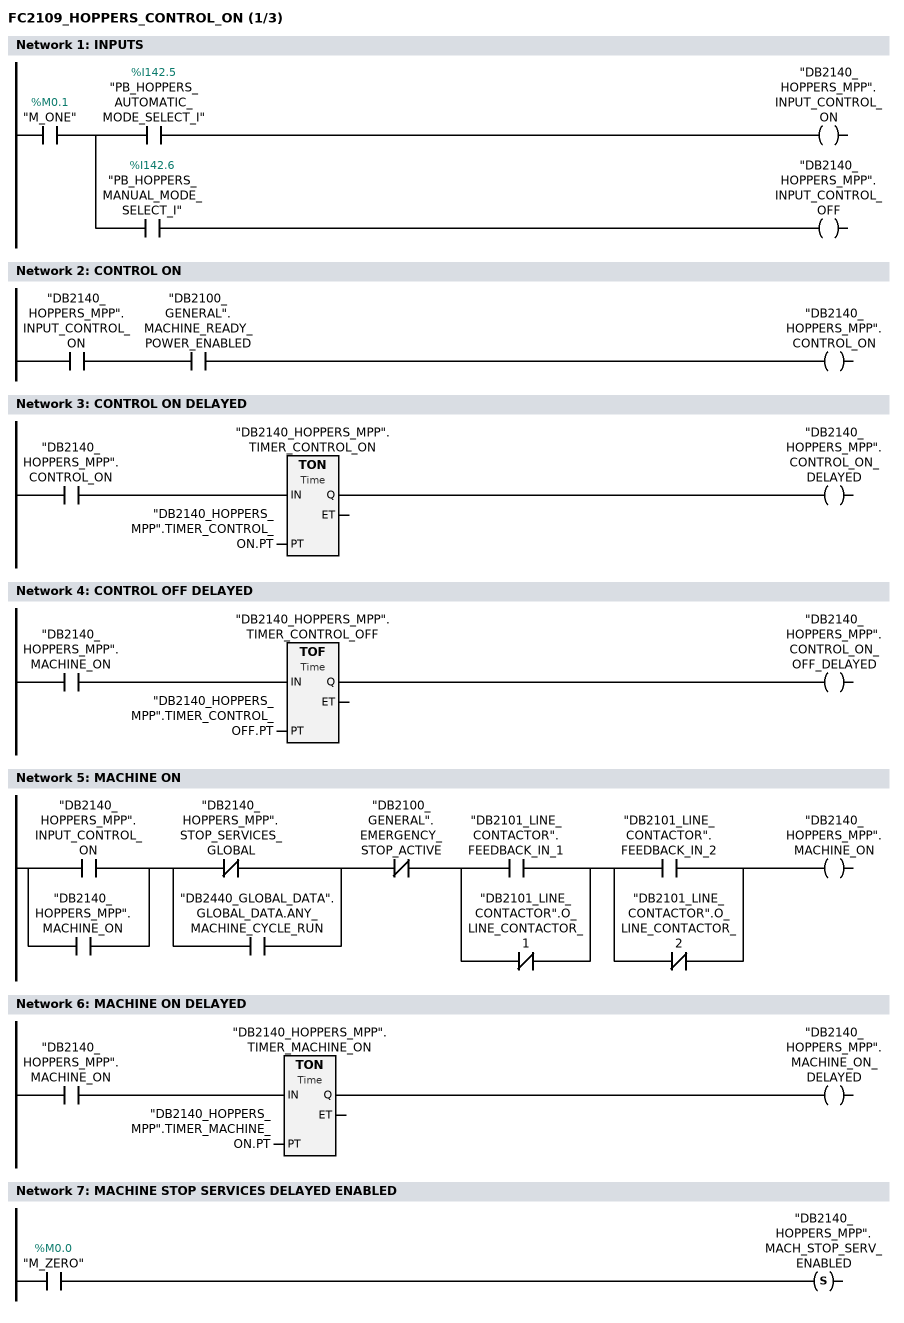
   RUNG wire#powerrail
      Contact( "M_ONE" )
      wire#w1
      Contact( "PB_HOPPERS_AUTOMATIC_MODE_SELECT_I" )
      Coil( "DB2140_HOPPERS_MPP".INPUT_CONTROL_ON )
   END_RUNG
   RUNG wire#w1
      Contact( "PB_HOPPERS_MANUAL_MODE_SELECT_I" )
      Coil( "DB2140_HOPPERS_MPP".INPUT_CONTROL_OFF )
   END_RUNG
   // the same network as SCL:
   "DB2140_HOPPERS_MPP".INPUT_CONTROL_ON := "M_ONE" AND "PB_HOPPERS_AUTOMATIC_MODE_SELECT_I";
   "DB2140_HOPPERS_MPP".INPUT_CONTROL_OFF := "M_ONE" AND "PB_HOPPERS_MANUAL_MODE_SELECT_I";
END_REGION

REGION Network 2: CONTROL ON
   RUNG wire#powerrail
      Contact( "DB2140_HOPPERS_MPP".INPUT_CONTROL_ON )
      Contact( "DB2100_GENERAL".MACHINE_READY_POWER_ENABLED )
      Coil( "DB2140_HOPPERS_MPP".CONTROL_ON )
   END_RUNG
   // the same network as SCL:
   "DB2140_HOPPERS_MPP".CONTROL_ON := "DB2140_HOPPERS_MPP".INPUT_CONTROL_ON AND "DB2100_GENERAL".MACHINE_READY_POWER_ENABLED;
END_REGION

REGION Network 3: CONTROL ON DELAYED
   RUNG wire#powerrail
      Contact( "DB2140_HOPPERS_MPP".CONTROL_ON )
      { S7_Templates := "time_type := Time" } "DB2140_HOPPERS_MPP".TIMER_CONTROL_ON.TON(pt := "DB2140_HOPPERS_MPP".TIMER_CONTROL_ON.PT, et =>)
      Coil( "DB2140_HOPPERS_MPP".CONTROL_ON_DELAYED )
   END_RUNG
   // the same network as SCL:
   "DB2140_HOPPERS_MPP".TIMER_CONTROL_ON.TON(IN := "DB2140_HOPPERS_MPP".CONTROL_ON,
                           PT := "DB2140_HOPPERS_MPP".TIMER_CONTROL_ON.PT);
   "DB2140_HOPPERS_MPP".CONTROL_ON_DELAYED := "DB2140_HOPPERS_MPP".TIMER_CONTROL_ON.Q;
END_REGION

REGION Network 4: CONTROL OFF DELAYED
   RUNG wire#powerrail
      Contact( "DB2140_HOPPERS_MPP".MACHINE_ON )
      { S7_Templates := "time_type := Time" } "DB2140_HOPPERS_MPP".TIMER_CONTROL_OFF.TOF(pt := "DB2140_HOPPERS_MPP".TIMER_CONTROL_OFF.PT, et =>)
      Coil( "DB2140_HOPPERS_MPP".CONTROL_ON_OFF_DELAYED )
   END_RUNG
   // the same network as SCL:
   "DB2140_HOPPERS_MPP".TIMER_CONTROL_OFF.TOF(IN := "DB2140_HOPPERS_MPP".MACHINE_ON,
                           PT := "DB2140_HOPPERS_MPP".TIMER_CONTROL_OFF.PT);
   "DB2140_HOPPERS_MPP".CONTROL_ON_OFF_DELAYED := "DB2140_HOPPERS_MPP".TIMER_CONTROL_OFF.Q;
END_REGION

REGION Network 5: MACHINE ON
   RUNG wire#powerrail
      Contact( "DB2140_HOPPERS_MPP".INPUT_CONTROL_ON )
      wire#w1
      I_Contact( "DB2140_HOPPERS_MPP".STOP_SERVICES_GLOBAL )
      wire#w2
      I_Contact( "DB2100_GENERAL".EMERGENCY_STOP_ACTIVE )
      wire#w3
      Contact( "DB2101_LINE_CONTACTOR".FEEDBACK_IN_1 )
      wire#w4
      Contact( "DB2101_LINE_CONTACTOR".FEEDBACK_IN_2 )
      wire#w5
      Coil( "DB2140_HOPPERS_MPP".MACHINE_ON )
   END_RUNG
   RUNG wire#powerrail
      Contact( "DB2140_HOPPERS_MPP".MACHINE_ON )
   END_RUNG wire#w1
   RUNG wire#w1
      Contact( "DB2440_GLOBAL_DATA".GLOBAL_DATA.ANY_MACHINE_CYCLE_RUN )
   END_RUNG wire#w2
   RUNG wire#w3
      I_Contact( "DB2101_LINE_CONTACTOR".O_LINE_CONTACTOR_1 )
   END_RUNG wire#w4
   RUNG wire#w4
      I_Contact( "DB2101_LINE_CONTACTOR".O_LINE_CONTACTOR_2 )
   END_RUNG wire#w5
   // the same network as SCL:
   "DB2140_HOPPERS_MPP".MACHINE_ON := ("DB2140_HOPPERS_MPP".INPUT_CONTROL_ON OR "DB2140_HOPPERS_MPP".MACHINE_ON) AND (NOT "DB2140_HOPPERS_MPP".STOP_SERVICES_GLOBAL OR "DB2440_GLOBAL_DATA".GLOBAL_DATA.ANY_MACHINE_CYCLE_RUN) AND NOT "DB2100_GENERAL".EMERGENCY_STOP_ACTIVE AND ("DB2101_LINE_CONTACTOR".FEEDBACK_IN_1 OR NOT "DB2101_LINE_CONTACTOR".O_LINE_CONTACTOR_1) AND ("DB2101_LINE_CONTACTOR".FEEDBACK_IN_2 OR NOT "DB2101_LINE_CONTACTOR".O_LINE_CONTACTOR_2);
END_REGION

REGION Network 6: MACHINE ON DELAYED
   RUNG wire#powerrail
      Contact( "DB2140_HOPPERS_MPP".MACHINE_ON )
      { S7_Templates := "time_type := Time" } "DB2140_HOPPERS_MPP".TIMER_MACHINE_ON.TON(pt := "DB2140_HOPPERS_MPP".TIMER_MACHINE_ON.PT, et =>)
      Coil( "DB2140_HOPPERS_MPP".MACHINE_ON_DELAYED )
   END_RUNG
   // the same network as SCL:
   "DB2140_HOPPERS_MPP".TIMER_MACHINE_ON.TON(IN := "DB2140_HOPPERS_MPP".MACHINE_ON,
                           PT := "DB2140_HOPPERS_MPP".TIMER_MACHINE_ON.PT);
   "DB2140_HOPPERS_MPP".MACHINE_ON_DELAYED := "DB2140_HOPPERS_MPP".TIMER_MACHINE_ON.Q;
END_REGION

REGION Network 7: MACHINE STOP SERVICES DELAYED ENABLED
   RUNG wire#powerrail
      Contact( "M_ZERO" )
      S_Coil( "DB2140_HOPPERS_MPP".MACH_STOP_SERV_ENABLED )
   END_RUNG
   // the same network as SCL:
   IF "M_ZERO" THEN "DB2140_HOPPERS_MPP".MACH_STOP_SERV_ENABLED := TRUE; END_IF;
END_REGION

REGION Network 8: MACHINE STOP SERVICES DELAYED ENABLED
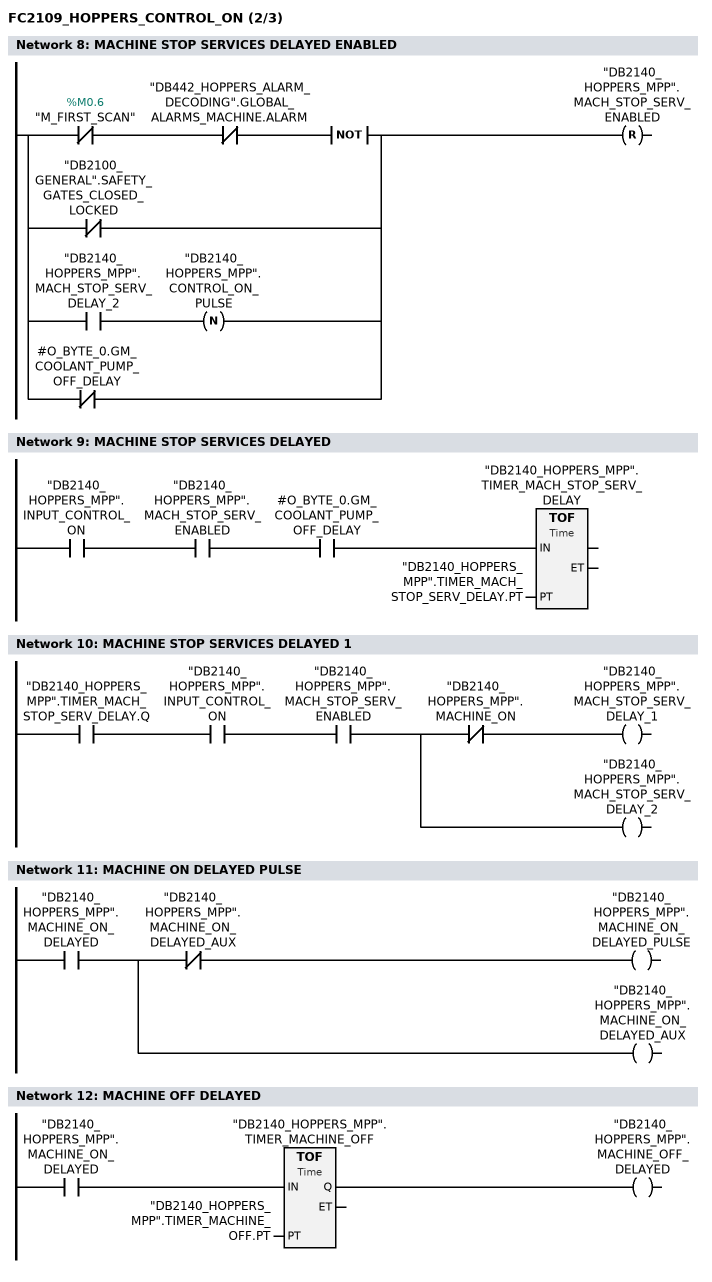
   RUNG wire#powerrail
      I_Contact( "M_FIRST_SCAN" )
      I_Contact( "DB442_HOPPERS_ALARM_DECODING".GLOBAL_ALARMS_MACHINE.ALARM )
      Not()
      wire#w1
      R_Coil( "DB2140_HOPPERS_MPP".MACH_STOP_SERV_ENABLED )
   END_RUNG
   RUNG wire#powerrail
      I_Contact( "DB2100_GENERAL".SAFETY_GATES_CLOSED_LOCKED )
   END_RUNG wire#w1
   RUNG wire#powerrail
      Contact( "DB2140_HOPPERS_MPP".MACH_STOP_SERV_DELAY_2 )
      N_Trig( "DB2140_HOPPERS_MPP".CONTROL_ON_PULSE )
   END_RUNG wire#w1
   RUNG wire#powerrail
      I_Contact( #O_BYTE_0.GM_COOLANT_PUMP_OFF_DELAY )
   END_RUNG wire#w1
   // the same network as SCL:
   #_w1 := NOT "DB2140_HOPPERS_MPP".MACH_STOP_SERV_DELAY_2 AND "DB2140_HOPPERS_MPP".CONTROL_ON_PULSE;   // falling edge
   "DB2140_HOPPERS_MPP".CONTROL_ON_PULSE := "DB2140_HOPPERS_MPP".MACH_STOP_SERV_DELAY_2;
   IF NOT (NOT "M_FIRST_SCAN" AND NOT "DB442_HOPPERS_ALARM_DECODING".GLOBAL_ALARMS_MACHINE.ALARM) OR NOT "DB2100_GENERAL".SAFETY_GATES_CLOSED_LOCKED OR #_w1 OR NOT #O_BYTE_0.GM_COOLANT_PUMP_OFF_DELAY THEN
       "DB2140_HOPPERS_MPP".MACH_STOP_SERV_ENABLED := FALSE;
   END_IF;
END_REGION

REGION Network 9: MACHINE STOP SERVICES DELAYED
   RUNG wire#powerrail
      Contact( "DB2140_HOPPERS_MPP".INPUT_CONTROL_ON )
      Contact( "DB2140_HOPPERS_MPP".MACH_STOP_SERV_ENABLED )
      Contact( #O_BYTE_0.GM_COOLANT_PUMP_OFF_DELAY )
      { S7_Templates := "time_type := Time" } "DB2140_HOPPERS_MPP".TIMER_MACH_STOP_SERV_DELAY.TOF(pt := "DB2140_HOPPERS_MPP".TIMER_MACH_STOP_SERV_DELAY.PT, et =>)
   END_RUNG
   // the same network as SCL:
   "DB2140_HOPPERS_MPP".TIMER_MACH_STOP_SERV_DELAY.TOF(IN := "DB2140_HOPPERS_MPP".INPUT_CONTROL_ON AND "DB2140_HOPPERS_MPP".MACH_STOP_SERV_ENABLED AND #O_BYTE_0.GM_COOLANT_PUMP_OFF_DELAY,
                           PT := "DB2140_HOPPERS_MPP".TIMER_MACH_STOP_SERV_DELAY.PT);
END_REGION

REGION Network 10: MACHINE STOP SERVICES DELAYED 1
   RUNG wire#powerrail
      Contact( "DB2140_HOPPERS_MPP".TIMER_MACH_STOP_SERV_DELAY.Q )
      Contact( "DB2140_HOPPERS_MPP".INPUT_CONTROL_ON )
      Contact( "DB2140_HOPPERS_MPP".MACH_STOP_SERV_ENABLED )
      wire#w1
      I_Contact( "DB2140_HOPPERS_MPP".MACHINE_ON )
      Coil( "DB2140_HOPPERS_MPP".MACH_STOP_SERV_DELAY_1 )
   END_RUNG
   RUNG wire#w1
      Coil( "DB2140_HOPPERS_MPP".MACH_STOP_SERV_DELAY_2 )
   END_RUNG
   // the same network as SCL:
   #_w1 := "DB2140_HOPPERS_MPP".TIMER_MACH_STOP_SERV_DELAY.Q AND "DB2140_HOPPERS_MPP".INPUT_CONTROL_ON AND "DB2140_HOPPERS_MPP".MACH_STOP_SERV_ENABLED;
   "DB2140_HOPPERS_MPP".MACH_STOP_SERV_DELAY_1 := #_w1 AND NOT "DB2140_HOPPERS_MPP".MACHINE_ON;
   "DB2140_HOPPERS_MPP".MACH_STOP_SERV_DELAY_2 := #_w1;
END_REGION

REGION Network 11: MACHINE ON DELAYED PULSE
   RUNG wire#powerrail
      Contact( "DB2140_HOPPERS_MPP".MACHINE_ON_DELAYED )
      wire#w1
      I_Contact( "DB2140_HOPPERS_MPP".MACHINE_ON_DELAYED_AUX )
      Coil( "DB2140_HOPPERS_MPP".MACHINE_ON_DELAYED_PULSE )
   END_RUNG
   RUNG wire#w1
      Coil( "DB2140_HOPPERS_MPP".MACHINE_ON_DELAYED_AUX )
   END_RUNG
   // the same network as SCL:
   "DB2140_HOPPERS_MPP".MACHINE_ON_DELAYED_PULSE := "DB2140_HOPPERS_MPP".MACHINE_ON_DELAYED AND NOT "DB2140_HOPPERS_MPP".MACHINE_ON_DELAYED_AUX;
   "DB2140_HOPPERS_MPP".MACHINE_ON_DELAYED_AUX := "DB2140_HOPPERS_MPP".MACHINE_ON_DELAYED;
END_REGION

REGION Network 12: MACHINE OFF DELAYED
   RUNG wire#powerrail
      Contact( "DB2140_HOPPERS_MPP".MACHINE_ON_DELAYED )
      { S7_Templates := "time_type := Time" } "DB2140_HOPPERS_MPP".TIMER_MACHINE_OFF.TOF(pt := "DB2140_HOPPERS_MPP".TIMER_MACHINE_OFF.PT, et =>)
      Coil( "DB2140_HOPPERS_MPP".MACHINE_OFF_DELAYED )
   END_RUNG
   // the same network as SCL:
   "DB2140_HOPPERS_MPP".TIMER_MACHINE_OFF.TOF(IN := "DB2140_HOPPERS_MPP".MACHINE_ON_DELAYED,
                           PT := "DB2140_HOPPERS_MPP".TIMER_MACHINE_OFF.PT);
   "DB2140_HOPPERS_MPP".MACHINE_OFF_DELAYED := "DB2140_HOPPERS_MPP".TIMER_MACHINE_OFF.Q;
END_REGION

REGION Network 13: MACHINE ON DELAYED AND HYDRAULIC AND PNEUMATIC IN SERVICE
